// TwinCAT 3 PLC project PLC
// ProgramVersion: 3.1.4024.0
// libraries:
//   Tc2_Standard, * (Beckhoff Automation GmbH)
//   Tc2_System, * (Beckhoff Automation GmbH)
//   Tc3_Module, * (Beckhoff Automation GmbH)
//   VisuSymbols,3.5.10.0,System
// project tree:
//   DUTs/ Input.TcDUT, Output.TcDUT, WeldRobotIn.TcDUT, WeldRobotOut.TcDUT
//   / GlobalTextList.TcGTLO, PlcTask.TcTTO, Visualization Manager.TcVMO (not stored)
//   GVLs/ Fixt1.TcGVL, Fixt2.TcGVL, Gen.TcGVL, Global.TcGVL, GVL.TcGVL, HMI.TcGVL, MH.TcGVL, Safety.TcGVL, WeldRobot.TcGVL, WeldRobots.TcGVL
//   POUs/ Fixt2_Seq_Call.TcPOU, Fixt2_Seq_Call_1.TcPOU, Fixt2_Seq_Call_1_1.TcPOU, MAIN.TcPOU, Mode_Call.TcPOU, Fixt1_Seq_Call.TcPOU
//   POUs/Library/ FB_AutoSeq.TcPOU, FB_CylinderModule.TcPOU, FB_ModeCall.TcPOU, FB_PartMonitoring_Fixt2.TcPOU, FB_Trunion.TcPOU, FB_TurnTable_0_180.TcPOU, FB_Roller_Door.TcPOU, FB_PartMonitoring_Fixt1.TcPOU
//   VISUs/ Visualization.TcVIS
// real-time tasks:
//   TASK PlcTask: cycle T#10ms, priority 20, ADS port 350
// I/O:
//   DEVICE Device 1 (EtherCAT) (disabled), AmsNetId 192.168.4.1.2.1
//     Term 1 (EK1100) [EK1100 EtherCAT Coupler (2A E-Bus)]
//       Term 2 (EL1008) [EL1008 8Ch. Dig. Input 24V, 3ms]
//       Term 4 (EL1904) [EL1904, 4 Ch. Safety Input 24V, TwinSAFE]
//         modules: Module 1 (FSOES)
//       Term 5 (EL2904) [EL2904, 4 Ch. Safety Output 24V, 0.5A, TwinSAFE]
//         modules: Module 1 (FSOES), Module 2 (DO)
//       Term 6 (EL2008) [EL2008 8Ch. Dig. Output 24V, 0.5A]
//       Term 3 (EL6910) [EL6910, TwinSAFE PLC]
// variable links:
//   Device 1 (EtherCAT) <-> Device 1 (EtherCAT)/Term 1 (EK1100)/Term 3 (EL6910)
//     Term 1 (EK1100)/Term 5 (EL2904)/Module 1 (FSOES)/RxPDO/FSOE <-> ConnectionInputs/TwinSafeGroup1.Term 5 (EL2904) - Module 1 (FSOES)_4 TxPDO
//     Term 1 (EK1100)/Term 5 (EL2904)/Module 1 (FSOES)/TxPDO/FSOE <-> ConnectionOutputs/TwinSafeGroup1.Term 5 (EL2904) - Module 1 (FSOES)_4 RxPDO
//   Device 1 (EtherCAT) <-> Device 1 (EtherCAT)/Term 1 (EK1100)/Term 4 (EL1904)
//     Term 1 (EK1100)/Term 3 (EL6910)/ConnectionInputs/TwinSafeGroup1.Term 4 (EL1904) - Module 1 (FSOES)_3 TxPDO <-> Module 1 (FSOES)/RxPDO/FSOE
//     Term 1 (EK1100)/Term 3 (EL6910)/ConnectionOutputs/TwinSafeGroup1.Term 4 (EL1904) - Module 1 (FSOES)_3 RxPDO <-> Module 1 (FSOES)/TxPDO/FSOE
//   PLC/PLC Instance <-> Device 1 (EtherCAT)/Term 1 (EK1100)/Term 3 (EL6910)
//     PlcTask Outputs/Safety.Ack <-> StandardOutputs/TwinSafeGroup1.ErrorAcknowledgement_1
//     PlcTask Outputs/Safety.sRun <-> StandardOutputs/TwinSafeGroup1.Run_2

CONFIGURATION PLC
    RESOURCE PLC ON TwinCAT3
        TASK PlcTask(INTERVAL := T#10ms, PRIORITY := 20);
        PROGRAM MAIN WITH PlcTask : MAIN;
    END_RESOURCE
END_CONFIGURATION

// ---- DUTs/Input.TcDUT
TYPE Input :
STRUCT
i_Control_Pressure_Sw_In1_BPB1	:	BOOL	;	//	Control Pressure Switch Input 1-BPB1  
i_Control_Pressure_Sw_In2_BPB1	:	Bool	;	//	Control Pressure Switch Input 2-BPB1  
i_Valve_Pos_BGB1	:	Bool	;	//	Valve Position-BGB1
i_Reserve_BPB1_0_3	:	Bool	;	//	Free
i_CC6_Clamp_1_Sensor_HP	:	Bool	;	//	Clamping Circuit 6 Clamping Unit 1 sensor  HP
i_CC6_Clamp_1_Sensor_WP	:	Bool	;	//	Clamping Circuit 6 Clamping Unit 1 sensor  WP
i_CC4_Clamp_3_Sensor_HP	:	Bool	;	//	Clamping Circuit 4 Clamping Unit 3 sensor  HP
i_CC4_Clamp_3_Sensor_WP	:	Bool	;	//	Clamping Circuit 4 Clamping Unit 3 sensor  WP
i_PART_CONTROL_B13	:	Bool	;	//	PART CONTROL  B13
i_PART_CONTROL_B27	:	Bool	;	//	PART CONTROL  B27
i_PART_CONTROL_B14	:	Bool	;	//	PART CONTROL  B14
i_PART_CONTROL_B28	:	Bool	;	//	PART CONTROL  B28
i_Reserve_BGB1_1_4	:	Bool	;	//	Free
i_Reserve_BGB1_1_5	:	Bool	;	//	Free
i_KEC6Salvemodule12_1	:	BOOL	;	//	Connect to KEC6 Salve module 1.2
i_KEC6Salvemodule12_2	:	BOOL	;	//	Connect to KEC6 Salve module 1.2
i_Reserve_2_0	:	Bool	;	//	i_Reserve_2_0
i_Reserve_2_1	:	Bool	;	//	i_Reserve_2_1
i_Reserve_2_2	:	Bool	;	//	i_Reserve_2_2
i_Reserve_2_3	:	Bool	;	//	i_Reserve_2_3
i_Reserve_2_4	:	Bool	;	//	i_Reserve_2_4
i_Reserve_2_5	:	Bool	;	//	i_Reserve_2_5
i_Reserve_2_6	:	Bool	;	//	i_Reserve_2_6
i_Reserve_2_7	:	Bool	;	//	i_Reserve_2_7
i_Reserve_3_0	:	Bool	;	//	i_Reserve_3_0
i_Reserve_3_1	:	Bool	;	//	i_Reserve_3_1
i_Reserve_3_2	:	Bool	;	//	i_Reserve_3_2
i_Reserve_3_3	:	Bool	;	//	i_Reserve_3_3
i_Reserve_3_4	:	Bool	;	//	i_Reserve_3_4
i_Reserve_3_5	:	Bool	;	//	i_Reserve_3_5
i_Reserve_3_6	:	Bool	;	//	i_Reserve_3_6
i_Reserve_3_7	:	Bool	;	//	i_Reserve_3_7
i_CC4_Clamp_1_Sensor_HP	:	Bool	;	//	Clamping Circuit 4 Clamping Unit 1 sensor  HP
i_CC4_Clamp_1_Sensor_WP	:	Bool	;	//	Clamping Circuit 4 Clamping Unit 1 sensor  WP
i_CC4_Clamp_2_Sensor_HP	:	Bool	;	//	Clamping Circuit 4 Clamping Unit 2 sensor  HP
i_CC4_Clamp_2_Sensor_WP	:	Bool	;	//	Clamping Circuit 4 Clamping Unit 2 sensor  WP
i_CC2_Clamp_3_Sensor_HP	:	Bool	;	//	Clamping Circuit 2 Clamping Unit 3 sensor  HP
i_CC2_Clamp_3_Sensor_WP	:	Bool	;	//	Clamping Circuit 2 Clamping Unit 3 sensor  WP
i_PART_CONTROL_B12	:	Bool	;	//	PART CONTROL  B12
i_PART_CONTROL_B26	:	Bool	;	//	PART CONTROL  B26
i_PART_CONTROL_B11	:	Bool	;	//	PART CONTROL  B11
i_PART_CONTROL_B25	:	Bool	;	//	PART CONTROL  B25
i_PART_CONTROL_B10	:	Bool	;	//	PART CONTROL  B10
i_PART_CONTROL_B24	:	Bool	;	//	PART CONTROL  B24
i_Reserve_5_4	:	Bool	;	//	Free
i_Reserve_5_5	:	Bool	;	//	Free
i_Reserve_5_6	:	Bool	;	//	Free
i_Reserve_5_7	:	Bool	;	//	Free
i_Reserve_6_0	:	Bool	;	//	i_Reserve_6_0
i_Reserve_6_1	:	Bool	;	//	i_Reserve_6_1
i_Reserve_6_2	:	Bool	;	//	i_Reserve_6_2
i_Reserve_6_3	:	Bool	;	//	i_Reserve_6_3
i_Reserve_6_4	:	Bool	;	//	i_Reserve_6_4
i_Reserve_6_5	:	Bool	;	//	i_Reserve_6_5
i_Reserve_6_6	:	Bool	;	//	i_Reserve_6_6
i_Reserve_6_7	:	Bool	;	//	i_Reserve_6_7
i_Reserve_7_0	:	Bool	;	//	i_Reserve_7_0
i_Reserve_7_1	:	Bool	;	//	i_Reserve_7_1
i_Reserve_7_2	:	Bool	;	//	i_Reserve_7_2
i_Reserve_7_3	:	Bool	;	//	i_Reserve_7_3
i_Reserve_7_4	:	Bool	;	//	i_Reserve_7_4
i_Reserve_7_5	:	Bool	;	//	i_Reserve_7_5
i_Reserve_7_6	:	Bool	;	//	i_Reserve_7_6
i_Reserve_7_7	:	Bool	;	//	i_Reserve_7_7
i_CC3_Clamp_1_Sensor_HP	:	Bool	;	//	Clamping Circuit 3 Clamping Unit 1 sensor  HP
i_CC3_Clamp_1_Sensor_WP	:	Bool	;	//	Clamping Circuit 3 Clamping Unit 1 sensor  WP
i_CC3_Clamp_2_Sensor_HP	:	Bool	;	//	Clamping Circuit 3 Clamping Unit 2 sensor  HP
i_CC3_Clamp_2_Sensor_WP	:	Bool	;	//	Clamping Circuit 3 Clamping Unit 2 sensor  WP
i_CC3_Clamp_3_Sensor_HP	:	Bool	;	//	Clamping Circuit 3 Clamping Unit 3 sensor  HP
i_CC3_Clamp_3_Sensor_WP	:	Bool	;	//	Clamping Circuit 3 Clamping Unit 3 sensor  WP
i_PART_CONTROL_B7	:	Bool	;	//	PART CONTROL  B7
i_PART_CONTROL_B21	:	Bool	;	//	PART CONTROL  B21
i_PART_CONTROL_B6	:	Bool	;	//	PART CONTROL  B6
i_PART_CONTROL_B20	:	Bool	;	//	PART CONTROL  B20
i_PART_CONTROL_B5	:	Bool	;	//	PART CONTROL  B5
i_PART_CONTROL_B19	:	Bool	;	//	PART CONTROL  B19
i_Reserve_9_4	:	Bool	;	//	Free
i_Reserve_9_5	:	Bool	;	//	Free
i_KEC8Salvemodule22_1	:	BOOL	;	//	Connect to KEC8 Salve module 2.2
i_KEC8Salvemodule22_2	:	BOOL	;	//	Connect to KEC8 Salve module 2.2
i_Reserve_10_0	:	Bool	;	//	i_Reserve_10_0
i_Reserve_10_1	:	Bool	;	//	i_Reserve_10_1
i_Reserve_10_2	:	Bool	;	//	i_Reserve_10_2
i_Reserve_10_3	:	Bool	;	//	i_Reserve_10_3
i_Reserve_10_4	:	Bool	;	//	i_Reserve_10_4
i_Reserve_10_5	:	Bool	;	//	i_Reserve_10_5
i_Reserve_10_6	:	Bool	;	//	i_Reserve_10_6
i_Reserve_10_7	:	Bool	;	//	i_Reserve_10_7
i_Reserve_11_0	:	Bool	;	//	i_Reserve_11_0
i_Reserve_11_1	:	Bool	;	//	i_Reserve_11_1
i_Reserve_11_2	:	Bool	;	//	i_Reserve_11_2
i_Reserve_11_3	:	Bool	;	//	i_Reserve_11_3
i_Reserve_11_4	:	Bool	;	//	i_Reserve_11_4
i_Reserve_11_5	:	Bool	;	//	i_Reserve_11_5
i_Reserve_11_6	:	Bool	;	//	i_Reserve_11_6
i_Reserve_11_7	:	Bool	;	//	i_Reserve_11_7
i_CC1_Clamp_1_Sensor_HP	:	Bool	;	//	Clamping Circuit 1 Clamping Unit 1 sensor  HP
i_CC1_Clamp_1_Sensor_WP	:	Bool	;	//	Clamping Circuit 1 Clamping Unit 1 sensor  WP
i_CC1_Clamp_2_Sensor_HP	:	Bool	;	//	Clamping Circuit 1 Clamping Unit 2 sensor  HP
i_CC1_Clamp_2_Sensor_WP	:	Bool	;	//	Clamping Circuit 1 Clamping Unit 2 sensor  WP
i_CC1_Clamp_3_Sensor_HP	:	Bool	;	//	Clamping Circuit 1 Clamping Unit 3 sensor  HP
i_CC1_Clamp_3_Sensor_WP	:	Bool	;	//	Clamping Circuit 1 Clamping Unit 3 sensor  WP
i_PART_CONTROL_B4	:	Bool	;	//	PART CONTROL  B4
i_PART_CONTROL_B18	:	Bool	;	//	PART CONTROL  B18
i_PART_CONTROL_B3	:	Bool	;	//	PART CONTROL  B3
i_PART_CONTROL_B17	:	Bool	;	//	PART CONTROL  B17
i_PART_CONTROL_B2	:	Bool	;	//	PART CONTROL  B2
i_PART_CONTROL_B16	:	Bool	;	//	PART CONTROL  B16
i_Reserve_13_4	:	Bool	;	//	Free
i_Reserve_13_5	:	Bool	;	//	Free
i_Reserve_13_6	:	Bool	;	//	Free
i_Reserve_13_7	:	Bool	;	//	Free
i_Reserve_14_0	:	Bool	;	//	i_Reserve_14_0
i_Reserve_14_1	:	Bool	;	//	i_Reserve_14_1
i_Reserve_14_2	:	Bool	;	//	i_Reserve_14_2
i_Reserve_14_3	:	Bool	;	//	i_Reserve_14_3
i_Reserve_14_4	:	Bool	;	//	i_Reserve_14_4
i_Reserve_14_5	:	Bool	;	//	i_Reserve_14_5
i_Reserve_14_6	:	Bool	;	//	i_Reserve_14_6
i_Reserve_14_7	:	Bool	;	//	i_Reserve_14_7
i_Reserve_15_0	:	Bool	;	//	i_Reserve_15_0
i_Reserve_15_1	:	Bool	;	//	i_Reserve_15_1
i_Reserve_15_2	:	Bool	;	//	i_Reserve_15_2
i_Reserve_15_3	:	Bool	;	//	i_Reserve_15_3
i_Reserve_15_4	:	Bool	;	//	i_Reserve_15_4
i_Reserve_15_5	:	Bool	;	//	i_Reserve_15_5
i_Reserve_15_6	:	Bool	;	//	i_Reserve_15_6
i_Reserve_15_7	:	Bool	;	//	i_Reserve_15_7
i_CC2_Clamp_1_Sensor_HP	:	Bool	;	//	Clamping Circuit 2 Clamping Unit 1 sensor  HP
i_CC2_Clamp_1_Sensor_WP	:	Bool	;	//	Clamping Circuit 2 Clamping Unit 1 sensor  WP
i_CC2_Clamp_2_Sensor_HP	:	Bool	;	//	Clamping Circuit 2 Clamping Unit 2 sensor  HP
i_CC2_Clamp_2_Sensor_WP	:	Bool	;	//	Clamping Circuit 2 Clamping Unit 2 sensor  WP
i_PART_CONTROL_B9	:	Bool	;	//	PART CONTROL  B9
i_PART_CONTROL_B23	:	Bool	;	//	PART CONTROL  B23
i_PART_CONTROL_B8	:	Bool	;	//	PART CONTROL  B8
i_PART_CONTROL_B22	:	Bool	;	//	PART CONTROL  B22
i_Reserve_17_0	:	Bool	;	//	Free
i_Reserve_17_1	:	Bool	;	//	Free
i_Reserve_17_2	:	Bool	;	//	Free
i_Reserve_17_3	:	Bool	;	//	Free
i_Reserve_17_4	:	Bool	;	//	Free
i_Reserve_17_5	:	Bool	;	//	Free
i_Reserve_17_6	:	Bool	;	//	Free
i_Reserve_17_7	:	Bool	;	//	Free
i_Reserve_18_0	:	Bool	;	//	i_Reserve_18_0
i_Reserve_18_1	:	Bool	;	//	i_Reserve_18_1
i_Reserve_18_2	:	Bool	;	//	i_Reserve_18_2
i_Reserve_18_3	:	Bool	;	//	i_Reserve_18_3
i_Reserve_18_4	:	Bool	;	//	i_Reserve_18_4
i_Reserve_18_5	:	Bool	;	//	i_Reserve_18_5
i_Reserve_18_6	:	Bool	;	//	i_Reserve_18_6
i_Reserve_18_7	:	Bool	;	//	i_Reserve_18_7
i_Reserve_19_0	:	Bool	;	//	i_Reserve_19_0
i_Reserve_19_1	:	Bool	;	//	i_Reserve_19_1
i_Reserve_19_2	:	Bool	;	//	i_Reserve_19_2
i_Reserve_19_3	:	Bool	;	//	i_Reserve_19_3
i_Reserve_19_4	:	Bool	;	//	i_Reserve_19_4
i_Reserve_19_5	:	Bool	;	//	i_Reserve_19_5
i_Reserve_19_6	:	Bool	;	//	i_Reserve_19_6
i_Reserve_19_7	:	Bool	;	//	i_Reserve_19_7
i_Reserve_20_0	:	Bool	;	//	i_Reserve_20_0
i_Reserve_20_1	:	Bool	;	//	i_Reserve_20_1
i_Reserve_20_2	:	Bool	;	//	i_Reserve_20_2
i_Reserve_20_3	:	Bool	;	//	i_Reserve_20_3
i_Reserve_20_4	:	Bool	;	//	i_Reserve_20_4
i_Reserve_20_5	:	Bool	;	//	i_Reserve_20_5
i_Reserve_20_6	:	Bool	;	//	i_Reserve_20_6
i_Reserve_20_7	:	Bool	;	//	i_Reserve_20_7
i_Reserve_21_0	:	Bool	;	//	i_Reserve_21_0
i_Reserve_21_1	:	Bool	;	//	i_Reserve_21_1
i_Reserve_21_2	:	Bool	;	//	i_Reserve_21_2
i_Reserve_21_3	:	Bool	;	//	i_Reserve_21_3
i_Reserve_21_4	:	Bool	;	//	i_Reserve_21_4
i_Reserve_21_5	:	Bool	;	//	i_Reserve_21_5
i_Reserve_21_6	:	Bool	;	//	i_Reserve_21_6
i_Reserve_21_7	:	Bool	;	//	i_Reserve_21_7
i_Reserve_22_0	:	Bool	;	//	i_Reserve_22_0
i_Reserve_22_1	:	Bool	;	//	i_Reserve_22_1
i_Reserve_22_2	:	Bool	;	//	i_Reserve_22_2
i_Reserve_22_3	:	Bool	;	//	i_Reserve_22_3
i_Reserve_22_4	:	Bool	;	//	i_Reserve_22_4
i_Reserve_22_5	:	Bool	;	//	i_Reserve_22_5
i_Reserve_22_6	:	Bool	;	//	i_Reserve_22_6
i_Reserve_22_7	:	Bool	;	//	i_Reserve_22_7
i_Reserve_23_0	:	Bool	;	//	i_Reserve_23_0
i_Reserve_23_1	:	Bool	;	//	i_Reserve_23_1
i_Reserve_23_2	:	Bool	;	//	i_Reserve_23_2
i_Reserve_23_3	:	Bool	;	//	i_Reserve_23_3
i_Reserve_23_4	:	Bool	;	//	i_Reserve_23_4
i_Reserve_23_5	:	Bool	;	//	i_Reserve_23_5
i_Reserve_23_6	:	Bool	;	//	i_Reserve_23_6
i_Reserve_23_7	:	Bool	;	//	i_Reserve_23_7
i_CC5_Clamp_1_Sensor_HP	:	Bool	;	//	Clamping Circuit 5 Clamping Unit 1 sensor  HP
i_CC5_Clamp_1_Sensor_WP	:	Bool	;	//	Clamping Circuit 5 Clamping Unit 1 sensor  WP
i_PART_CONTROL_B1	:	Bool	;	//	PART CONTROL  B1
i_PART_CONTROL_B15	:	Bool	;	//	PART CONTROL  B15
i_Reserve_24_4	:	Bool	;	//	Free
i_Reserve_24_5	:	Bool	;	//	Free
i_Reserve_24_6	:	Bool	;	//	Free
i_Reserve_24_7	:	Bool	;	//	Free
i_Reserve_25_0	:	Bool	;	//	Free
i_Reserve_25_1	:	Bool	;	//	Free
i_Reserve_25_2	:	Bool	;	//	Free
i_Reserve_25_3	:	Bool	;	//	Free
i_Reserve_25_4	:	Bool	;	//	Free
i_Reserve_25_5	:	Bool	;	//	Free
i_Reserve_25_6	:	Bool	;	//	Free
i_Reserve_25_7	:	Bool	;	//	Free
i_Reserve_26_0	:	Bool	;	//	i_Reserve_26_0
i_Reserve_26_1	:	Bool	;	//	i_Reserve_26_1
i_Reserve_26_2	:	Bool	;	//	i_Reserve_26_2
i_Reserve_26_3	:	Bool	;	//	i_Reserve_26_3
i_Reserve_26_4	:	Bool	;	//	i_Reserve_26_4
i_Reserve_26_5	:	Bool	;	//	i_Reserve_26_5
i_Reserve_26_6	:	Bool	;	//	i_Reserve_26_6
i_Reserve_26_7	:	Bool	;	//	i_Reserve_26_7
i_Reserve_27_0	:	Bool	;	//	i_Reserve_27_0
i_Reserve_27_1	:	Bool	;	//	i_Reserve_27_1
i_Reserve_27_2	:	Bool	;	//	i_Reserve_27_2
i_Reserve_27_3	:	Bool	;	//	i_Reserve_27_3
i_Reserve_27_4	:	Bool	;	//	i_Reserve_27_4
i_Reserve_27_5	:	Bool	;	//	i_Reserve_27_5
i_Reserve_27_6	:	Bool	;	//	i_Reserve_27_6
i_Reserve_27_7	:	Bool	;	//	i_Reserve_27_7
i_Reserve_28_0	:	Bool	;	//	i_Reserve_28_0
i_Reserve_28_1	:	Bool	;	//	i_Reserve_28_1
i_Reserve_28_2	:	Bool	;	//	i_Reserve_28_2
i_Reserve_28_3	:	Bool	;	//	i_Reserve_28_3
i_Reserve_28_4	:	Bool	;	//	i_Reserve_28_4
i_Reserve_28_5	:	Bool	;	//	i_Reserve_28_5
i_Reserve_28_6	:	Bool	;	//	i_Reserve_28_6
i_Reserve_28_7	:	Bool	;	//	i_Reserve_28_7
i_Reserve_29_0	:	Bool	;	//	i_Reserve_29_0
i_Reserve_29_1	:	Bool	;	//	i_Reserve_29_1
i_Reserve_29_2	:	Bool	;	//	i_Reserve_29_2
i_Reserve_29_3	:	Bool	;	//	i_Reserve_29_3
i_Reserve_29_4	:	Bool	;	//	i_Reserve_29_4
i_Reserve_29_5	:	Bool	;	//	i_Reserve_29_5
i_Reserve_29_6	:	Bool	;	//	i_Reserve_29_6
i_Reserve_29_7	:	Bool	;	//	i_Reserve_29_7
i_Reserve_30_0	:	Bool	;	//	i_Reserve_30_0
i_Reserve_30_1	:	Bool	;	//	i_Reserve_30_1
i_Reserve_30_2	:	Bool	;	//	i_Reserve_30_2
i_Reserve_30_3	:	Bool	;	//	i_Reserve_30_3
i_Reserve_30_4	:	Bool	;	//	i_Reserve_30_4
i_Reserve_30_5	:	Bool	;	//	i_Reserve_30_5
i_Reserve_30_6	:	Bool	;	//	i_Reserve_30_6
i_Reserve_30_7	:	Bool	;	//	i_Reserve_30_7
i_Reserve_31_0	:	Bool	;	//	i_Reserve_31_0
i_Reserve_31_1	:	Bool	;	//	i_Reserve_31_1
i_Reserve_31_2	:	Bool	;	//	i_Reserve_31_2
i_Reserve_31_3	:	Bool	;	//	i_Reserve_31_3
i_Reserve_31_4	:	Bool	;	//	i_Reserve_31_4
i_Reserve_31_5	:	Bool	;	//	i_Reserve_31_5
i_Reserve_31_6	:	Bool	;	//	i_Reserve_31_6
i_Reserve_31_7	:	Bool	;	//	i_Reserve_31_7

END_STRUCT
END_TYPE

// ---- DUTs/Output.TcDUT
TYPE Output :
STRUCT
o_CC1_CLAMPING_UNIT1_3_WP	:	BOOL	;	//	Clamping Circuit 1 Clamping Unit 1-3  WP
o_CC1_CLAMPING_UNIT1_3_HP	:	Bool	;	//	Clamping Circuit 1 Clamping Unit 1-3  HP
o_CC2_CLAMPING_UNIT2_3_WP	:	Bool	;	//	Clamping Circuit 2 Clamping Unit 1-3  WP
o_CC2_CLAMPING_UNIT2_3_HP	:	Bool	;	//	Clamping Circuit 2 Clamping Unit 1-3  HP
o_CC3_CLAMPING_UNIT3_3_WP	:	Bool	;	//	Clamping Circuit 3 Clamping Unit 1-3  WP
o_CC3_CLAMPING_UNIT3_3_HP	:	Bool	;	//	Clamping Circuit 3 Clamping Unit 1-3  HP
o_CC4_CLAMPING_UNIT4_3_WP	:	Bool	;	//	Clamping Circuit 4 Clamping Unit 1-3  WP
o_CC4_CLAMPING_UNIT4_3_HP	:	Bool	;	//	Clamping Circuit 4 Clamping Unit 1-3  HP
o_CC5_CLAMPING_UNIT5_1_WP	:	Bool	;	//	Clamping Circuit 5 Clamping Unit 1  WP
o_CC5_CLAMPING_UNIT5_1_HP	:	Bool	;	//	Clamping Circuit 5 Clamping Unit 1  HP
o_CC6_CLAMPING_UNIT6_1_WP	:	Bool	;	//	Clamping Circuit 6 Clamping Unit 1  WP
o_CC6_CLAMPING_UNIT6_1_HP	:	Bool	;	//	Clamping Circuit 6 Clamping Unit 1  HP
o_RESERVE_1_4	:	Bool	;	//	Free
o_RESERVE_1_5	:	Bool	;	//	Free
o_RESERVE_1_6	:	Bool	;	//	Free
o_RESERVE_1_7	:	Bool	;	//	Free
o_RESERVE_2_0	:	Bool	;	//	Free
o_RESERVE_2_1	:	Bool	;	//	Free
o_RESERVE_2_2	:	Bool	;	//	Free
o_RESERVE_2_3	:	Bool	;	//	Free
o_RESERVE_2_4	:	Bool	;	//	Free
o_RESERVE_2_5	:	Bool	;	//	Free
o_RESERVE_2_6	:	Bool	;	//	Free
o_RESERVE_2_7	:	Bool	;	//	Free
o_RESERVE_3_0	:	Bool	;	//	Free
o_RESERVE_3_1	:	Bool	;	//	Free
o_RESERVE_3_2	:	Bool	;	//	Free
o_RESERVE_3_3	:	Bool	;	//	Free
o_RESERVE_3_4	:	Bool	;	//	Free
o_RESERVE_3_5	:	Bool	;	//	Free
o_RESERVE_3_6	:	Bool	;	//	Free
o_RESERVE_3_7	:	Bool	;	//	Free

END_STRUCT
END_TYPE

// ---- DUTs/WeldRobotIn.TcDUT
TYPE WeldRobotIn :
STRUCT
	iMainJobActive: BOOL;
	iAtParkPos: BOOL;
	iWeldOn:BOOL;
	iProgramNumber: INT;
	Pos_20      : BOOL;
    Pos_0       : BOOL;   // 0 degree feedback
    Pos_M45     : BOOL;
    Pos_M80     : BOOL;
	LS_0        : BOOL;
    LS_180      : BOOL;
	
END_STRUCT
END_TYPE

// ---- DUTs/WeldRobotOut.TcDUT
TYPE WeldRobotOut :
STRUCT
	oProgramNumber: INT;
	oWeldStart: BOOL;
	Move_20     : BOOL;
    Move_0      : BOOL;   // Move to 0 degree
    Move_M45    : BOOL;
    Move_M80    : BOOL;
	Motor_CW_0    : BOOL;
    Motor_CCW_180   : BOOL;
END_STRUCT
END_TYPE

// ---- GVLs/Fixt1.TcGVL
{attribute 'qualified_only'}
VAR_GLOBAL
	I AT %I* :Input;
	O AT %Q* :Output;
	Seq:FB_AutoSeq;
	Trunion:FB_Trunion;
END_VAR

// ---- GVLs/Fixt2.TcGVL
{attribute 'qualified_only'}
VAR_GLOBAL
	I AT %I* :Input;
	O AT %Q* :Output;
	Seq:FB_AutoSeq;
	Trunion:FB_Trunion;
END_VAR

// ---- GVLs/Gen.TcGVL
{attribute 'qualified_only'}
VAR_GLOBAL
	ix_RCD_fuse_fdb	AT	%I*	:	BOOL	;
ix_24VDC_Fuse_TBA1_OK	AT	%I*	:	Bool	;
ix_AIEnergyMeterCbFbOK	AT	%I*	:	BOOL	;
ix_24VDC_Fuse1_OK	AT	%I*	:	Bool	;
ix_24VDC_Fuse2_OK	AT	%I*	:	Bool	;
ix_24VDC_Fuse3_OK	AT	%I*	:	Bool	;
ix_Reserve_0_6	AT	%I*	:	Bool	;
ix_24VDC_PowerSupply_Lightning_OK	AT	%I*	:	Bool	;
ix_TBA2FCB8_Cb_fbb	AT	%I*	:	BOOL	;
ix_AirConditioner_MainCabinet_Error_fdb	AT	%I*	:	Bool	;
ix_RD1_PowerSupply_fdb	AT	%I*	:	Bool	;
ix_RD2_PowerSupply_fdb	AT	%I*	:	Bool	;
ix_Ventilation_Malfunction_fdb	AT	%I*	:	Bool	;
ix_Ventilation_Operating_fdb	AT	%I*	:	Bool	;
ix_BGB1_door_lmt_Sw1_fdb	AT	%I*	:	Bool	;
ix_BGB1_door_lmt_Sw2_fdb	AT	%I*	:	Bool	;
ix_PowerSource_AW1_PowerSupply_fdb	AT	%I*	:	Bool	;
ix_PowerSource_AW1_ON	AT	%I*	:	Bool	;
ix_PowerSource_AW2_PowerSupply_fdb	AT	%I*	:	Bool	;
ix_PowerSource_AW2_ON	AT	%I*	:	Bool	;
ix_RC1_PowerSupply_OK	AT	%I*	:	Bool	;
ix_RC2_PowerSupply_OK	AT	%I*	:	Bool	;
ix_PB_RD2_Open	AT	%I*	:	Bool	;
ix_PB_RD2_Close	AT	%I*	:	Bool	;
ix_RD2_isReady	AT	%I*	:	Bool	;
ix_RD2_isOpen_top	AT	%I*	:	Bool	;
ix_RD2_safetyedge	AT	%I*	:	Bool	;
ix_CompressedAir_Pressure_OK	AT	%I*	:	Bool	;
ix_FlowRate_Sensor_outputA	AT	%I*	:	Bool	;
ix_FlowRate_Sensor_outputB	AT	%I*	:	Bool	;
ix_WireEnd_Sensor_R1	AT	%I*	:	Bool	;
ix_WireEnd_Sensor_R2	AT	%I*	:	Bool	;
ix_PB_PowerON	AT	%I*	:	Bool	;
ix_PB_PowerOFF	AT	%I*	:	Bool	;
ix_PB_Reset	AT	%I*	:	Bool	;
ix_PB_Start	AT	%I*	:	Bool	;
ix_PB_ack_LB	AT	%I*	:	Bool	;
ix_PB_Rbt_Start_Stop	AT	%I*	:	Bool	;
ix_RD1_isReady	AT	%I*	:	Bool	;
ix_RD1_isOpen_top	AT	%I*	:	Bool	;
ix_RD1_Safetyedge	AT	%I*	:	Bool	;
ix_ControlOn	AT	%I*	:	BOOL	;
ix_Reserve_201_2	AT	%I*	:	Bool	;
ix_Reserve_201_3	AT	%I*	:	Bool	;
ix_Reserve_201_4	AT	%I*	:	Bool	;
ix_Reserve_201_5	AT	%I*	:	Bool	;
ix_PB_preAck_UB2	AT	%I*	:	Bool	;
ix_Reserve_201_7	AT	%I*	:	Bool	;
qx_Light_InputArea_ON	AT	%Q*	:	Bool	;
qx_Light_WorkArea_ON	AT	%Q*	:	Bool	;
qx_AirConditionerTurn_ON	AT	%Q*	:	Bool	;
qx_CabinetLight_ON	AT	%Q*	:	Bool	;
qx_ControlPixelCameraST9100	AT	%Q*	:	Bool	;
qx_Valve_CompressedAir_ON	AT	%Q*	:	Bool	;
qx_Valve_GasON_Rob1	AT	%Q*	:	Bool	;
qx_Valve_blowOut_Rob1	AT	%Q*	:	Bool	;
qx_Valve_GasON_Rob2	AT	%Q*	:	Bool	;
qx_Valve_blowOut_Rob2	AT	%Q*	:	Bool	;
qx_Valve_GasON_Rob3	AT	%Q*	:	Bool	;
qx_Valve_blowOut_Rob3	AT	%Q*	:	Bool	;
qx_Valve_GasON_Rob4	AT	%Q*	:	Bool	;
qx_Valve_blowOut_Rob4	AT	%Q*	:	Bool	;
qx_Reserve_1_6	AT	%Q*	:	Bool	;
qx_IL_preAck_Box_UB2	AT	%Q*	:	Bool	;
qx_Reserve_2_0	AT	%Q*	:	Bool	;
qx_Reserve_2_1	AT	%Q*	:	Bool	;
qx_Reserve_2_2	AT	%Q*	:	Bool	;
qx_Reserve_2_3	AT	%Q*	:	Bool	;
qx_Reserve_2_4	AT	%Q*	:	Bool	;
qx_Reserve_2_5	AT	%Q*	:	Bool	;
qx_Reserve_2_6	AT	%Q*	:	Bool	;
qx_Reserve_2_7	AT	%Q*	:	Bool	;
qx_Reserve_3_0	AT	%Q*	:	Bool	;
qx_Reserve_3_1	AT	%Q*	:	Bool	;
qx_Reserve_3_2	AT	%Q*	:	Bool	;
qx_Reserve_3_3	AT	%Q*	:	Bool	;
qx_Reserve_3_4	AT	%Q*	:	Bool	;
qx_Reserve_3_5	AT	%Q*	:	Bool	;
qx_Reserve_3_6	AT	%Q*	:	Bool	;
qx_Reserve_3_7	AT	%Q*	:	Bool	;
qx_RD2_open_narrow_hight	AT	%Q*	:	Bool	;
qx_RD2_open_FullHight	AT	%Q*	:	Bool	;
qx_RD2_close	AT	%Q*	:	Bool	;
qx_Ventilation_ON	AT	%Q*	:	Bool	;
qx_Reserve_6_0	AT	%Q*	:	Bool	;
qx_Reserve_6_1	AT	%Q*	:	Bool	;
qx_Reserve_6_2	AT	%Q*	:	Bool	;
qx_Reserve_6_3	AT	%Q*	:	Bool	;
qx_IL_PowerON	AT	%Q*	:	Bool	;
qx_IL_Reset_PB	AT	%Q*	:	Bool	;
qx_IL_Start_PB	AT	%Q*	:	Bool	;
qx_IL_ack_LB_PB	AT	%Q*	:	Bool	;
qx_IL_RbtStartStop_PB	AT	%Q*	:	Bool	;
qx_Reserve_200_5	AT	%Q*	:	Bool	;
qx_Reserve_200_6	AT	%Q*	:	Bool	;
qx_Reserve_200_7	AT	%Q*	:	Bool	;
qx_Reserve_201_0	AT	%Q*	:	Bool	;
qx_Reserve_201_1	AT	%Q*	:	Bool	;
qx_Reserve_201_2	AT	%Q*	:	Bool	;
qx_Reserve_201_3	AT	%Q*	:	Bool	;
qx_Reserve_201_4	AT	%Q*	:	Bool	;
qx_Reserve_201_5	AT	%Q*	:	Bool	;
qx_Reserve_201_6	AT	%Q*	:	Bool	;
qx_Reserve_201_7	AT	%Q*	:	Bool	;
qx_RD1_open_narrow_hight	AT	%Q*	:	Bool	;
qx_RD1_open_fullHight	AT	%Q*	:	Bool	;
qx_RD1_close	AT	%Q*	:	Bool	;
qx_Reserve_202_3	AT	%Q*	:	Bool	;

END_VAR

// ---- GVLs/Global.TcGVL
{attribute 'qualified_only'}
VAR_GLOBAL
	ModeMang:FB_ModeCall;
	Clamp_1:FB_CylinderModule;
	Clamp_2:FB_CylinderModule;
	Clamp_3:FB_CylinderModule;
	Clamp_4:FB_CylinderModule;
	Clamp_5:FB_CylinderModule;
	Clamp_6:FB_CylinderModule;
	RD1:FB_Roller_Door;
	RD2:FB_Roller_Door;
	Htable:FB_TurnTable_0_180;
END_VAR

// ---- GVLs/GVL.TcGVL
{attribute 'qualified_only'}
VAR_GLOBAL
	start AT %I*:BOOL;
	start1 AT %I*:BOOL;
	FB_ModeCall_0: FB_ModeCall;
END_VAR

// ---- GVLs/HMI.TcGVL
{attribute 'qualified_only'}
VAR_GLOBAL
	Cycle_Start:BOOL;
	Cycle_Stop:BOOL;
	AutoMode:BOOL;
	ManualMode:BOOL;
	Estop:BOOL;
	Reset:BOOL;
	
END_VAR

// ---- GVLs/MH.TcGVL
{attribute 'qualified_only'}
VAR_GLOBAL
//qx_7102R1_CellToHandling	AT	%Q*	:	//udt_HDL_CellToHandling	;	//	
qStatus	AT	%Q*	:	WORD	;	//	0 Auto -- 1 Auto Startup -- 2 Manual -- 3 Error -- 4 LineMode -- 5 PowerOn -- 6 EnergySave -- 7 SafeOk
qTime_Stamp	AT	%Q*	:	DATE_AND_TIME	;	//	
qPartId	AT	%Q*	:	DINT	;	//	Unique Part Id (DMC Serial Number)
qState	AT	%Q*	:	BOOL	;	//	Part state 0=OK, 1=NOK
qPartType	AT	%Q*	:	BOOL	;	//	Part type 1=Long, 0=Short
qExists	AT	%Q*	:	BOOL	;	//	Part exist
qRequest	AT	%Q*	:	USINT	;	//	20 - Pick, 10 - Drop
qRequestPartType	AT	%Q*	:	BOOL	;	//	Part types
qGateOpened	AT	%Q*	:	BOOL	;	//	Handling gate opened
qGateClosed	AT	%Q*	:	BOOL	;	//	Handling gate closed
qFixtureReady	AT	%Q*	:	BOOL	;	//	Postioner in Cube
qRaiseEnable1	AT	%Q*	:	BOOL	;	//	Handshake for raise to go all the way OUT
qRaiseEnable2	AT	%Q*	:	BOOL	;	//	Handshake for raise to go all the way OUT
qReduceEnable1	AT	%Q*	:	BOOL	;	//	Handshake for reduce to go all the way IN
qReduceEnable2	AT	%Q*	:	BOOL	;	//	Handshake for reduce to go all the way IN
qPickJobAck	AT	%Q*	:	BOOL	;	//	Handshake for pick job end
qDropJobAck	AT	%Q*	:	BOOL	;	//	Handshake for drop job end
qHold	AT	%Q*	:	BOOL	;	//	Robot hold
qGripper1ReadyToClose	AT	%Q*	:	BOOL	;	//	Gripper1ReadyToClose
qGripper1ReadyToOpen	AT	%Q*	:	BOOL	;	//	Gripper1ReadyToOpen
qGripper2ReadyToClose	AT	%Q*	:	BOOL	;	//	Gripper2ReadyToClose
qGripper2ReadyToOpen	AT	%Q*	:	BOOL	;	//	Gripper2ReadyToOpen
qFeatureBit6	AT	%Q*	:	BOOL	;	//	Free use
qFeatureBit7	AT	%Q*	:	BOOL	;	//	Free use
//	AT	%Q*	:		;	//	
//ix_7102R1_HandlingToCell	AT	%I*	:	//udt_HDL_HandlingToCell	;	//	
iStatus	AT	%I*	:	WORD	;	//	0 Auto -- 1 Auto Startup -- 2 Manual -- 3 Error -- 4 LineMode -- 5 PowerOn -- 6 EnergySave -- 7 SafeOk
iPartId	AT	%I*	:	DINT	;	//	Unique Part Id (DMC Serial Number)
iState	AT	%I*	:	BOOL	;	//	Part state 0=OK, 1=NOK
iPartType	AT	%I*	:	BOOL	;	//	Part type 1=Long, 0=Short
iExists	AT	%I*	:	BOOL	;	//	Part exist
iGateOpenRequest	AT	%I*	:	BOOL	;	//	Open handling gate
iGateCloseRequest	AT	%I*	:	BOOL	;	//	Close handling gate
iPickJobProceed	AT	%I*	:	BOOL	;	//	Pick job active
iDropJobProceed	AT	%I*	:	BOOL	;	//	Drop job active
iRaiseFinished1	AT	%I*	:	BOOL	;	//	Handshake for raise/ Robot reach at out off fixture pos
iRaiseFinished2	AT	%I*	:	BOOL	;	//	Handshake for reduce/Robot reach at into fixture pos
iReduceFinished1	AT	%I*	:	BOOL	;	//	Handshake for pick job end
iReduceFinished2	AT	%I*	:	BOOL	;	//	Handshake for drop job end
iPickJobOK	AT	%I*	:	BOOL	;	//	Robot in station area/robot infront of cell area
iDropJobOK	AT	%I*	:	BOOL	;	//	PickJobOK
iInArea	AT	%I*	:	BOOL	;	//	DropJobOK
iPickDropProceed	AT	%I*	:	BOOL	;	//	InArea
iGripper1ClosedAck	AT	%I*	:	BOOL	;	//	PickDropProceed
iGripper1OpenedAck	AT	%I*	:	BOOL	;	//	Gripper1OpenedAck
iGripper2ClosedAck	AT	%I*	:	BOOL	;	//	Gripper2ClosedAck
iGripper2OpenedAck	AT	%I*	:	BOOL	;	//	Gripper2OpenedAck
iFeatureBit6	AT	%I*	:	BOOL	;	//	Free use
iFeatureBit7	AT	%I*	:	BOOL	;	//	Free use

END_VAR

// ---- GVLs/Safety.TcGVL
{attribute 'qualified_only'}
VAR_GLOBAL
		ixf_CA1_PowerON_vs	AT	%I*	:	BOOL	;	//	
	ixf_RD2_PowerON_vs	AT	%I*	:	Bool	;	//	
	ixf_FXC1_Safe_24VDC_vs	AT	%I*	:	Bool	;	//	
	ixf_FXC2_Safe_24VDC_vs	AT	%I*	:	Bool	;	//	
	ixf_AW1_PowerSource_vs	AT	%I*	:	Bool	;	//	
	ixf_AW2_PowerSource_vs	AT	%I*	:	Bool	;	//	
	ixf_FXC1_Safe_AirON_vs	AT	%I*	:	Bool	;	//	
	ixf_FXC2_Safe_AirON_vs	AT	%I*	:	Bool	;	//	
	ixf_CA1_EStop_ch1	AT	%I*	:	Bool	;	//	
	ixf_UB3_EStop_ch1	AT	%I*	:	Bool	;	//	
	ixf_UB2_EStop_ch1	AT	%I*	:	Bool	;	//	
	ixf_RD2_isClosed_ch1	AT	%I*	:	Bool	;	//	
	ixf_CA1_EStop_ch2	AT	%I*	:	Bool	;	//	
	ixf_UB3_EStop_ch2	AT	%I*	:	Bool	;	//	
	ixf_UB2_EStop_ch2	AT	%I*	:	Bool	;	//	
	ixf_RD2_isClosed_ch2	AT	%I*	:	Bool	;	//	
	//ixf_CA1_EStop_ch1_vs	AT	%I*	:	Bool	;	//	
	//ixf_UB3_EStop_ch1_vs	AT	%I*	:	Bool	;	//	
	//ixf_UB2_EStop_ch1_vs	AT	%I*	:	Bool	;	//	
	//ixf_RD2_isClosed_ch1_vs	AT	%I*	:	Bool	;	//	
	//ixf_CA1_EStop_ch2_vs	AT	%I*	:	Bool	;	//	
	//ixf_UB3_EStop_ch2_vs	AT	%I*	:	Bool	;	//	
	//ixf_UB2_EStop_ch2_vs	AT	%I*	:	Bool	;	//	
	//ixf_RD2_isClosed_ch2_vs	AT	%I*	:	Bool	;	//	
	//ixf_Reserve_300700_0	AT	%I*	:	Bool	;	//	
	//ixf_Reserve_300700_1	AT	%I*	:	Bool	;	//	
	//ixf_Reserve_300700_2	AT	%I*	:	Bool	;	//	
	//ixf_Reserve_300700_3	AT	%I*	:	Bool	;	//	
	//ixf_Reserve_300700_4	AT	%I*	:	Bool	;	//	
	//ixf_Reserve_300700_5	AT	%I*	:	Bool	;	//	
	//ixf_Reserve_300700_6	AT	%I*	:	Bool	;	//	
	//ixf_Reserve_300700_7	AT	%I*	:	Bool	;	//	
	//ixf_RD1_PowerON_vs	AT	%I*	:	Bool	;	//	
	ixf_UB1_EStop_ch1	AT	%I*	:	Bool	;	//	
	ixf_LB1_InputArea_ch1	AT	%I*	:	Bool	;	//	
	ixf_SW_AutomaticMode	AT	%I*	:	Bool	;	//	
	ixf_RD1_isClosed_ch1	AT	%I*	:	Bool	;	//	
	ixf_UB1_EStop_ch2	AT	%I*	:	Bool	;	//	
	ixf_SW_ManualMode	AT	%I*	:	Bool	;	//	
	ixf_RD1_isClosed_ch2	AT	%I*	:	Bool	;	//	
	//ixf_UB1_EStop_ch1_vs	AT	%I*	:	Bool	;	//	
	//ixf_LB1_InputArea_vs	AT	%I*	:	Bool	;	//	
	//ixf_SW_AutomaticMode_vs	AT	%I*	:	Bool	;	//	
	//ixf_RD1_isClosed_ch1_vs	AT	%I*	:	Bool	;	//	
	//ixf_UB1_EStop_ch2_vs	AT	%I*	:	Bool	;	//	
	//ixf_SW_ManualMode_vs	AT	%I*	:	Bool	;	//	
	//ixf_RD1_isClosed_ch2_vs	AT	%I*	:	Bool	;	//	
	//ixf_Reserve_30150_0	AT	%I*	:	Bool	;	//	
	//ixf_Reserve_30150_1	AT	%I*	:	Bool	;	//	
	//ixf_Reserve_30150_2	AT	%I*	:	Bool	;	//	
	//ixf_Reserve_30150_3	AT	%I*	:	Bool	;	//	
	//ixf_Reserve_30150_4	AT	%I*	:	Bool	;	//	
	//ixf_Reserve_30150_5	AT	%I*	:	Bool	;	//	
	//ixf_Reserve_30150_6	AT	%I*	:	Bool	;	//	
	//ixf_Reserve_30150_7	AT	%I*	:	Bool	;	//	Seq_Reset_WM
	qxf_CA1_PowerON	AT	%Q*	:	Bool	;	//	
	qxf_RD2_PowerON	AT	%Q*	:	Bool	;	//	
	qxf_FXC1_Safe_24VDC	AT	%Q*	:	Bool	;	//	
	qxf_FXC2_Safe_24VDC	AT	%Q*	:	Bool	;	//	
	qxf_AW1_PowerON	AT	%Q*	:	Bool	;	//	
	qxf_AW2_PowerON	AT	%Q*	:	Bool	;	//	
	qxf_FXC1_Safe_AirON	AT	%Q*	:	Bool	;	//	
	qxf_FXC2_Safe_AirON	AT	%Q*	:	Bool	;	//	
	qxf_Reserve_30020_0	AT	%Q*	:	Bool	;	//	
	qxf_Reserve_30020_1	AT	%Q*	:	Bool	;	//	
	qxf_Reserve_30020_2	AT	%Q*	:	Bool	;	//	
	qxf_Reserve_30020_3	AT	%Q*	:	Bool	;	//	
	qxf_RD1_PowerON	AT	%Q*	:	Bool	;	//	
	qxf_Reserve_30100_1	AT	%Q*	:	Bool	;	//	
	qxf_Reserve_30100_2	AT	%Q*	:	Bool	;	//	
	qxf_Reserve_30100_3	AT	%Q*	:	BOOL	;	//	
	sRun AT	%Q*	:BOOL;
	Ack AT	%Q*	:BOOL;
	

END_VAR

// ---- GVLs/WeldRobot.TcGVL
{attribute 'qualified_only'}
VAR_GLOBAL
	In AT %I*:WeldRobotIn;
	Out AT %Q*:WeldRobotOut;
END_VAR

// ---- GVLs/WeldRobots.TcGVL
{attribute 'qualified_only'}
VAR_GLOBAL
	
END_VAR

// ---- POUs/MAIN.TcPOU
PROGRAM MAIN
VAR
END_VAR

END_PROGRAM

// ---- POUs/Library/FB_AutoSeq.TcPOU
FUNCTION_BLOCK FB_AutoSeq
VAR
	
	sRegularCycle: BOOL;
	sJumpWeldSideCycle: BOOL;
	MainJobActive: BOOL;
	temp: BOOL;
END_VAR

VAR_INPUT
	iAutorunning: BOOL;
	iInputAreaActive: BOOL;
	iHTableAt_0_DegreeFB: BOOL;
	iPartPresent: BOOL;
	iWeldRobotAtSafeArea: BOOL;
	iStationDeactivate: BOOL;
	iWorkAreaActive: BOOL;
	iTrunionAt_0_DegreeFB: BOOL;
	iHDLRbtAtSafeArea: BOOL;
	iRollerDoor1CLosed: BOOL;
	iHTableAt_180_DegreeFB: BOOL;
	iRollerDoor2CLosed: BOOL;
	iRawPartPresent1: BOOL;
	iRawPartPresent2: BOOL;
	iRawPartPresent3: bool;
	iRawPartPresent4: BOOL;
	iValve1Home: BOOL;
	iValve2Home: BOOL;
	iValve3Home: BOOL;
	iValve4Home: BOOL;
	iValve5Home: BOOL;
	iValve6Home: BOOL;
	iValve1Work: BOOL;
	iValve2Work: BOOL;
	iValve3Work: BOOL;
	iValve4Work: BOOL;
	iValve5Work: BOOL;
	iValve6Work: BOOL;
	iTrunionAt_20_DegreeFB: BOOL;
	iTrunionAt_minus80_DegreeFB: BOOL;
	iTrunionAt_minus45_DegreeFB: BOOL;
	iRollerDoor1Opened: BOOL;
	iRollerDoor2Opened: BOOL;
	iAuthorization: BOOL;
	iMainJobActive: BOOL;
	iWeldOn:BOOL;
	iHDLGateopenRequest: BOOL;
	iReducedEnable1Finished: BOOL;
	iReducedEnable2Finished: BOOL;
	iHDLGripperClosedFB1: BOOL;
	iHDLGripperClosedFB2: BOOL;
	iHDLRaisedEnable1Finished: BOOL;
	iHDLRaisedEnable2Finished: BOOL;
	iHDLRobotInArea: BOOL;
	iHDLPickJobACK: BOOL;
	iProgramNumber: INT;
END_VAR
VAR RETAIN
	Step: INT;
END_VAR
VAR PERSISTENT
	Steps: INT;
END_VAR
VAR_OUTPUT
	oResetAutoCHain: BOOL;
	
	oHTableStart_0_Degree_OP: BOOL;
	oRollerDoor1Close_OP: BOOL;
	oRollerDoor2Close_OP: BOOL;
	oHTableStart_180_Degree_OP: BOOL;
	oValve1Home: BOOL;
	oValve1Home1: BOOL;
	oValve1Home2: BOOL;
	oValve1Home3: BOOL;
	oValve1Home4: BOOL;
	oValve1Home5: BOOL;
	oValve1Home6: BOOL;
	oTrunionRotate_20_Degree_OP: BOOL;
	oTrunionRotate_0_Degree_OP: BOOL;
	oRollerDoor1Opens_OP: BOOL;
	oRollerDoor2Opens_OP: BOOL;
	oLightcurtainMute: BOOL;
	oValve1Work1: BOOL;
	oValve1Work3: BOOL;
	oValve1Work5: BOOL;
	oAuthorization: BOOL;
	oTrunionRotate_minus80_Degree_OP: BOOL;
	oTrunionRotate_minus45_Degree_OP: BOOL;
	oValve1Work2: BOOL;
	oValve1Work4: BOOL;
	oValve1Work6: BOOL;
	oProgramNumber: INT;
	oWeldStart: BOOL;
	oFixtureReady: BOOL;
	oPickJobReady: BOOL;
	oReducedEnable1: BOOL;
	oReducedEnable2: BOOL;
	oGripperCloseRequest1: BOOL;
	oGripperCloseRequest2: BOOL;
	oHDLRaisedEnable1: BOOL;
	oHDLRaisedEnable2: BOOL;
	oHDLPickJobACK: BOOL;
END_VAR

CASE step OF
	0:// Step0- Idle
	IF iAutorunning THEN
		oResetAutoCHain:= TRUE;
		
		Step:=10;
	END_IF;
	10:// Step10- Init
	IF iAutorunning AND iInputAreaActive 
           AND iTrunionAt_0_DegreeFB AND NOT iPartPresent 
           AND iWeldRobotAtSafeArea AND NOT iStationDeactivate 
           THEN
		   sRegularCycle:= TRUE;
		   oHTableStart_0_Degree_OP:= TRUE;
		   Step:=20;
	ELSIF iAutorunning AND iWorkAreaActive 
           AND iTrunionAt_0_DegreeFB AND NOT iPartPresent 
           AND iWeldRobotAtSafeArea AND NOT iStationDeactivate 
           THEN
		   sJumpWeldSideCycle:= TRUE;
		   Step:=280;
	ELSIF iAutorunning AND iInputAreaActive 
           AND iTrunionAt_0_DegreeFB AND NOT iPartPresent 
           AND iWeldRobotAtSafeArea AND iStationDeactivate
		   THEN
		   IF iStationDeactivate AND iWeldRobotAtSafeArea
			   AND iInputAreaActive
			   THEN
			   oRollerDoor1Close_OP:= TRUE;    
		   END_IF;
		   IF iStationDeactivate AND iWeldRobotAtSafeArea
			   AND iInputAreaActive
			   AND iTrunionAt_0_DegreeFB AND NOT MainJobActive AND iRollerDoor1CLosed
			   THEN 
			   oHTableStart_180_Degree_OP:= TRUE;
		   END_IF;
		   IF iStationDeactivate AND iWeldRobotAtSafeArea AND iRollerDoor2CLosed
			   AND iHDLRbtAtSafeArea AND iWorkAreaActive
			   AND iTrunionAt_0_DegreeFB AND NOT MainJobActive AND iHTableAt_180_DegreeFB
			   THEN
			   temp:=TRUE;
		   END_IF
		   IF iStationDeactivate AND iWeldRobotAtSafeArea
			   AND iHDLRbtAtSafeArea AND iWorkAreaActive AND iRollerDoor2CLosed
			   AND iTrunionAt_0_DegreeFB AND NOT MainJobActive AND iHTableAt_180_DegreeFB
			   THEN
			   oHTableStart_0_Degree_OP:= TRUE;
		   END_IF;
		   IF iHTableAt_0_DegreeFB AND iWeldRobotAtSafeArea
			   AND iInputAreaActive
			   AND iTrunionAt_0_DegreeFB AND NOT MainJobActive AND iRollerDoor1CLosed
			   THEN
			   Step:=0;
			END_IF;     
	END_IF;
	20:// Step20- all Valve Home Commd
	IF iAutorunning AND iInputAreaActive AND sRegularCycle
        AND iHTableAt_0_DegreeFB AND NOT iPartPresent 
        AND NOT iRawPartPresent1 AND NOT iRawPartPresent2
		AND NOT iRawPartPresent3 AND NOT iRawPartPresent4
        AND NOT iStationDeactivate 
        THEN
		oValve1Home1:= TRUE;
		oValve1Home2:= TRUE;
		oValve1Home3:= TRUE;
		oValve1Home4:= TRUE;
		oValve1Home5:= TRUE;
		oValve1Home6:= TRUE;
		Step:=30;
	ELSIF iAutorunning AND iInputAreaActive AND sRegularCycle
        AND iHTableAt_0_DegreeFB AND NOT iPartPresent 
        AND  iRawPartPresent1 AND iRawPartPresent2
		AND NOT iRawPartPresent3 AND NOT iRawPartPresent4
        AND NOT iStationDeactivate
		THEN 
		Step:=777;
	ELSIF iAutorunning AND iInputAreaActive AND sRegularCycle
        AND iHTableAt_0_DegreeFB AND NOT iPartPresent 
        AND  iRawPartPresent1 AND iRawPartPresent2
		AND  iRawPartPresent3 AND iRawPartPresent4
        AND NOT iStationDeactivate
		THEN 
		Step:=777;
	END_IF;
				
    30:// Step30- Trunion 20 degree
	IF iAutorunning AND iInputAreaActive AND sRegularCycle
        AND iHTableAt_0_DegreeFB  
        AND NOT iRawPartPresent1 AND NOT iRawPartPresent2
		AND NOT iRawPartPresent3 AND NOT iRawPartPresent4
        AND NOT iStationDeactivate AND iValve1Home AND iValve2Home
		AND iValve3Home AND iValve4Home AND iValve5Home
		AND iValve6Home
        THEN
		oTrunionRotate_20_Degree_OP:= TRUE;
		Step:=40;
	END_IF;
	40:// Step40- Roller Door 1 open CMD
	IF iAutorunning AND iInputAreaActive
        AND iHTableAt_0_DegreeFB  AND iTrunionAt_20_DegreeFB
        AND NOT iRawPartPresent1 AND NOT iRawPartPresent2
		AND NOT iRawPartPresent3 AND NOT iRawPartPresent4
        AND NOT iStationDeactivate 
        THEN
		oRollerDoor1Opens_OP:= TRUE;
		Step:=50;
	END_IF;
	50:// Step50- Door Open Check
	IF iAutorunning AND iInputAreaActive
        AND iHTableAt_0_DegreeFB  AND iTrunionAt_20_DegreeFB
        AND NOT iRawPartPresent1 AND NOT iRawPartPresent2
		AND NOT iRawPartPresent3 AND NOT iRawPartPresent4
        AND NOT iStationDeactivate AND iRollerDoor1Opened
        THEN
		temp:= TRUE;
		oLightcurtainMute:=TRUE;
		
		Step:=60;
	END_IF;
	60:// Step60- Load part check 
	IF iAutorunning AND iInputAreaActive
        AND iHTableAt_0_DegreeFB  AND iTrunionAt_20_DegreeFB
        AND iRawPartPresent1 AND iRawPartPresent2
		AND NOT iRawPartPresent3 AND NOT iRawPartPresent4
        AND NOT iStationDeactivate AND iRollerDoor1Opened
        THEN
		temp:= TRUE;
		oAuthorization:=TRUE;
		Step:=70;
	END_IF;
	70:// Step70- Clamp Close 1-3-5 and RD close
	IF iAutorunning AND iInputAreaActive
        AND iHTableAt_0_DegreeFB  AND iTrunionAt_20_DegreeFB
        AND iRawPartPresent1 AND iRawPartPresent2
		AND NOT iRawPartPresent3 AND NOT iRawPartPresent4
        AND NOT iStationDeactivate AND iRollerDoor1Opened AND iAuthorization
        THEN
		oValve1Work1:= TRUE;
		oValve1Work3:= TRUE;
		oValve1Work5:= TRUE;
		oRollerDoor1Close_OP:=TRUE;
		Step:=80;
	END_IF;
	80:// Step80- Trunion rotates -80 
	IF iAutorunning AND iInputAreaActive
        AND iHTableAt_0_DegreeFB  AND iTrunionAt_20_DegreeFB
        AND iRawPartPresent1 AND iRawPartPresent2
		AND iValve1Work AND iValve3Work AND iValve5Work
		AND NOT iRawPartPresent3 AND NOT iRawPartPresent4
        AND NOT iStationDeactivate AND iRollerDoor1closed 
        THEN
		oTrunionRotate_minus80_Degree_OP:= TRUE;
		Step:=90;
	END_IF;
	90:// Step90- RD1 Open
	IF iAutorunning AND iInputAreaActive
        AND iHTableAt_0_DegreeFB  AND iTrunionAt_minus80_DegreeFB
        AND iRawPartPresent1 AND iRawPartPresent2
		AND iValve1Work AND iValve3Work AND iValve5Work
		AND NOT iRawPartPresent3 AND NOT iRawPartPresent4
        AND NOT iStationDeactivate AND iRollerDoor1closed 
        THEN
		oRollerDoor1Opens_OP:= TRUE;
		oLightcurtainMute:=TRUE;
		Step:=100;
	END_IF;
	100:// Step100- Load part check 3-4
	IF iAutorunning AND iInputAreaActive
        AND iHTableAt_0_DegreeFB  AND iTrunionAt_minus80_DegreeFB
		AND iValve1Work AND iValve3Work AND iValve5Work
        AND iRawPartPresent1 AND iRawPartPresent2
		AND iRawPartPresent3 AND iRawPartPresent4
        AND NOT iStationDeactivate AND iRollerDoor1Opened
        THEN
		temp:= TRUE;
		oAuthorization:=TRUE;
		Step:=110;
	END_IF;
	110:// Step110- Clamp Close 2-4-6 and RD close
	IF iAutorunning AND iInputAreaActive
        AND iHTableAt_0_DegreeFB  AND iTrunionAt_minus80_DegreeFB
		AND iValve1Work AND iValve3Work AND iValve5Work
        AND iRawPartPresent1 AND iRawPartPresent2
		AND iRawPartPresent3 AND iRawPartPresent4
        AND NOT iStationDeactivate AND iRollerDoor1Opened
        THEN
		oValve1Work2:= TRUE;
		oValve1Work4:= TRUE;
		oValve1Work6:= TRUE;
		oRollerDoor1Close_OP:=TRUE;
		Step:=120;
	END_IF;
	120:// Step120- trunion rotates 0 degree
	IF iAutorunning AND iInputAreaActive
        AND iHTableAt_0_DegreeFB  AND iTrunionAt_minus80_DegreeFB
		AND iValve1Work AND iValve3Work AND iValve5Work
		AND iValve2Work AND iValve4Work AND iValve6Work
        AND iRawPartPresent1 AND iRawPartPresent2
		AND iRawPartPresent3 AND iRawPartPresent4
        AND NOT iStationDeactivate AND iRollerDoor1closed
        THEN
		oTrunionRotate_0_Degree_OP:=TRUE;
		Step:=130;
	END_IF;
	130:// Step130- H-Table Rotates 180 Degree
	IF iAutorunning AND iInputAreaActive
        AND iHTableAt_0_DegreeFB  AND iTrunionAt_0_DegreeFB
		AND iValve1Work AND iValve3Work AND iValve5Work
		AND iValve2Work AND iValve4Work AND iValve6Work
        AND iRawPartPresent1 AND iRawPartPresent2
		AND iRawPartPresent3 AND iRawPartPresent4
        AND NOT iStationDeactivate AND iRollerDoor1closed
		AND iWeldRobotAtSafeArea AND iRollerDoor2closed 
		AND NOT iMainJobActive
        THEN
		oHTableStart_180_Degree_OP:=TRUE;
		Step:=140;
	END_IF;
	140:// Step140- Weld Program Move in Robot
	IF iAutorunning AND iworkAreaActive
        AND iHTableAt_180_DegreeFB  AND iTrunionAt_0_DegreeFB
		AND iValve1Work AND iValve3Work AND iValve5Work
		AND iValve2Work AND iValve4Work AND iValve6Work
        AND iRawPartPresent1 AND iRawPartPresent2
		AND iRawPartPresent3 AND iRawPartPresent4
        AND NOT iStationDeactivate 
		AND iWeldRobotAtSafeArea AND iRollerDoor2closed 
        THEN
		oProgramNumber:=1;
		Step:=150;
	END_IF;
	150:// Step150- Robots Welding Start
	IF iAutorunning AND iworkAreaActive
        AND iHTableAt_180_DegreeFB  AND iTrunionAt_0_DegreeFB
		AND iValve1Work AND iValve3Work AND iValve5Work
		AND iValve2Work AND iValve4Work AND iValve6Work
        AND iRawPartPresent1 AND iRawPartPresent2
		AND iRawPartPresent3 AND iRawPartPresent4
        AND NOT iStationDeactivate AND iRollerDoor2closed 
		AND iProgramNumber =1
        THEN
		oWeldStart:=TRUE;
		Step:=160;
	END_IF;
	160:// Step160- Weld Finish and Unclamp part and RD2 open
	IF iAutorunning AND iWorkAreaActive
        AND iHTableAt_180_DegreeFB  AND iTrunionAt_0_DegreeFB
		AND iValve1Work AND iValve3Work AND iValve5Work
		AND iValve2Work AND iValve4Work AND iValve6Work
        AND iRawPartPresent1 AND iRawPartPresent2
		AND iRawPartPresent3 AND iRawPartPresent4
        AND NOT iStationDeactivate AND iRollerDoor2closed 
		AND NOT iMainJobActive AND NOT iWeldon
        THEN
		iValve1Home:=TRUE;
		iValve3Home:=TRUE;
		iValve5Home:=TRUE;
		oRollerDoor2Opens_OP:=TRUE;
		Step:=170;
	END_IF;
	170:// Step170- Fixtre ready and Pick Job request
	IF iAutorunning AND iWorkAreaActive
        AND iHTableAt_180_DegreeFB  AND iTrunionAt_0_DegreeFB
		AND iValve1home AND iValve3home AND iValve5home
		AND iValve2Work AND iValve4Work AND iValve6Work
        AND iRawPartPresent1 AND iRawPartPresent2
		AND iRawPartPresent3 AND iRawPartPresent4
        AND NOT iStationDeactivate AND iRollerDoor2Opened
		AND NOT iMainJobActive AND NOT iWeldon
        THEN
		oFixtureReady:=TRUE;
		oPickJobReady:=TRUE;
		Step:=175;
	END_IF;
	175:// Step175- Gate Open Request request
	IF iAutorunning AND iWorkAreaActive
        AND iHTableAt_180_DegreeFB  AND iTrunionAt_0_DegreeFB
		AND iValve1home AND iValve3home AND iValve5home
		AND iValve2Work AND iValve4Work AND iValve6Work
        AND iRawPartPresent1 AND iRawPartPresent2
		AND iRawPartPresent3 AND iRawPartPresent4
        AND NOT iStationDeactivate AND iRollerDoor2Opened
		AND NOT iMainJobActive AND NOT iWeldon AND iHDLGateopenRequest
        THEN
		oRollerDoor2Opens_OP:=TRUE;
		oPickJobReady:=TRUE;
		Step:=180;
	END_IF;
	180:// Step180- Reduce enble1 request
	IF iAutorunning AND iWorkAreaActive
        AND iHTableAt_180_DegreeFB  AND iTrunionAt_0_DegreeFB
		AND iValve1home AND iValve3home AND iValve5home
		AND iValve2Work AND iValve4Work AND iValve6Work
        AND iRawPartPresent1 AND iRawPartPresent2
		AND iRawPartPresent3 AND iRawPartPresent4
        AND NOT iStationDeactivate AND iRollerDoor2Opened
		AND NOT iMainJobActive AND NOT iWeldon
        THEN
		oReducedEnable1:=TRUE;
		oPickJobReady:=TRUE;
		Step:=190;
	END_IF;
	190:// Step190- Gripper Close request
	IF iAutorunning AND iWorkAreaActive
        AND iHTableAt_180_DegreeFB  AND iTrunionAt_0_DegreeFB
		AND iValve1home AND iValve3home AND iValve5home
		AND iValve2Work AND iValve4Work AND iValve6Work
        AND iRawPartPresent1 AND iRawPartPresent2
		AND iRawPartPresent3 AND iRawPartPresent4
        AND NOT iStationDeactivate AND iRollerDoor2Opened
		AND NOT iMainJobActive AND NOT iWeldon AND iReducedEnable1Finished
        THEN
		oGripperCloseRequest1:=TRUE;
		oPickJobReady:=TRUE;
		Step:=200;
	END_IF;
	200:// Step200- Raise Enable Request
	IF iAutorunning AND iWorkAreaActive
        AND iHTableAt_180_DegreeFB  AND iTrunionAt_0_DegreeFB
		AND iValve1home AND iValve3home AND iValve5home
		AND iValve2Work AND iValve4Work AND iValve6Work
        AND NOT iRawPartPresent1 AND NOT iRawPartPresent2
		AND iRawPartPresent3 AND iRawPartPresent4
        AND NOT iStationDeactivate AND iRollerDoor2Opened
		AND NOT iMainJobActive AND NOT iWeldon AND iHDLGripperClosedFB1
        THEN
		oHDLRaisedEnable1:=TRUE;
		Step:=210;
	END_IF;
	210:// Step210- Trunion -45 degree
	IF iAutorunning AND iWorkAreaActive
        AND iHTableAt_180_DegreeFB  AND iTrunionAt_0_DegreeFB
		AND iValve1home AND iValve3home AND iValve5home
		AND iValve2Work AND iValve4Work AND iValve6Work
        AND NOT iRawPartPresent1 AND NOT iRawPartPresent2
		AND iRawPartPresent3 AND iRawPartPresent4
        AND NOT iStationDeactivate AND iRollerDoor2Opened
		AND NOT iMainJobActive AND NOT iWeldon AND iHDLRaisedEnable1Finished
        THEN
		oTrunionRotate_minus45_Degree_OP:=TRUE;
		Step:=220;
	END_IF;
	220:// Step220- Unclamp 2-4-6
	IF iAutorunning AND iWorkAreaActive
        AND iHTableAt_180_DegreeFB  AND iTrunionAt_0_DegreeFB
		AND iValve2Work AND iValve4Work AND iValve6Work
        AND iRawPartPresent3 AND iRawPartPresent4
        AND NOT iStationDeactivate AND iRollerDoor2Opened
		AND NOT iMainJobActive AND NOT iWeldon AND iHDLRaisedEnable1Finished
        THEN
		oValve1Home2:=TRUE;
		oValve1Home4:=TRUE;
		oValve1Home6:=TRUE;
		oPickJobReady:=TRUE;
		Step:=230;
	END_IF;
	230:// Step230-Reduced enable 2
	IF iAutorunning AND iWorkAreaActive
        AND iHTableAt_180_DegreeFB  AND iTrunionAt_minus45_DegreeFB
		AND iValve2Home AND iValve4Home AND iValve6Home
		AND iRawPartPresent3 AND iRawPartPresent4
        AND NOT iStationDeactivate AND iRollerDoor2Opened
		AND NOT iMainJobActive AND NOT iWeldon 
        THEN
		oReducedEnable2:=TRUE;
		Step:=240;
	END_IF;
	240:// Step240-Gripper 2 Request
	IF iAutorunning AND iWorkAreaActive
        AND iHTableAt_180_DegreeFB  AND iTrunionAt_minus45_DegreeFB
		AND iValve2Home AND iValve4Home AND iValve6Home
		AND iRawPartPresent3 AND iRawPartPresent4
        AND NOT iStationDeactivate AND iRollerDoor2Opened
		AND NOT iMainJobActive AND NOT iWeldon AND iReducedEnable2Finished
        THEN
		oGripperCloseRequest2:=TRUE;
		Step:=250;
	END_IF;
	250:// Step250-Raised enable 2
	IF iAutorunning AND iWorkAreaActive
        AND iHTableAt_180_DegreeFB  AND iTrunionAt_minus45_DegreeFB
        AND NOT iStationDeactivate AND iRollerDoor2Opened
		AND NOT iMainJobActive AND NOT iWeldon AND iHDLGripperClosedFB2
        THEN
		oHDLRaisedEnable2:=TRUE;
		Step:=260;
	END_IF;
	260:// Step260-HDL Robot Outof work Area
	IF iAutorunning AND iWorkAreaActive
        AND iHTableAt_180_DegreeFB  AND iTrunionAt_minus45_DegreeFB
        AND NOT iStationDeactivate AND iRollerDoor2Opened
		AND NOT iMainJobActive AND NOT iWeldon AND iHDLRaisedEnable2Finished
		AND NOT iHDLRobotInArea 
        THEN
		oHDLPickJobACK:=TRUE;
		Step:=270;
	END_IF;
	270:// Step270-RD2 Close and Trunion 0
	IF iAutorunning AND iWorkAreaActive
        AND iHTableAt_180_DegreeFB  AND iTrunionAt_minus45_DegreeFB
        AND NOT iStationDeactivate AND iRollerDoor2Opened
		AND NOT iMainJobActive AND NOT iWeldon AND iHDLRaisedEnable2Finished
		AND NOT iHDLRobotInArea AND iHDLPickJobACK
        THEN
		oHDLPickJobACK:=FALSE;
		oRollerDoor2Close_OP:=TRUE;
		oTrunionRotate_0_Degree_OP:=TRUE;
		Step:=280;
	END_IF;
	280:// Step280-H Table rotates 0 degree
	IF iAutorunning AND iWorkAreaActive
        AND iHTableAt_180_DegreeFB  AND iTrunionAt_0_DegreeFB
        AND NOT iStationDeactivate AND iRollerDoor2closed
		AND NOT iMainJobActive AND NOT iWeldon AND ((iHDLRaisedEnable2Finished
		AND NOT iHDLRobotInArea AND iHDLPickJobACK) OR sJumpWeldSideCycle) 
        THEN
		oHTableStart_0_Degree_OP:=TRUE;
		Step:=290;
	END_IF;
	300:// Step300- all Valve Home Commd
	IF iAutorunning AND iInputAreaActive 
        AND iHTableAt_0_DegreeFB  
        AND NOT iRawPartPresent1 AND NOT iRawPartPresent2
		AND NOT iRawPartPresent3 AND NOT iRawPartPresent4
        AND NOT iStationDeactivate 
        THEN
		oValve1Home1:= TRUE;
		oValve1Home2:= TRUE;
		oValve1Home3:= TRUE;
		oValve1Home4:= TRUE;
		oValve1Home5:= TRUE;
		oValve1Home6:= TRUE;
		Step:=0;
	END_IF;	
END_CASE

END_FUNCTION_BLOCK

// ---- POUs/Library/FB_Trunion.TcPOU
FUNCTION_BLOCK FB_Trunion
VAR_INPUT
    // Commands
    Cmd_20      : BOOL;
    Cmd_0       : BOOL;   // 0 degree
    Cmd_M45     : BOOL;   // -45 degree
    Cmd_M80     : BOOL;   // -80 degree
    Start       : BOOL;
    Stop        : BOOL;
 
    // Feedbacks
    Pos_20      : BOOL;
    Pos_0       : BOOL;   // 0 degree feedback
    Pos_M45     : BOOL;
    Pos_M80     : BOOL;
END_VAR
 
VAR_OUTPUT
    // Motion Outputs
    Move_20     : BOOL;
    Move_0      : BOOL;   // Move to 0 degree
    Move_M45    : BOOL;
    Move_M80    : BOOL;
 
    // Reached Outputs
    Reached_20  : BOOL;
    Reached_0   : BOOL;   // Reached 0 degree
    Reached_M45 : BOOL;
    Reached_M80 : BOOL;
END_VAR
 
VAR
    Target_20   : BOOL;
    Target_0    : BOOL;   // Target 0 degree
    Target_M45  : BOOL;
    Target_M80  : BOOL;
END_VAR

//--------------------------------------------------
// Command Selection Logic
//--------------------------------------------------
IF Start THEN
    Target_20  := Cmd_20;
    Target_0   := Cmd_0;
    Target_M45 := Cmd_M45;
    Target_M80 := Cmd_M80;
END_IF;
 
// Stop resets everything
IF Stop THEN
    Target_20  := FALSE;
    Target_0   := FALSE;
    Target_M45 := FALSE;
    Target_M80 := FALSE;
 
    Move_20  := FALSE;
    Move_0   := FALSE;
    Move_M45 := FALSE;
    Move_M80 := FALSE;
END_IF;
 
//--------------------------------------------------
// Movement Logic
//--------------------------------------------------
 
// Move to 20°
IF Target_20 AND NOT Pos_20 THEN
    Move_20 := TRUE;
ELSE
    Move_20 := FALSE;
END_IF;
 
// Move to 0°
IF Target_0 AND NOT Pos_0 THEN
    Move_0 := TRUE;
ELSE
    Move_0 := FALSE;
END_IF;
 
// Move to -45°
IF Target_M45 AND NOT Pos_M45 THEN
    Move_M45 := TRUE;
ELSE
    Move_M45 := FALSE;
END_IF;
 
// Move to -80°
IF Target_M80 AND NOT Pos_M80 THEN
    Move_M80 := TRUE;
ELSE
    Move_M80 := FALSE;
END_IF;
 
//--------------------------------------------------
// Reached Status
//--------------------------------------------------
Reached_20  := Pos_20;
Reached_0   := Pos_0;
Reached_M45 := Pos_M45;
Reached_M80 := Pos_M80;

END_FUNCTION_BLOCK

// ---- POUs/Library/FB_ModeCall.TcPOU
FUNCTION_BLOCK FB_ModeCall
VAR_INPUT
	iControlOn: BOOL;
	iAutoMode: BOOL;
	iManMode : BOOL;
	iCycleStart: BOOL;
	iCycleStop:BOOL;
	iHome:BOOL;
	iEndOfCycle:BOOL;
	iDryCycle:BOOL;
	iHomeComplete:BOOL;
	iImmediateStop:BOOL;
	iCycleStartDelay:TIME;
	iFaultReset:BOOL;
	
END_VAR
VAR_OUTPUT
	qAutoModeActive:BOOL;
	qManModeActive:BOOL;
	qWaitForStart:BOOL;
	qAutoRunningActive:BOOL;
	qHomeRunningActive:BOOL;
	qCycleStopActive:BOOL;
	qDryCycleActive:BOOL;
	qMsgCSnotStartNoHome:BOOL;
	qManModeAutoRunning:BOOL;
	
	
END_VAR
VAR
	sAlwaysOn:BOOL;
	sAlwaysOff:BOOL;
	sPowerOnReset: BOOL;
	sManModeActive: BOOL;
	sAutoRunningActive: BOOL;
	sAutoModeActive: BOOL;
	sHomeRunningActive: BOOL;
	sWaitForCycleStart: BOOL;
	CycleStartOn: TON;
	sDryCycleActive: BOOL;
	sCycleStopActive: BOOL;
	sMsgCStartandNoHome: BOOL;
	sMsgManModeInAutoRunning: BOOL;
END_VAR

// Always ON Logic
sAlwaysOn := TRUE;
sPowerOnReset := NOT iControlOn;
//Manual_Mode_active:
IF (
    (iManMode ) OR 
    (sManModeActive)
   )
   AND NOT iAutoMode
   AND NOT sAutoRunningActive
   AND NOT sPowerOnReset
THEN
    sManModeActive := TRUE;
ELSE
    sManModeActive := FALSE;
END_IF;
//Auto_Mode_active:
IF (
    (iAutoMode ) OR 
    (sAutoModeActive)
   )
   AND NOT iManMode
   AND NOT sPowerOnReset
   AND NOT sHomeRunningActive
   AND NOT iImmediateStop
THEN
    sAutoModeActive := TRUE;
ELSE
    sAutoModeActive := FALSE;
END_IF;
//Wait_For_Cycle_Start:
IF (
    (sAutoModeActive AND NOT iManMode ) OR 
    (sWaitForCycleStart)
   )
   AND NOT sManModeActive
   AND NOT sPowerOnReset
   AND NOT sAutoRunningActive
   AND NOT iImmediateStop
THEN
    sWaitForCycleStart := TRUE;
ELSE
    sWaitForCycleStart := FALSE;
END_IF;
// Sensor Timeout Timer
CycleStartOn(
    IN := (
            (iCycleStart AND sWaitForCycleStart AND iHomeComplete AND NOT iCycleStop)
                   ),
    PT := iCycleStartDelay
);
//CycleStartOn.Q:= CycleStartOn.Q;
//Dry Cycle Active:
IF (
    (iDryCycle AND NOT sWaitForCycleStart ) OR
    sWaitForCycleStart
   )
   AND  sAutoModeActive
   AND NOT sManModeActive
   AND NOT sPowerOnReset
   AND NOT iImmediateStop
THEN
    sDryCycleActive := TRUE;
ELSE
    sDryCycleActive := FALSE;
END_IF;
//Cycle stop Active:
IF (
    (iCycleStop ) OR
    sCycleStopActive
   )
   AND  sAutoModeActive
   AND NOT sManModeActive
   AND NOT sPowerOnReset
   AND NOT iHomeComplete
THEN
    sCycleStopActive := TRUE;
ELSE
    sCycleStopActive := FALSE;
END_IF;
//AutoCycleStart:
IF (
    (sWaitForCycleStart AND CycleStartOn.Q ) OR
    (sAutoRunningActive AND NOT iImmediateStop)
   )
   AND  sAutoModeActive
   AND NOT sManModeActive
   AND NOT sPowerOnReset
   AND NOT sCycleStopActive
THEN
    sAutoRunningActive := TRUE;
ELSE
    sAutoRunningActive := FALSE;
END_IF;
//HomeCycleStart:
IF (
    (iHome ) OR
    (sHomeRunningActive)
   )
   AND  sManModeActive
   AND NOT sAutoModeActive
   AND NOT sPowerOnReset
   AND NOT iImmediateStop
   AND NOT iHomeComplete
THEN
    sHomeRunningActive := TRUE;
ELSE
    sHomeRunningActive := FALSE;
END_IF;
//AutoCycleNotStart:
IF    iCycleStart
   AND sWaitForCycleStart
   AND NOT sPowerOnReset
   AND NOT iHomeComplete
THEN
    sMsgCStartandNoHome := TRUE;
ELSE
    sMsgCStartandNoHome := FALSE;
END_IF;
//ManModeinAutoRunning:
IF    sAutoRunningActive
   AND sManModeActive
  
THEN
    sMsgManModeInAutoRunning := TRUE;
ELSE
    sMsgManModeInAutoRunning := FALSE;
END_IF;
qManModeActive:=sManModeActive;
qAutoModeActive:=sAutoModeActive;
qWaitForStart:=sWaitForCycleStart;
qDryCycleActive:=sDryCycleActive;
qAutoRunningActive:=sAutoRunningActive;
qHomeRunningActive:=sHomeRunningActive;
qMsgCSnotStartNoHome:=sMsgCStartandNoHome;
qManModeAutoRunning:=sMsgManModeInAutoRunning;

END_FUNCTION_BLOCK

// ---- POUs/Library/FB_CylinderModule.TcPOU
FUNCTION_BLOCK FB_CylinderModule
VAR_INPUT
	iResetModule:BOOL ;
    iResetFaults:BOOL;//Reset Fault CMD
    iEnergizeAtPwrOn:BOOL; // Energize Poweron Input
    iWorkCmd:BOOL ;//Cyl Work Postion CMD
    iHomeCmd:BOOL ;//Cyl Home Postion CMD
    iWorkSen:BOOL ;// Cyl Work Postion Input
    iHomeSen:BOOL ;// Cyl Home Postion Input
    iWorkCleartoMove:BOOL ;// Condition Healthy then 1
    iHomeCleartoMove:BOOL ;// Condition Healthy then 1
    iTimeoutValue:TIME ;// Time Required E.gT#500MS,T#2S
    iWorkSensDebounceVal:TIME ;//Time Required E.gT#500MS,T#2S
    iHomeSensDebounceVal:TIME;
END_VAR
VAR_OUTPUT
	qWorkSol: BOOL; // Cyl Work Position Sol Output
    qHomeSol: BOOL; //Cyl Home Position Sol Output
    qWorkOver: BOOL; // Cyl AT Work Position
    qHomeOver: BOOL; //Cyl AT Home Position
    qErrBothSensorOn: BOOL; //IF both WorkSen AND Homeen inputs are high AT the same TIME.
    qErrHomeInterlock: BOOL; //homeCleartoMove is low AND home command is active.
    qErrHomeSenNotLeft: BOOL; //home position sensor did NOT turn off within defined TIME
    qErrHomeTout: BOOL; //cylinder did NOT reachhome position within definedTIME
    qHomePosLost: BOOL; //home position achieved AND lost its position withoutwork
    qErrWorkInterlock: BOOL; //WorkCleartoMove is low AND work command is active.
    qErrWorkSenNotLeft: BOOL; //work position sensor didnot turn off within definedtime
    qErrWorkTout: BOOL; //cylinder did NOT reachwork position within definedtime
    qWorkPosLost: BOOL; //work position achievedand lost its position withouthome
    qErrPipeSwaped: BOOL; //Pipe OR sensor swapped
    qModError: BOOL; //Module error output
END_VAR
VAR
	sFltRstPls: BOOL; //Stat BIT FOR positive edge OF reset fault input
    sFltEdge: R_TRIG; //Positive edge OF fault reset input
    sWorkPosMemBit: BOOL; //Stat BIT FOR work positionmemory BIT
    sHomePosMemBit: BOOL; //Stat BIT FOR Home positionmemory BIT
    sModError: BOOL; //Stat BIT FOR Module error
    sRodLockTestNegBit: BOOL; //Stat BIT FOR Rod lock test negative pulse
    sModuleResNegBit: BOOL; //Stat BIT FOR reset module negative pulse
    sBrakeSolOffBit: BOOL; //Stat BIT FOR Brake solenoid offbit
    sWorkSensDebTime: TIME; //Stat BIT work sensor debouncetime
    sHomeSensDebTime: TIME; //Stat BIT work sensor debouncetime
    sTimeoutValue: TIME; //Stat BIT FOR TIME out value
    sPosEdge1: BOOL; //Positive Edge
    sPosEdge4: BOOL; //Positive Edge
    sPosEdge3: BOOL; //Positive Edge
    sPosEdge2: BOOL; //Positive Edge
    sPosEdge: BOOL; //Positive Edge
    sRegainHomePos: BOOL; //Regain Home Position
    sRegainWrkPos: BOOL; //Regain Work Position
    sPipeSwapHomePulse: BOOL; //Pipe Swap pulse FOR Home solenoid
	sWorkPosLost: BOOL; // 
    sHomeSol: BOOL; //
    sWorkSol: BOOL; //
    sErrBothSensorOn: BOOL; 
    sErrWorkInterlock: BOOL; 
    sErrHomeInterlock: BOOL; 
    sHomePosLost: BOOL; 
    sErrWorkTout: BOOL; 
    sErrWorkSenNotLeft: BOOL; 
    sErrHomeTOut: BOOL; 
    sErrHomeSenNotLeft: BOOL; 
    sErrPipeSwaped: BOOL; 
    sWorkOver: BOOL; 
    sHomeOver: BOOL; 
    sErrWorkCommon: BOOL; 
    sErrHomeCommon: BOOL; 
	tAlwaysOn: BOOL; //Temporary BIT FOR Always On
    tAlwaysOff: BOOL; //Temporary BIT FOR Always Off

	sDlyWorkSens: TON;
	TON_0: TON;
	sDlyHomeSens: TON;
	sDlyTimeOutt: TON;
END_VAR

// Always ON Logic
tAlwaysOn := TRUE;
 // Rising Edge Detection for Fault Reset

sFltEdge(CLK := iResetFaults);
sFltRstPls := sFltEdge.Q;
 
 
// Work Sensor Debounce Timer
sDlyWorkSens(

    IN := iWorkSen,
    PT := iWorkSensDebounceVal
);
 
// Output after debounce (optional if needed)
//sDlyWorkSens.Q := sDlyWorkSens.Q;
 
 // Home Sensor Debounce Timer
sDlyHomeSens(
    IN := iHomeSen,
    PT := iHomeSensDebounceVal
);
 
// Output after debounce (optional if needed)
//sDlyHomeSens.Q:= sDlyHomeSens.Q;
 // Work Command Logic
IF (
    (iWorkCmd AND iWorkCleartomove) OR 
    (sWorkSol AND sDlyWorkSens.Q AND NOT sDlyHomeSens.Q)
   )
   AND NOT iHomeCmd
   AND NOT sHomeSol
   AND NOT iResetModule
   AND NOT sModError
THEN
    sWorkSol := TRUE;
ELSE
    sWorkSol := FALSE;
END_IF;
// Home Command Logic
IF (
    (iHomeCmd AND iHomeCleartomove) OR 
    (sHomeSol AND sDlyHomeSens.Q AND NOT sDlyWorkSens.Q)
   )
   AND NOT iWorkCmd
   AND NOT sWorkSol
   AND NOT iResetModule
   AND NOT sModError
THEN
    sHomeSol := TRUE;
ELSE
    sHomeSol := FALSE;
END_IF;
// Both Sensors ON Error
IF (sDlyWorkSens.Q AND sDlyHomeSens.Q) THEN
    sErrBothSensoron := TRUE;
ELSIF (sFltRstPls) THEN
    sErrBothSensoron := FALSE;
END_IF;
// Work Interlock Error
IF (iWorkCmd AND NOT iWorkCleartomove) THEN
    sErrWorkInterlock := TRUE;
ELSIF (sFltRstPls) THEN
    sErrWorkInterlock := FALSE;
END_IF;
// Home Interlock Error
IF (iHomeCmd AND NOT iHomeCleartomove) THEN
    sErrHomeInterlock := TRUE;
 
ELSIF (sFltRstPls) THEN
    sErrHomeInterlock := FALSE;
END_IF;
// Sensor Timeout Timer
sDlyTimeOutt(
    IN := (
            (sWorkSol AND NOT sDlyWorkSens.Q AND NOT sErrWorkTout)
         OR (sHomeSol AND NOT sDlyHomeSens.Q AND NOT sErrHomeTout)
          ),
    PT := iTimeoutValue
);
//sDlyTimeOutt.Q:= sDlyTimeOutt.Q;
//Work Timeout Error
IF (
   (sWorkSol AND NOT sDlyWorkSens.Q AND sDlyTimeOutt.Q) OR
   (sErrWorkTout AND NOT sFltRstPls)
   )
   THEN
   sErrWorkTout := TRUE;
   ELSE
	   sErrWorkTout := FALSE;
   END_IF;
   
   //Home Timeout Error
IF (
   (sHomeSol AND NOT sDlyHomeSens.Q AND sDlyTimeOutt.Q) OR
   (sErrHomeTOut AND NOT sFltRstPls)
   )
   THEN
   sErrHomeTOut := TRUE;
   ELSE
	   sErrHomeTOut := FALSE;
   END_IF;
//mode errors   
   IF (
   (sErrBothSensoron OR sErrWorkinterlock OR sErrHomeinterlock OR sErrWorkSenNotleft OR sErrWorkTout OR sErrHomeSennotleft OR sErrHomeTOut OR sErrPipeSwaped  OR sHomePosLost OR sWorkPosLost)
   )
   THEN
   sModError := TRUE;
   ELSE
	   sModError := FALSE;
   END_IF;
	
//Workover
IF (
   (sDlyWorkSens.Q AND NOT sDlyHomeSens.Q AND NOT sModError AND NOT iResetModule AND NOT sHomePosLost ) 
   )
   THEN
   sWorkOver := TRUE;
   ELSE
	   sWorkOver := FALSE;
   END_IF; 
//Homeover
IF (
   (sDlyHomeSens.Q AND NOT sDlyWorkSens.Q AND NOT sModError AND NOT iResetModule AND NOT sWorkPosLost ) 
   )
   THEN
   sHomeOver := TRUE;
   ELSE
	   sHomeOver := FALSE;
   END_IF;   
   
   qHomeSol := sHomeSol;
   qWorkSol := sWorkSol;
   qErrBothSensoron := sErrBothSensoron;
   qErrWorkinterlock := sErrWorkinterlock;
   qErrHomeinterlock := sErrHomeinterlock;
   qErrWorkSenNotleft := sErrWorkSenNotleft;
   qErrHomeSennotleft := sErrHomeSennotleft;
   qErrWorkTout := sErrWorkTout;
   qErrHomeTout := sErrHomeTOut;
   qErrPipeSwaped := sErrPipeSwaped;
   qWorkPosLost := sWorkPosLost;
   qHomePosLost := sHomePosLost;
   qModError := sModError;
   qWorkOver := sWorkOver;
   qHomeOver := sHomeOver;

END_FUNCTION_BLOCK

// ---- POUs/Library/FB_Roller_Door.TcPOU
FUNCTION_BLOCK FB_Roller_Door
VAR_INPUT
	// Inputs
    OpenBtn   : BOOL;
    CloseBtn  : BOOL;
    StopBtn   : BOOL;
    LS_Open   : BOOL;
    LS_Close  : BOOL;
END_VAR
VAR_OUTPUT
	// Outputs
    Motor_Up   : BOOL;
    Motor_Down : BOOL;
	Motor_Up_Reached:BOOL;
	Motor_Down_Reached:BOOL;
END_VAR
VAR
	// Internal states (latch)
    Opening : BOOL := FALSE;
    Closing : BOOL := FALSE;
END_VAR

// OPEN command
IF OpenBtn AND NOT LS_Open THEN
    Opening := TRUE;
    Closing := FALSE;
END_IF;
  
// CLOSE command
IF CloseBtn AND NOT LS_Close THEN
    Closing := TRUE;
    Opening := FALSE;
END_IF;
  
// STOP command
IF StopBtn THEN
    Opening := FALSE;
    Closing := FALSE;
END_IF;
  
// Limit conditions (auto stop)
IF LS_Open THEN
    Opening := FALSE;
END_IF;
 
IF LS_Close THEN
    Closing := FALSE;
END_IF;

// --- Outputs ---
Motor_Up := Opening AND NOT LS_Open;
Motor_Down := Closing AND NOT LS_Close;


Motor_Up_Reached := LS_Open;
Motor_Down_Reached := LS_Close;

END_FUNCTION_BLOCK

// ---- POUs/Library/FB_TurnTable_0_180.TcPOU
FUNCTION_BLOCK FB_TurnTable_0_180
VAR_INPUT
	// Inputs
    Start_0     : BOOL;
    Start_180   : BOOL;
    LS_0        : BOOL;
    LS_180      : BOOL;
    StopBtn     : BOOL;

END_VAR
VAR_OUTPUT
	// Outputs
    Motor_CW    : BOOL;
    Motor_CCW   : BOOL;
    Reached_180 : BOOL;
    Reached_0   : BOOL;
END_VAR
VAR
	// Internal states
    Move_0      : BOOL := FALSE;
    Move_180    : BOOL := FALSE;
END_VAR

// =========================
// COMMAND LOGIC
// =========================
// Move to 0°
IF Start_0 AND NOT LS_0 THEN
    Move_0 := TRUE;
    Move_180 := FALSE;
END_IF;

// Move to 180°
IF Start_180 AND NOT LS_180 THEN
    Move_180 := TRUE;
    Move_0 := FALSE;
END_IF;

// =========================
// STOP LOGIC
// =========================
IF StopBtn THEN
    Move_0 := FALSE;
    Move_180 := FALSE;
END_IF;

// =========================
// LIMIT SWITCH STOP
// =========================
IF LS_0 THEN
    Move_0 := FALSE;
END_IF;
IF LS_180 THEN
    Move_180 := FALSE;
END_IF;

// =========================
// SAFETY: BOTH LIMIT ACTIVE
// =========================
IF LS_0 AND LS_180 THEN
    Move_0 := FALSE;
    Move_180 := FALSE;
END_IF;

// =========================
// OUTPUT LOGIC
// =========================
Motor_CCW := Move_0;     // Move toward 0°
Motor_CW  := Move_180;   // Move toward 180°

// =========================
// INTERLOCK (VERY IMPORTANT)
// =========================
IF Motor_CW THEN
    Motor_CCW := FALSE;
END_IF;
IF Motor_CCW THEN
    Motor_CW := FALSE;
END_IF;

// =========================
// POSITION REACHED SIGNALS
// =========================
Reached_0   := LS_0 AND NOT Move_0;
Reached_180 := LS_180 AND NOT Move_180;
 
// =========================
// COMMAND LOGIC
// =========================
// Move to 0°

IF Start_0 AND NOT LS_0 THEN
    Move_0 := TRUE;
    Move_180 := FALSE;
END_IF;
// Move to 180°
IF Start_180 AND NOT LS_180 THEN
    Move_180 := TRUE;
    Move_0 := FALSE;
END_IF;

// =========================
// STOP LOGIC
// =========================
IF StopBtn THEN
    Move_0 := FALSE;
    Move_180 := FALSE;
END_IF;

// =========================
// LIMIT SWITCH STOP
// =========================
IF LS_0 THEN
    Move_0 := FALSE;
END_IF;
IF LS_180 THEN
    Move_180 := FALSE;
END_IF;

// =========================
// SAFETY: BOTH LIMIT ACTIVE
// =========================
IF LS_0 AND LS_180 THEN
    Move_0 := FALSE;
    Move_180 := FALSE;
END_IF;

// =========================
// OUTPUT LOGIC
// =========================
Motor_CCW := Move_0;     // Move toward 0°
Motor_CW  := Move_180;   // Move toward 180°

// =========================
// INTERLOCK (VERY IMPORTANT)
// =========================
IF Motor_CW THEN
    Motor_CCW := FALSE;
END_IF;
IF Motor_CCW THEN
    Motor_CW := FALSE;
END_IF;

// =========================
// POSITION REACHED SIGNALS
// =========================
Reached_0   := LS_0 AND NOT Move_0;
Reached_180 := LS_180 AND NOT Move_180;

END_FUNCTION_BLOCK

// ---- POUs/Fixt2_Seq_Call.TcPOU
PROGRAM Fixt2_Seq_Call
VAR
	Clamp_1: FB_CylinderModule;
	Clamp_2: FB_CylinderModule;
	Clamp_3: FB_CylinderModule;
	Clamp_4: FB_CylinderModule;
	Clamp_5: FB_CylinderModule;
	Clamp_6: FB_CylinderModule;
	sAlwaysoff: BOOL;
	FB_AutoSeq_0: FB_AutoSeq;
	alwayson:BOOL;
	partmonitor:FB_PartMonitoring_fixt2;
	trunion:FB_Trunion;
END_VAR
VAR // added by the converter: edge detectors and wires of the graphical bodies
    _w1, _w2, _w3, _w4, _w5, _w6 : BOOL;
END_VAR

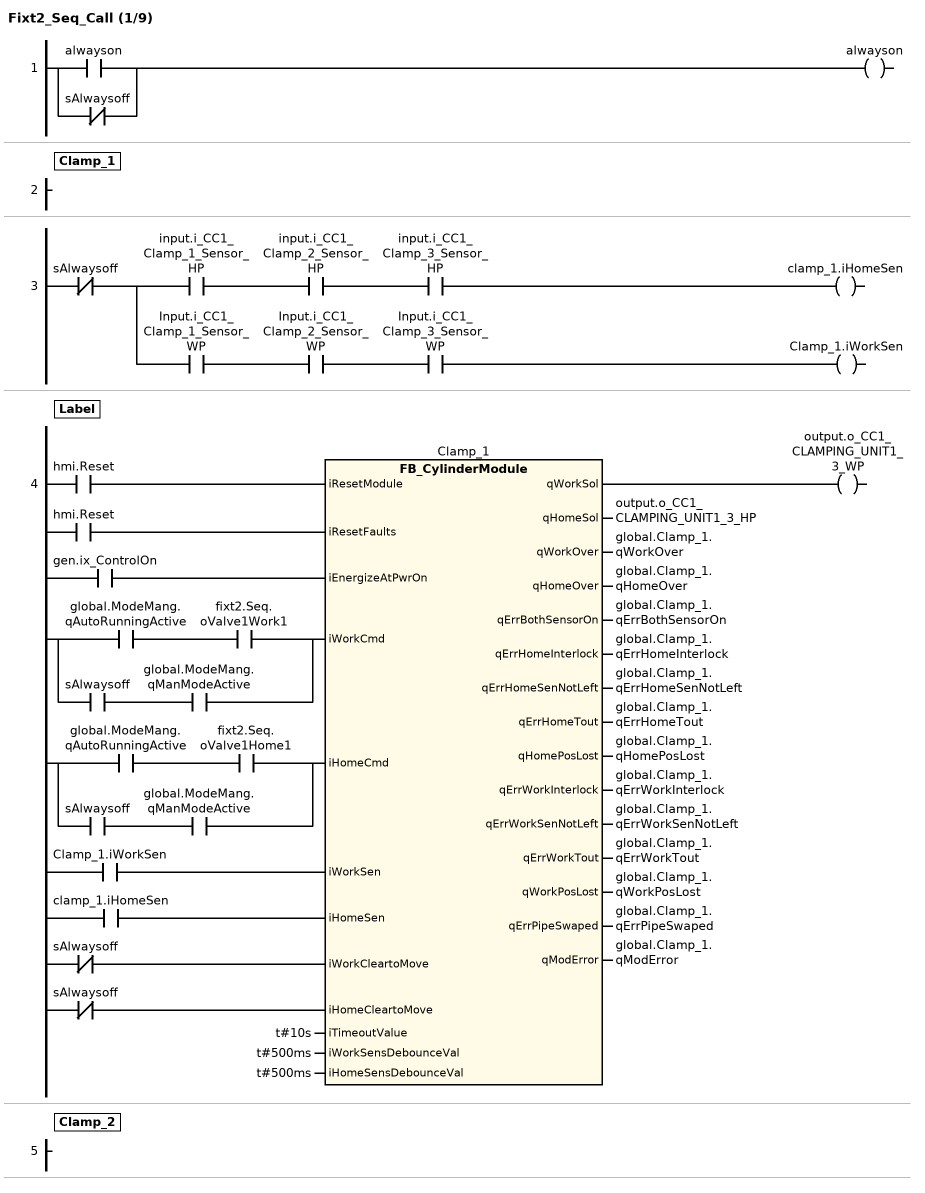
// NETWORK 1
alwayson := alwayson OR NOT sAlwaysoff;

// NETWORK 2
Clamp_1: ;

// NETWORK 3
_w1 := NOT sAlwaysoff;
clamp_1.iHomeSen := _w1 AND input.i_CC1_Clamp_1_Sensor_HP AND input.i_CC1_Clamp_2_Sensor_HP AND input.i_CC1_Clamp_3_Sensor_HP;
Clamp_1.iWorkSen := _w1 AND Input.i_CC1_Clamp_1_Sensor_WP AND Input.i_CC1_Clamp_2_Sensor_WP AND Input.i_CC1_Clamp_3_Sensor_WP;

// NETWORK 4
Label:
Clamp_1(
    iResetModule := hmi.Reset,
    iResetFaults := hmi.Reset,
    iEnergizeAtPwrOn := gen.ix_ControlOn,
    iWorkCmd := global.ModeMang.qAutoRunningActive AND fixt2.Seq.oValve1Work1 OR sAlwaysoff AND global.ModeMang.qManModeActive,
    iHomeCmd := global.ModeMang.qAutoRunningActive AND fixt2.Seq.oValve1Home1 OR sAlwaysoff AND global.ModeMang.qManModeActive,
    iWorkSen := Clamp_1.iWorkSen,
    iHomeSen := clamp_1.iHomeSen,
    iWorkCleartoMove := NOT sAlwaysoff,
    iHomeCleartoMove := NOT sAlwaysoff,
    iTimeoutValue := t#10s,
    iWorkSensDebounceVal := t#500ms,
    iHomeSensDebounceVal := t#500ms,
    qHomeSol => output.o_CC1_CLAMPING_UNIT1_3_HP,
    qWorkOver => global.Clamp_1.qWorkOver,
    qHomeOver => global.Clamp_1.qHomeOver,
    qErrBothSensorOn => global.Clamp_1.qErrBothSensorOn,
    qErrHomeInterlock => global.Clamp_1.qErrHomeInterlock,
    qErrHomeSenNotLeft => global.Clamp_1.qErrHomeSenNotLeft,
    qErrHomeTout => global.Clamp_1.qErrHomeTout,
    qHomePosLost => global.Clamp_1.qHomePosLost,
    qErrWorkInterlock => global.Clamp_1.qErrWorkInterlock,
    qErrWorkSenNotLeft => global.Clamp_1.qErrWorkSenNotLeft,
    qErrWorkTout => global.Clamp_1.qErrWorkTout,
    qWorkPosLost => global.Clamp_1.qWorkPosLost,
    qErrPipeSwaped => global.Clamp_1.qErrPipeSwaped,
    qModError => global.Clamp_1.qModError); // FB_CylinderModule
output.o_CC1_CLAMPING_UNIT1_3_WP := Clamp_1.qWorkSol;

// NETWORK 5
Clamp_2: ;

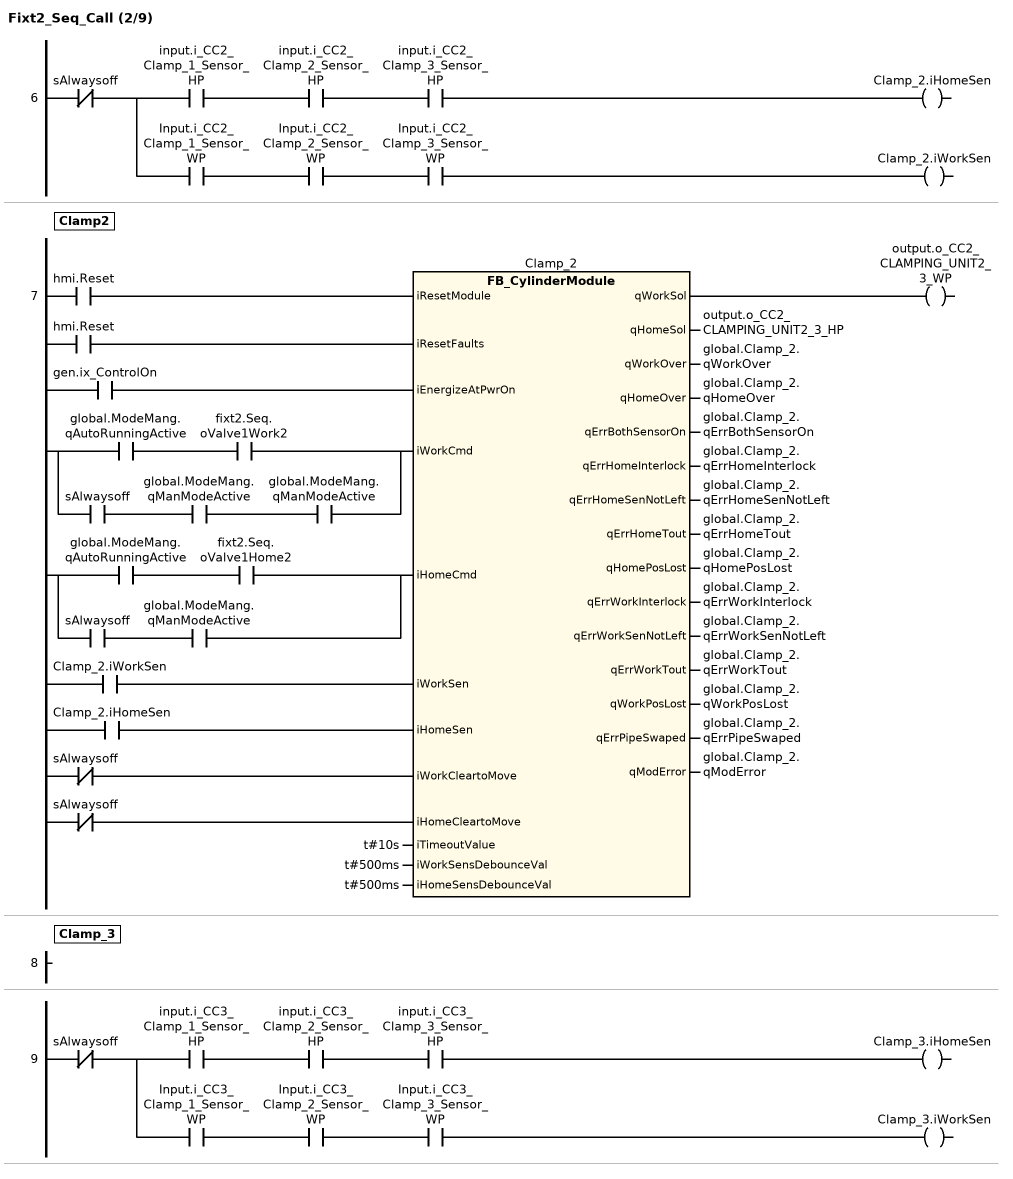
// NETWORK 6
_w2 := NOT sAlwaysoff;
Clamp_2.iHomeSen := _w2 AND input.i_CC2_Clamp_1_Sensor_HP AND input.i_CC2_Clamp_2_Sensor_HP AND input.i_CC2_Clamp_3_Sensor_HP;
Clamp_2.iWorkSen := _w2 AND Input.i_CC2_Clamp_1_Sensor_WP AND Input.i_CC2_Clamp_2_Sensor_WP AND Input.i_CC2_Clamp_3_Sensor_WP;

// NETWORK 7
Clamp2:
Clamp_2(
    iResetModule := hmi.Reset,
    iResetFaults := hmi.Reset,
    iEnergizeAtPwrOn := gen.ix_ControlOn,
    iWorkCmd := global.ModeMang.qAutoRunningActive AND fixt2.Seq.oValve1Work2 OR sAlwaysoff AND global.ModeMang.qManModeActive AND global.ModeMang.qManModeActive,
    iHomeCmd := global.ModeMang.qAutoRunningActive AND fixt2.Seq.oValve1Home2 OR sAlwaysoff AND global.ModeMang.qManModeActive,
    iWorkSen := Clamp_2.iWorkSen,
    iHomeSen := Clamp_2.iHomeSen,
    iWorkCleartoMove := NOT sAlwaysoff,
    iHomeCleartoMove := NOT sAlwaysoff,
    iTimeoutValue := t#10s,
    iWorkSensDebounceVal := t#500ms,
    iHomeSensDebounceVal := t#500ms,
    qHomeSol => output.o_CC2_CLAMPING_UNIT2_3_HP,
    qWorkOver => global.Clamp_2.qWorkOver,
    qHomeOver => global.Clamp_2.qHomeOver,
    qErrBothSensorOn => global.Clamp_2.qErrBothSensorOn,
    qErrHomeInterlock => global.Clamp_2.qErrHomeInterlock,
    qErrHomeSenNotLeft => global.Clamp_2.qErrHomeSenNotLeft,
    qErrHomeTout => global.Clamp_2.qErrHomeTout,
    qHomePosLost => global.Clamp_2.qHomePosLost,
    qErrWorkInterlock => global.Clamp_2.qErrWorkInterlock,
    qErrWorkSenNotLeft => global.Clamp_2.qErrWorkSenNotLeft,
    qErrWorkTout => global.Clamp_2.qErrWorkTout,
    qWorkPosLost => global.Clamp_2.qWorkPosLost,
    qErrPipeSwaped => global.Clamp_2.qErrPipeSwaped,
    qModError => global.Clamp_2.qModError); // FB_CylinderModule
output.o_CC2_CLAMPING_UNIT2_3_WP := Clamp_2.qWorkSol;

// NETWORK 8
Clamp_3: ;

// NETWORK 9
_w3 := NOT sAlwaysoff;
Clamp_3.iHomeSen := _w3 AND input.i_CC3_Clamp_1_Sensor_HP AND input.i_CC3_Clamp_2_Sensor_HP AND input.i_CC3_Clamp_3_Sensor_HP;
Clamp_3.iWorkSen := _w3 AND Input.i_CC3_Clamp_1_Sensor_WP AND Input.i_CC3_Clamp_2_Sensor_WP AND Input.i_CC3_Clamp_3_Sensor_WP;

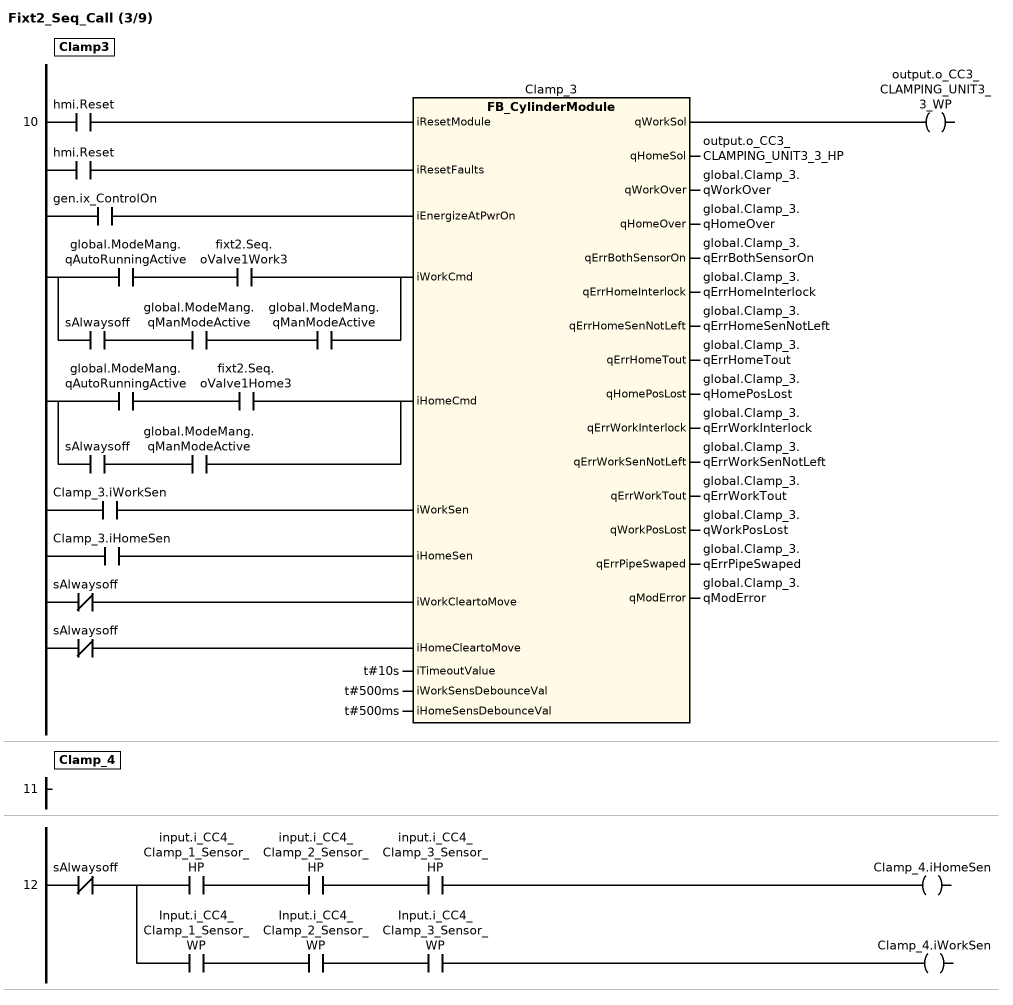
// NETWORK 10
Clamp3:
Clamp_3(
    iResetModule := hmi.Reset,
    iResetFaults := hmi.Reset,
    iEnergizeAtPwrOn := gen.ix_ControlOn,
    iWorkCmd := global.ModeMang.qAutoRunningActive AND fixt2.Seq.oValve1Work3 OR sAlwaysoff AND global.ModeMang.qManModeActive AND global.ModeMang.qManModeActive,
    iHomeCmd := global.ModeMang.qAutoRunningActive AND fixt2.Seq.oValve1Home3 OR sAlwaysoff AND global.ModeMang.qManModeActive,
    iWorkSen := Clamp_3.iWorkSen,
    iHomeSen := Clamp_3.iHomeSen,
    iWorkCleartoMove := NOT sAlwaysoff,
    iHomeCleartoMove := NOT sAlwaysoff,
    iTimeoutValue := t#10s,
    iWorkSensDebounceVal := t#500ms,
    iHomeSensDebounceVal := t#500ms,
    qHomeSol => output.o_CC3_CLAMPING_UNIT3_3_HP,
    qWorkOver => global.Clamp_3.qWorkOver,
    qHomeOver => global.Clamp_3.qHomeOver,
    qErrBothSensorOn => global.Clamp_3.qErrBothSensorOn,
    qErrHomeInterlock => global.Clamp_3.qErrHomeInterlock,
    qErrHomeSenNotLeft => global.Clamp_3.qErrHomeSenNotLeft,
    qErrHomeTout => global.Clamp_3.qErrHomeTout,
    qHomePosLost => global.Clamp_3.qHomePosLost,
    qErrWorkInterlock => global.Clamp_3.qErrWorkInterlock,
    qErrWorkSenNotLeft => global.Clamp_3.qErrWorkSenNotLeft,
    qErrWorkTout => global.Clamp_3.qErrWorkTout,
    qWorkPosLost => global.Clamp_3.qWorkPosLost,
    qErrPipeSwaped => global.Clamp_3.qErrPipeSwaped,
    qModError => global.Clamp_3.qModError); // FB_CylinderModule
output.o_CC3_CLAMPING_UNIT3_3_WP := Clamp_3.qWorkSol;

// NETWORK 11
Clamp_4: ;

// NETWORK 12
_w4 := NOT sAlwaysoff;
Clamp_4.iHomeSen := _w4 AND input.i_CC4_Clamp_1_Sensor_HP AND input.i_CC4_Clamp_2_Sensor_HP AND input.i_CC4_Clamp_3_Sensor_HP;
Clamp_4.iWorkSen := _w4 AND Input.i_CC4_Clamp_1_Sensor_WP AND Input.i_CC4_Clamp_2_Sensor_WP AND Input.i_CC4_Clamp_3_Sensor_WP;

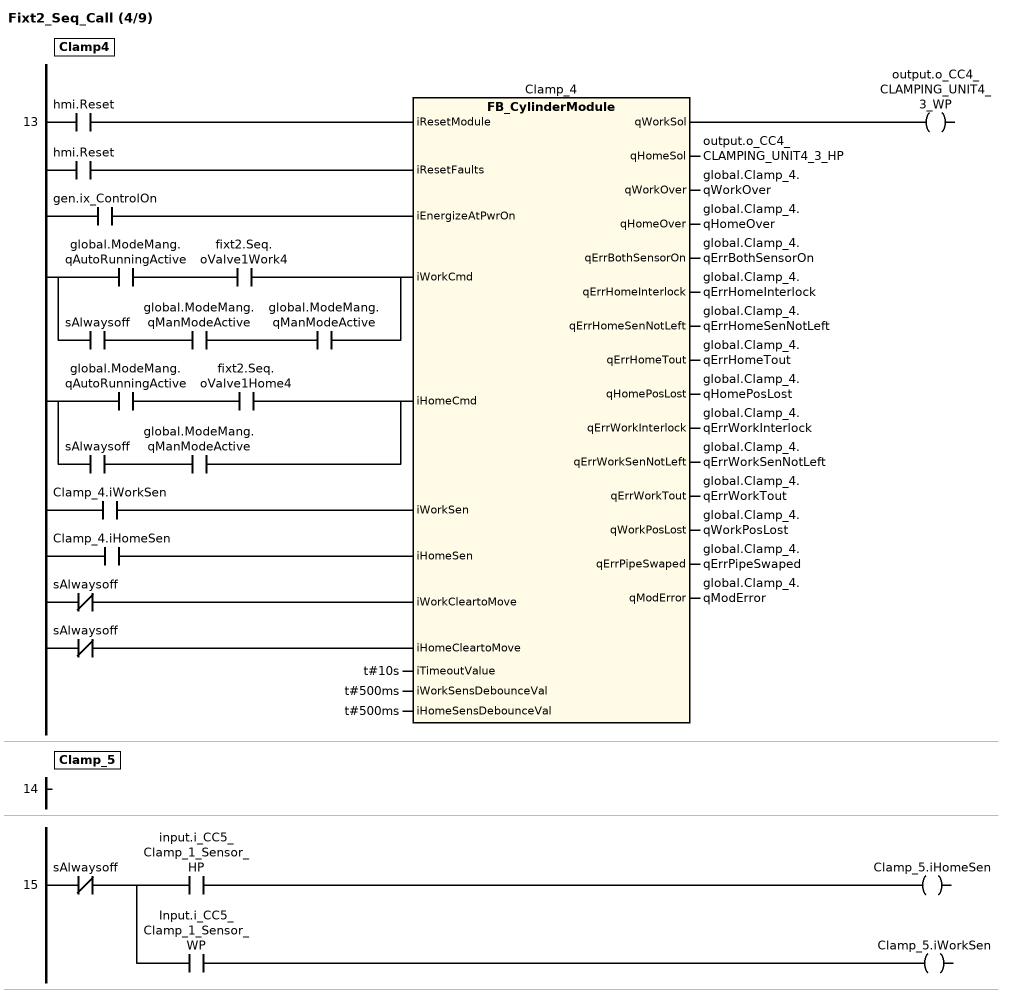
// NETWORK 13
Clamp4:
Clamp_4(
    iResetModule := hmi.Reset,
    iResetFaults := hmi.Reset,
    iEnergizeAtPwrOn := gen.ix_ControlOn,
    iWorkCmd := global.ModeMang.qAutoRunningActive AND fixt2.Seq.oValve1Work4 OR sAlwaysoff AND global.ModeMang.qManModeActive AND global.ModeMang.qManModeActive,
    iHomeCmd := global.ModeMang.qAutoRunningActive AND fixt2.Seq.oValve1Home4 OR sAlwaysoff AND global.ModeMang.qManModeActive,
    iWorkSen := Clamp_4.iWorkSen,
    iHomeSen := Clamp_4.iHomeSen,
    iWorkCleartoMove := NOT sAlwaysoff,
    iHomeCleartoMove := NOT sAlwaysoff,
    iTimeoutValue := t#10s,
    iWorkSensDebounceVal := t#500ms,
    iHomeSensDebounceVal := t#500ms,
    qHomeSol => output.o_CC4_CLAMPING_UNIT4_3_HP,
    qWorkOver => global.Clamp_4.qWorkOver,
    qHomeOver => global.Clamp_4.qHomeOver,
    qErrBothSensorOn => global.Clamp_4.qErrBothSensorOn,
    qErrHomeInterlock => global.Clamp_4.qErrHomeInterlock,
    qErrHomeSenNotLeft => global.Clamp_4.qErrHomeSenNotLeft,
    qErrHomeTout => global.Clamp_4.qErrHomeTout,
    qHomePosLost => global.Clamp_4.qHomePosLost,
    qErrWorkInterlock => global.Clamp_4.qErrWorkInterlock,
    qErrWorkSenNotLeft => global.Clamp_4.qErrWorkSenNotLeft,
    qErrWorkTout => global.Clamp_4.qErrWorkTout,
    qWorkPosLost => global.Clamp_4.qWorkPosLost,
    qErrPipeSwaped => global.Clamp_4.qErrPipeSwaped,
    qModError => global.Clamp_4.qModError); // FB_CylinderModule
output.o_CC4_CLAMPING_UNIT4_3_WP := Clamp_4.qWorkSol;

// NETWORK 14
Clamp_5: ;

// NETWORK 15
_w5 := NOT sAlwaysoff;
Clamp_5.iHomeSen := _w5 AND input.i_CC5_Clamp_1_Sensor_HP;
Clamp_5.iWorkSen := _w5 AND Input.i_CC5_Clamp_1_Sensor_WP;

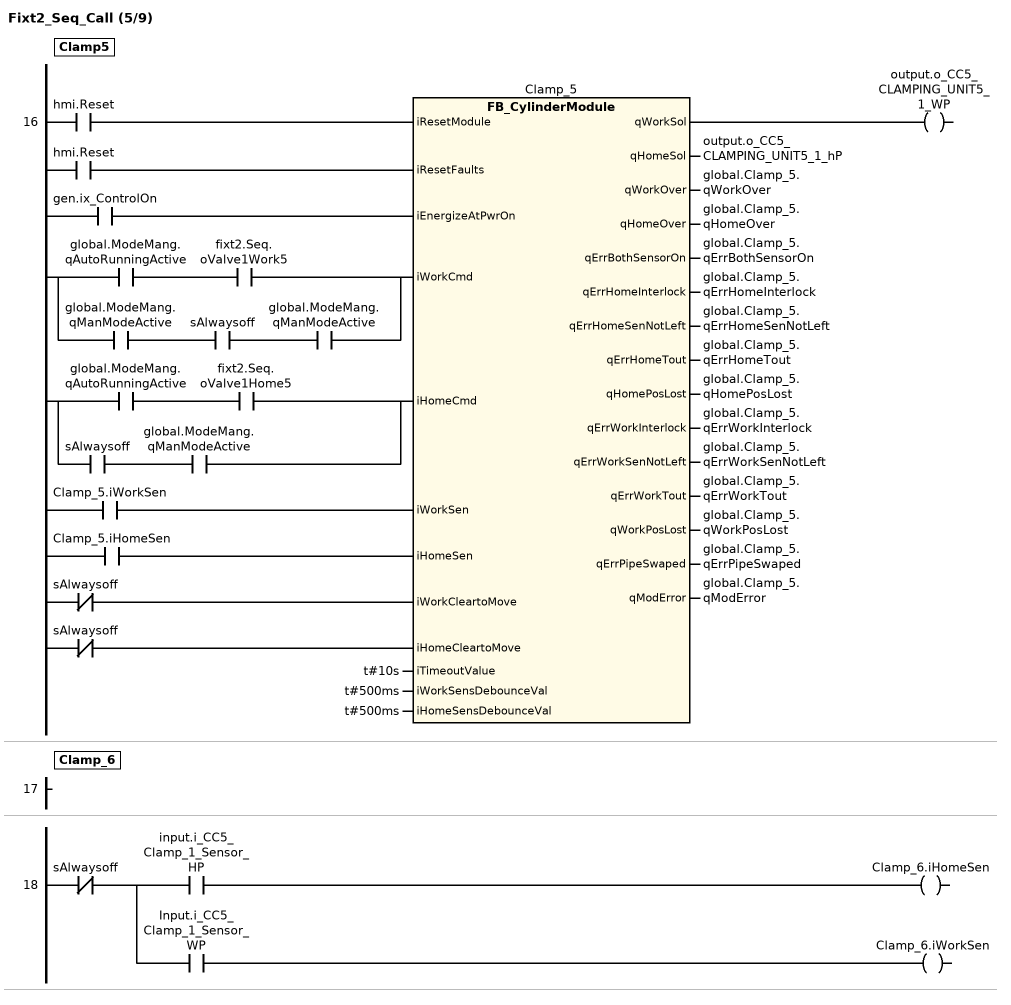
// NETWORK 16
Clamp5:
Clamp_5(
    iResetModule := hmi.Reset,
    iResetFaults := hmi.Reset,
    iEnergizeAtPwrOn := gen.ix_ControlOn,
    iWorkCmd := global.ModeMang.qAutoRunningActive AND fixt2.Seq.oValve1Work5 OR global.ModeMang.qManModeActive AND sAlwaysoff AND global.ModeMang.qManModeActive,
    iHomeCmd := global.ModeMang.qAutoRunningActive AND fixt2.Seq.oValve1Home5 OR sAlwaysoff AND global.ModeMang.qManModeActive,
    iWorkSen := Clamp_5.iWorkSen,
    iHomeSen := Clamp_5.iHomeSen,
    iWorkCleartoMove := NOT sAlwaysoff,
    iHomeCleartoMove := NOT sAlwaysoff,
    iTimeoutValue := t#10s,
    iWorkSensDebounceVal := t#500ms,
    iHomeSensDebounceVal := t#500ms,
    qHomeSol => output.o_CC5_CLAMPING_UNIT5_1_hP,
    qWorkOver => global.Clamp_5.qWorkOver,
    qHomeOver => global.Clamp_5.qHomeOver,
    qErrBothSensorOn => global.Clamp_5.qErrBothSensorOn,
    qErrHomeInterlock => global.Clamp_5.qErrHomeInterlock,
    qErrHomeSenNotLeft => global.Clamp_5.qErrHomeSenNotLeft,
    qErrHomeTout => global.Clamp_5.qErrHomeTout,
    qHomePosLost => global.Clamp_5.qHomePosLost,
    qErrWorkInterlock => global.Clamp_5.qErrWorkInterlock,
    qErrWorkSenNotLeft => global.Clamp_5.qErrWorkSenNotLeft,
    qErrWorkTout => global.Clamp_5.qErrWorkTout,
    qWorkPosLost => global.Clamp_5.qWorkPosLost,
    qErrPipeSwaped => global.Clamp_5.qErrPipeSwaped,
    qModError => global.Clamp_5.qModError); // FB_CylinderModule
output.o_CC5_CLAMPING_UNIT5_1_WP := Clamp_5.qWorkSol;

// NETWORK 17
Clamp_6: ;

// NETWORK 18
_w6 := NOT sAlwaysoff;
Clamp_6.iHomeSen := _w6 AND input.i_CC5_Clamp_1_Sensor_HP;
Clamp_6.iWorkSen := _w6 AND Input.i_CC5_Clamp_1_Sensor_WP;

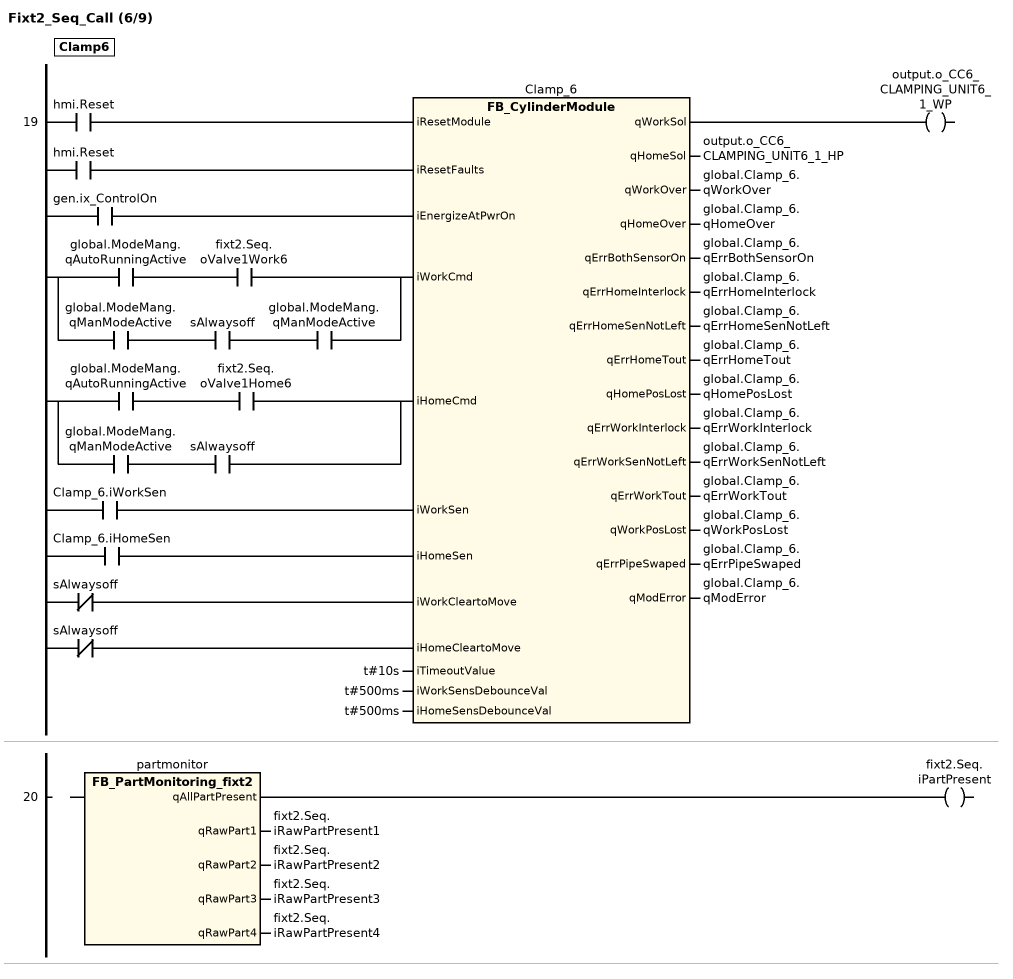
// NETWORK 19
Clamp6:
Clamp_6(
    iResetModule := hmi.Reset,
    iResetFaults := hmi.Reset,
    iEnergizeAtPwrOn := gen.ix_ControlOn,
    iWorkCmd := global.ModeMang.qAutoRunningActive AND fixt2.Seq.oValve1Work6 OR global.ModeMang.qManModeActive AND sAlwaysoff AND global.ModeMang.qManModeActive,
    iHomeCmd := global.ModeMang.qAutoRunningActive AND fixt2.Seq.oValve1Home6 OR global.ModeMang.qManModeActive AND sAlwaysoff,
    iWorkSen := Clamp_6.iWorkSen,
    iHomeSen := Clamp_6.iHomeSen,
    iWorkCleartoMove := NOT sAlwaysoff,
    iHomeCleartoMove := NOT sAlwaysoff,
    iTimeoutValue := t#10s,
    iWorkSensDebounceVal := t#500ms,
    iHomeSensDebounceVal := t#500ms,
    qHomeSol => output.o_CC6_CLAMPING_UNIT6_1_HP,
    qWorkOver => global.Clamp_6.qWorkOver,
    qHomeOver => global.Clamp_6.qHomeOver,
    qErrBothSensorOn => global.Clamp_6.qErrBothSensorOn,
    qErrHomeInterlock => global.Clamp_6.qErrHomeInterlock,
    qErrHomeSenNotLeft => global.Clamp_6.qErrHomeSenNotLeft,
    qErrHomeTout => global.Clamp_6.qErrHomeTout,
    qHomePosLost => global.Clamp_6.qHomePosLost,
    qErrWorkInterlock => global.Clamp_6.qErrWorkInterlock,
    qErrWorkSenNotLeft => global.Clamp_6.qErrWorkSenNotLeft,
    qErrWorkTout => global.Clamp_6.qErrWorkTout,
    qWorkPosLost => global.Clamp_6.qWorkPosLost,
    qErrPipeSwaped => global.Clamp_6.qErrPipeSwaped,
    qModError => global.Clamp_6.qModError); // FB_CylinderModule
output.o_CC6_CLAMPING_UNIT6_1_WP := Clamp_6.qWorkSol;

// NETWORK 20
partmonitor(
    qRawPart1 => fixt2.Seq.iRawPartPresent1,
    qRawPart2 => fixt2.Seq.iRawPartPresent2,
    qRawPart3 => fixt2.Seq.iRawPartPresent3,
    qRawPart4 => fixt2.Seq.iRawPartPresent4); // FB_PartMonitoring_fixt2
fixt2.Seq.iPartPresent := partmonitor.qAllPartPresent;

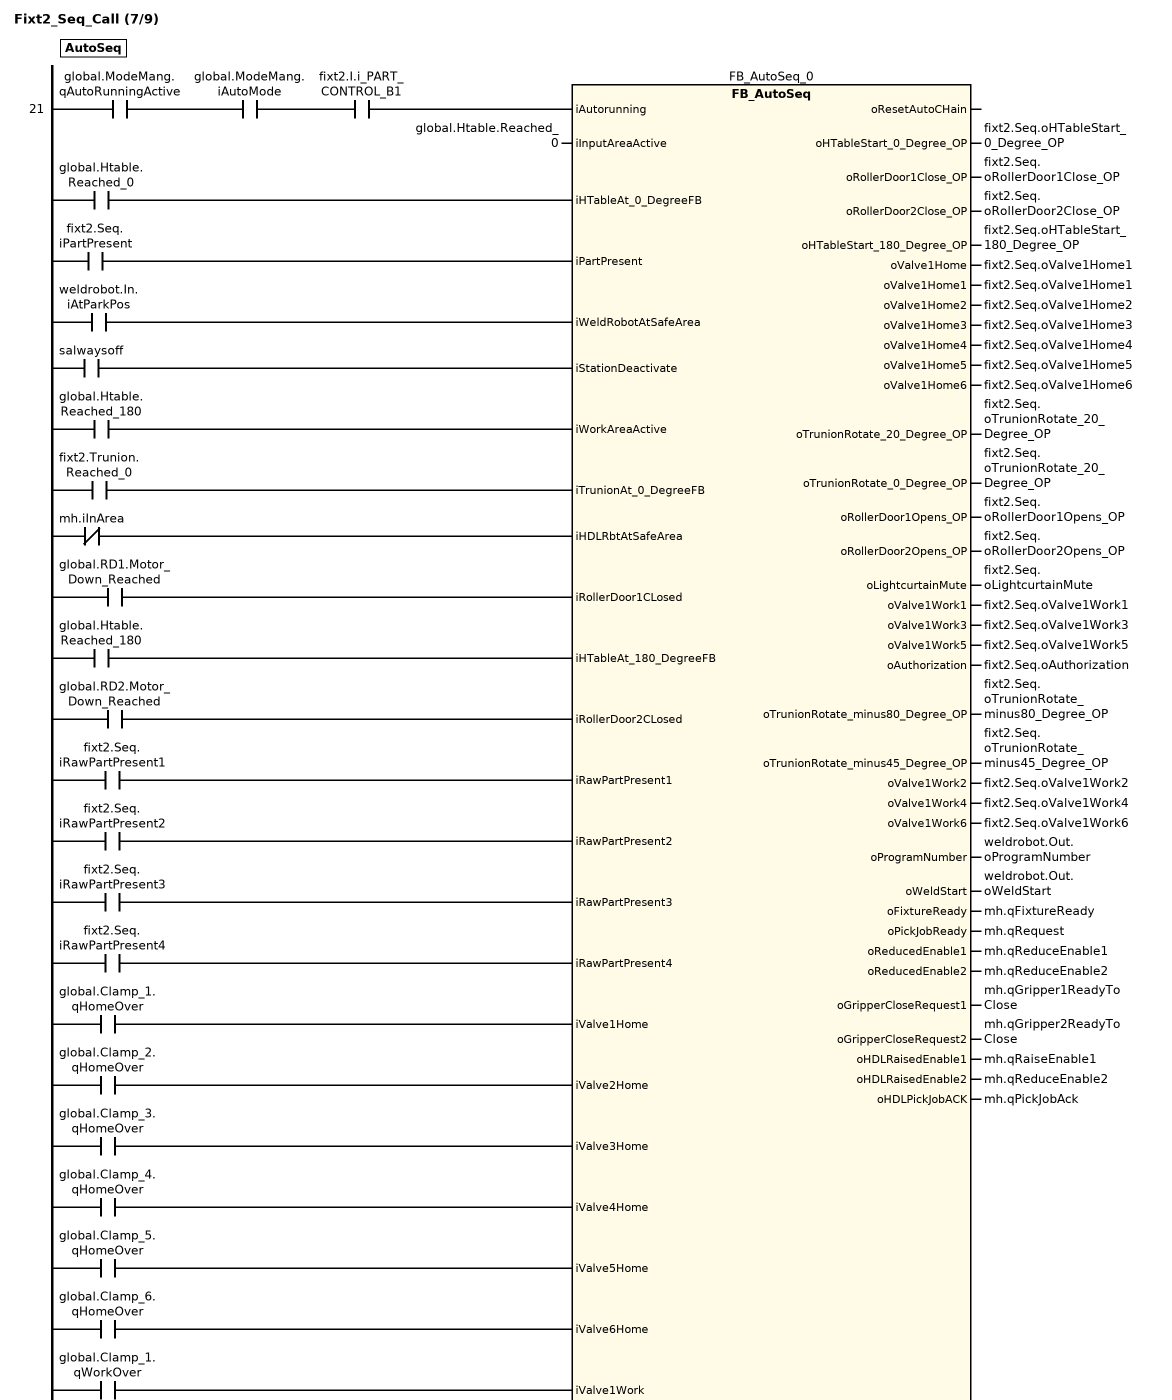
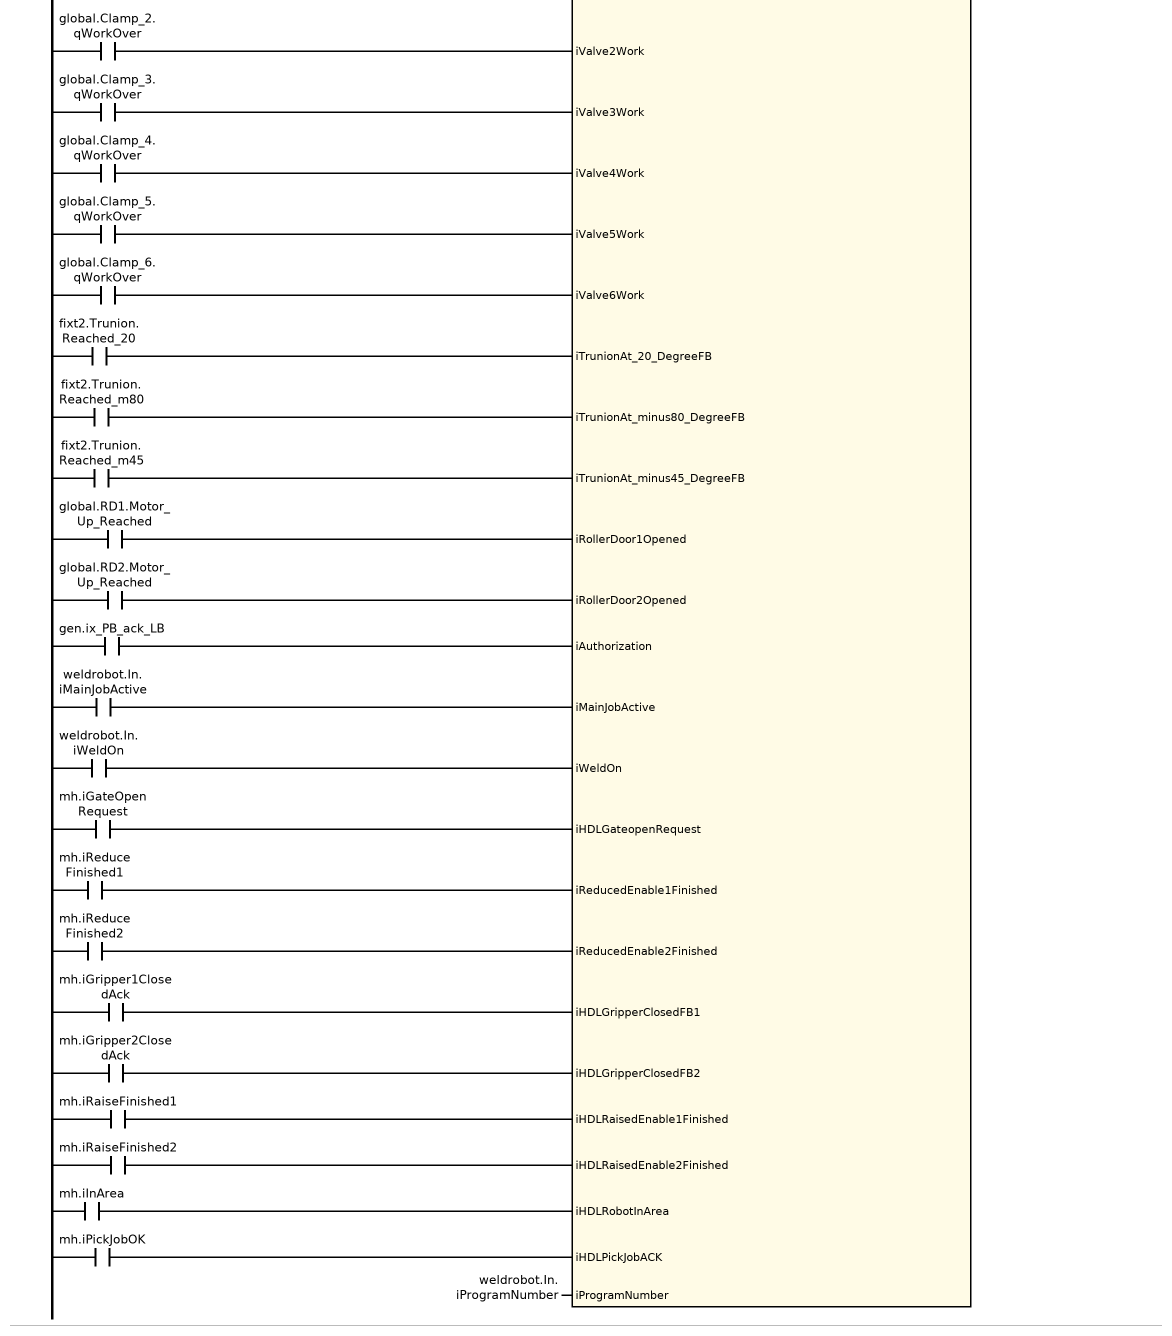
// NETWORK 21
AutoSeq:
FB_AutoSeq_0(
    iAutorunning := global.ModeMang.qAutoRunningActive AND global.ModeMang.iAutoMode AND fixt2.I.i_PART_CONTROL_B1,
    iInputAreaActive := global.Htable.Reached_0,
    iHTableAt_0_DegreeFB := global.Htable.Reached_0,
    iPartPresent := fixt2.Seq.iPartPresent,
    iWeldRobotAtSafeArea := weldrobot.In.iAtParkPos,
    iStationDeactivate := salwaysoff,
    iWorkAreaActive := global.Htable.Reached_180,
    iTrunionAt_0_DegreeFB := fixt2.Trunion.Reached_0,
    iHDLRbtAtSafeArea := NOT mh.iInArea,
    iRollerDoor1CLosed := global.RD1.Motor_Down_Reached,
    iHTableAt_180_DegreeFB := global.Htable.Reached_180,
    iRollerDoor2CLosed := global.RD2.Motor_Down_Reached,
    iRawPartPresent1 := fixt2.Seq.iRawPartPresent1,
    iRawPartPresent2 := fixt2.Seq.iRawPartPresent2,
    iRawPartPresent3 := fixt2.Seq.iRawPartPresent3,
    iRawPartPresent4 := fixt2.Seq.iRawPartPresent4,
    iValve1Home := global.Clamp_1.qHomeOver,
    iValve2Home := global.Clamp_2.qHomeOver,
    iValve3Home := global.Clamp_3.qHomeOver,
    iValve4Home := global.Clamp_4.qHomeOver,
    iValve5Home := global.Clamp_5.qHomeOver,
    iValve6Home := global.Clamp_6.qHomeOver,
    iValve1Work := global.Clamp_1.qWorkOver,
    iValve2Work := global.Clamp_2.qWorkOver,
    iValve3Work := global.Clamp_3.qWorkOver,
    iValve4Work := global.Clamp_4.qWorkOver,
    iValve5Work := global.Clamp_5.qWorkOver,
    iValve6Work := global.Clamp_6.qWorkOver,
    iTrunionAt_20_DegreeFB := fixt2.Trunion.Reached_20,
    iTrunionAt_minus80_DegreeFB := fixt2.Trunion.Reached_m80,
    iTrunionAt_minus45_DegreeFB := fixt2.Trunion.Reached_m45,
    iRollerDoor1Opened := global.RD1.Motor_Up_Reached,
    iRollerDoor2Opened := global.RD2.Motor_Up_Reached,
    iAuthorization := gen.ix_PB_ack_LB,
    iMainJobActive := weldrobot.In.iMainJobActive,
    iWeldOn := weldrobot.In.iWeldOn,
    iHDLGateopenRequest := mh.iGateOpenRequest,
    iReducedEnable1Finished := mh.iReduceFinished1,
    iReducedEnable2Finished := mh.iReduceFinished2,
    iHDLGripperClosedFB1 := mh.iGripper1ClosedAck,
    iHDLGripperClosedFB2 := mh.iGripper2ClosedAck,
    iHDLRaisedEnable1Finished := mh.iRaiseFinished1,
    iHDLRaisedEnable2Finished := mh.iRaiseFinished2,
    iHDLRobotInArea := mh.iInArea,
    iHDLPickJobACK := mh.iPickJobOK,
    iProgramNumber := weldrobot.In.iProgramNumber,
    oHTableStart_0_Degree_OP => fixt2.Seq.oHTableStart_0_Degree_OP,
    oRollerDoor1Close_OP => fixt2.Seq.oRollerDoor1Close_OP,
    oRollerDoor2Close_OP => fixt2.Seq.oRollerDoor2Close_OP,
    oHTableStart_180_Degree_OP => fixt2.Seq.oHTableStart_180_Degree_OP,
    oValve1Home => fixt2.Seq.oValve1Home1,
    oValve1Home1 => fixt2.Seq.oValve1Home1,
    oValve1Home2 => fixt2.Seq.oValve1Home2,
    oValve1Home3 => fixt2.Seq.oValve1Home3,
    oValve1Home4 => fixt2.Seq.oValve1Home4,
    oValve1Home5 => fixt2.Seq.oValve1Home5,
    oValve1Home6 => fixt2.Seq.oValve1Home6,
    oTrunionRotate_20_Degree_OP => fixt2.Seq.oTrunionRotate_20_Degree_OP,
    oTrunionRotate_0_Degree_OP => fixt2.Seq.oTrunionRotate_20_Degree_OP,
    oRollerDoor1Opens_OP => fixt2.Seq.oRollerDoor1Opens_OP,
    oRollerDoor2Opens_OP => fixt2.Seq.oRollerDoor2Opens_OP,
    oLightcurtainMute => fixt2.Seq.oLightcurtainMute,
    oValve1Work1 => fixt2.Seq.oValve1Work1,
    oValve1Work3 => fixt2.Seq.oValve1Work3,
    oValve1Work5 => fixt2.Seq.oValve1Work5,
    oAuthorization => fixt2.Seq.oAuthorization,
    oTrunionRotate_minus80_Degree_OP => fixt2.Seq.oTrunionRotate_minus80_Degree_OP,
    oTrunionRotate_minus45_Degree_OP => fixt2.Seq.oTrunionRotate_minus45_Degree_OP,
    oValve1Work2 => fixt2.Seq.oValve1Work2,
    oValve1Work4 => fixt2.Seq.oValve1Work4,
    oValve1Work6 => fixt2.Seq.oValve1Work6,
    oProgramNumber => weldrobot.Out.oProgramNumber,
    oWeldStart => weldrobot.Out.oWeldStart,
    oFixtureReady => mh.qFixtureReady,
    oPickJobReady => mh.qRequest,
    oReducedEnable1 => mh.qReduceEnable1,
    oReducedEnable2 => mh.qReduceEnable2,
    oGripperCloseRequest1 => mh.qGripper1ReadyToClose,
    oGripperCloseRequest2 => mh.qGripper2ReadyToClose,
    oHDLRaisedEnable1 => mh.qRaiseEnable1,
    oHDLRaisedEnable2 => mh.qReduceEnable2,
    oHDLPickJobACK => mh.qPickJobAck); // FB_AutoSeq

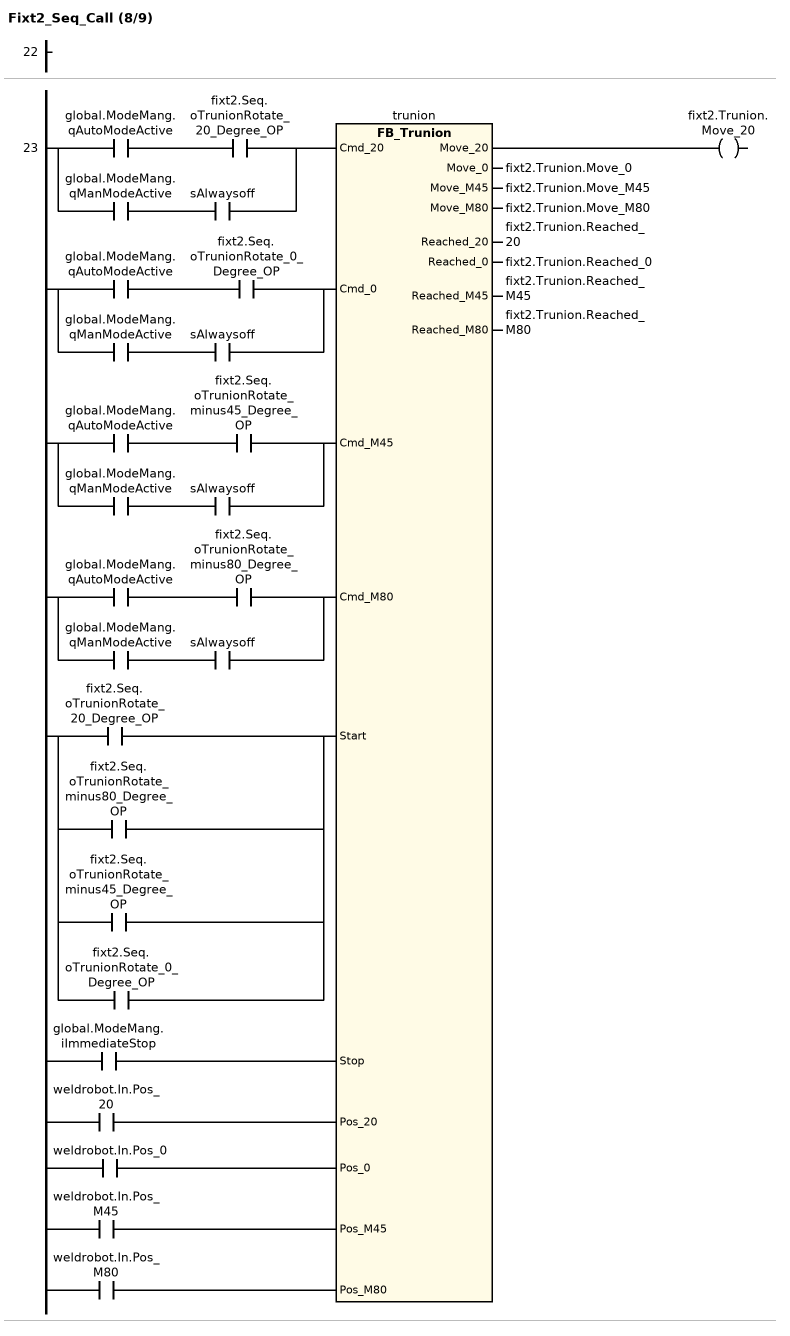
// NETWORK 22

// NETWORK 23
trunion(
    Cmd_20 := global.ModeMang.qAutoModeActive AND fixt2.Seq.oTrunionRotate_20_Degree_OP OR global.ModeMang.qManModeActive AND sAlwaysoff,
    Cmd_0 := global.ModeMang.qAutoModeActive AND fixt2.Seq.oTrunionRotate_0_Degree_OP OR global.ModeMang.qManModeActive AND sAlwaysoff,
    Cmd_M45 := global.ModeMang.qAutoModeActive AND fixt2.Seq.oTrunionRotate_minus45_Degree_OP OR global.ModeMang.qManModeActive AND sAlwaysoff,
    Cmd_M80 := global.ModeMang.qAutoModeActive AND fixt2.Seq.oTrunionRotate_minus80_Degree_OP OR global.ModeMang.qManModeActive AND sAlwaysoff,
    Start := fixt2.Seq.oTrunionRotate_20_Degree_OP OR fixt2.Seq.oTrunionRotate_minus80_Degree_OP OR fixt2.Seq.oTrunionRotate_minus45_Degree_OP OR fixt2.Seq.oTrunionRotate_0_Degree_OP,
    Stop := global.ModeMang.iImmediateStop,
    Pos_20 := weldrobot.In.Pos_20,
    Pos_0 := weldrobot.In.Pos_0,
    Pos_M45 := weldrobot.In.Pos_M45,
    Pos_M80 := weldrobot.In.Pos_M80,
    Move_0 => fixt2.Trunion.Move_0,
    Move_M45 => fixt2.Trunion.Move_M45,
    Move_M80 => fixt2.Trunion.Move_M80,
    Reached_20 => fixt2.Trunion.Reached_20,
    Reached_0 => fixt2.Trunion.Reached_0,
    Reached_M45 => fixt2.Trunion.Reached_M45,
    Reached_M80 => fixt2.Trunion.Reached_M80); // FB_Trunion
fixt2.Trunion.Move_20 := trunion.Move_20;

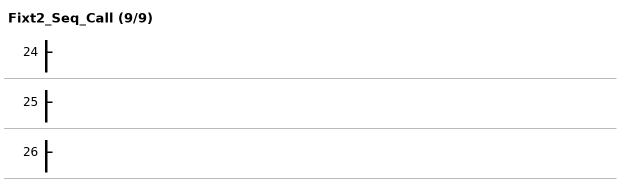
// NETWORK 24

// NETWORK 25

// NETWORK 26

END_PROGRAM

// ---- POUs/Library/FB_PartMonitoring_Fixt2.TcPOU
FUNCTION_BLOCK FB_PartMonitoring_Fixt2
VAR_INPUT
END_VAR
VAR_OUTPUT
	qRawPart1:BOOL;
	qRawPart2:BOOL;
	qRawPart3:BOOL;
	qRawPart4:BOOL;
	qAllPartPresent:BOOL;
	
END_VAR
VAR
END_VAR

qRawPart1:= (
             fixt2.I.i_PART_CONTROL_B1 AND fixt2.I.i_PART_CONTROL_B2 AND fixt2.I.i_PART_CONTROL_B3 AND fixt2.I.i_PART_CONTROL_B4
			 AND fixt2.I.i_PART_CONTROL_B5 AND fixt2.I.i_PART_CONTROL_B6 AND fixt2.I.i_PART_CONTROL_B7
			 );
qRawPart2:= (
             fixt2.I.i_PART_CONTROL_B15 AND fixt2.I.i_PART_CONTROL_B16 AND fixt2.I.i_PART_CONTROL_B17 AND fixt2.I.i_PART_CONTROL_B18
			 AND fixt2.I.i_PART_CONTROL_B19 AND fixt2.I.i_PART_CONTROL_B20 AND fixt2.I.i_PART_CONTROL_B21
			 );
qRawPart3:= (
             fixt2.I.i_PART_CONTROL_B8 AND fixt2.I.i_PART_CONTROL_B9 AND fixt2.I.i_PART_CONTROL_B10 AND fixt2.I.i_PART_CONTROL_B11
			 AND fixt2.I.i_PART_CONTROL_B12 AND fixt2.I.i_PART_CONTROL_B13 AND fixt2.I.i_PART_CONTROL_B14
			 );
qRawPart4:= (
             fixt2.I.i_PART_CONTROL_B22 AND fixt2.I.i_PART_CONTROL_B23 AND fixt2.I.i_PART_CONTROL_B24 AND fixt2.I.i_PART_CONTROL_B25
			 AND fixt2.I.i_PART_CONTROL_B26 AND fixt2.I.i_PART_CONTROL_B27 AND fixt2.I.i_PART_CONTROL_B28
			 );			 
			 
qAllPartPresent:= (
             fixt2.I.i_PART_CONTROL_B22 AND fixt2.I.i_PART_CONTROL_B23 AND fixt2.I.i_PART_CONTROL_B24 AND fixt2.I.i_PART_CONTROL_B25
			 AND fixt2.I.i_PART_CONTROL_B26 AND fixt2.I.i_PART_CONTROL_B27 AND fixt2.I.i_PART_CONTROL_B28
			 AND fixt2.I.i_PART_CONTROL_B1 AND fixt2.I.i_PART_CONTROL_B2 AND fixt2.I.i_PART_CONTROL_B3 AND fixt2.I.i_PART_CONTROL_B4
			 AND fixt2.I.i_PART_CONTROL_B5 AND fixt2.I.i_PART_CONTROL_B6 AND fixt2.I.i_PART_CONTROL_B7
			 AND fixt2.I.i_PART_CONTROL_B15 AND fixt2.I.i_PART_CONTROL_B16 AND fixt2.I.i_PART_CONTROL_B17 AND fixt2.I.i_PART_CONTROL_B18
			 AND fixt2.I.i_PART_CONTROL_B19 AND fixt2.I.i_PART_CONTROL_B20 AND fixt2.I.i_PART_CONTROL_B21
             AND fixt2.I.i_PART_CONTROL_B8 AND fixt2.I.i_PART_CONTROL_B9 AND fixt2.I.i_PART_CONTROL_B10 AND fixt2.I.i_PART_CONTROL_B11
			 AND fixt2.I.i_PART_CONTROL_B12 AND fixt2.I.i_PART_CONTROL_B13 AND fixt2.I.i_PART_CONTROL_B14 
			 );

END_FUNCTION_BLOCK

// ---- POUs/Fixt2_Seq_Call_1.TcPOU
PROGRAM Fixt2_Seq_Call_1
VAR
	Clamp_1: FB_CylinderModule;
	Clamp_2: FB_CylinderModule;
	Clamp_3: FB_CylinderModule;
	Clamp_4: FB_CylinderModule;
	Clamp_5: FB_CylinderModule;
	Clamp_6: FB_CylinderModule;
	sAlwaysoff: BOOL;
	FB_AutoSeq_0: FB_AutoSeq;
	alwayson:BOOL;
	partmonitor:FB_PartMonitoring_fixt2;
	trunion:FB_Trunion;
END_VAR
VAR // added by the converter: edge detectors and wires of the graphical bodies
    _w1, _w2, _w3, _w4, _w5, _w6 : BOOL;
END_VAR

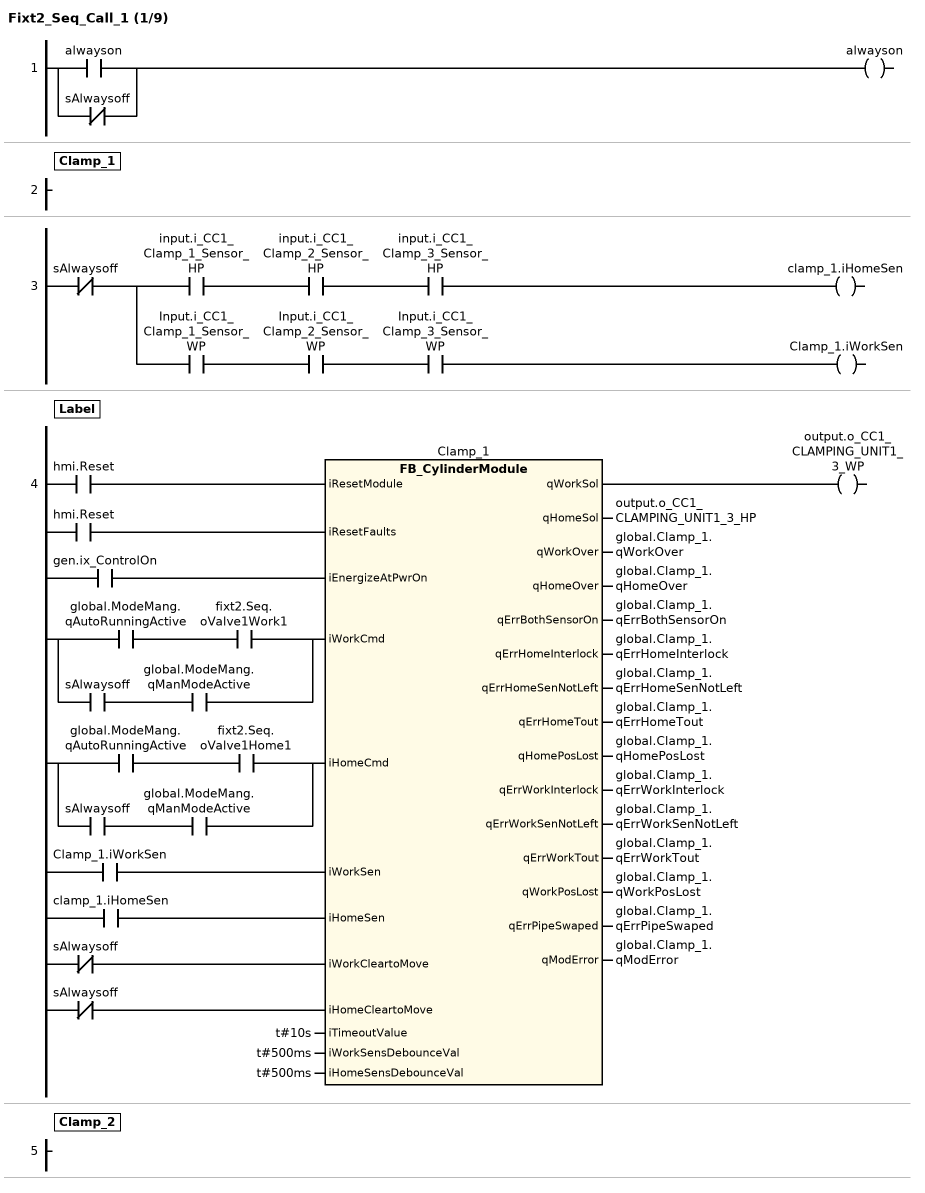
// NETWORK 1
alwayson := alwayson OR NOT sAlwaysoff;

// NETWORK 2
Clamp_1: ;

// NETWORK 3
_w1 := NOT sAlwaysoff;
clamp_1.iHomeSen := _w1 AND input.i_CC1_Clamp_1_Sensor_HP AND input.i_CC1_Clamp_2_Sensor_HP AND input.i_CC1_Clamp_3_Sensor_HP;
Clamp_1.iWorkSen := _w1 AND Input.i_CC1_Clamp_1_Sensor_WP AND Input.i_CC1_Clamp_2_Sensor_WP AND Input.i_CC1_Clamp_3_Sensor_WP;

// NETWORK 4
Label:
Clamp_1(
    iResetModule := hmi.Reset,
    iResetFaults := hmi.Reset,
    iEnergizeAtPwrOn := gen.ix_ControlOn,
    iWorkCmd := global.ModeMang.qAutoRunningActive AND fixt2.Seq.oValve1Work1 OR sAlwaysoff AND global.ModeMang.qManModeActive,
    iHomeCmd := global.ModeMang.qAutoRunningActive AND fixt2.Seq.oValve1Home1 OR sAlwaysoff AND global.ModeMang.qManModeActive,
    iWorkSen := Clamp_1.iWorkSen,
    iHomeSen := clamp_1.iHomeSen,
    iWorkCleartoMove := NOT sAlwaysoff,
    iHomeCleartoMove := NOT sAlwaysoff,
    iTimeoutValue := t#10s,
    iWorkSensDebounceVal := t#500ms,
    iHomeSensDebounceVal := t#500ms,
    qHomeSol => output.o_CC1_CLAMPING_UNIT1_3_HP,
    qWorkOver => global.Clamp_1.qWorkOver,
    qHomeOver => global.Clamp_1.qHomeOver,
    qErrBothSensorOn => global.Clamp_1.qErrBothSensorOn,
    qErrHomeInterlock => global.Clamp_1.qErrHomeInterlock,
    qErrHomeSenNotLeft => global.Clamp_1.qErrHomeSenNotLeft,
    qErrHomeTout => global.Clamp_1.qErrHomeTout,
    qHomePosLost => global.Clamp_1.qHomePosLost,
    qErrWorkInterlock => global.Clamp_1.qErrWorkInterlock,
    qErrWorkSenNotLeft => global.Clamp_1.qErrWorkSenNotLeft,
    qErrWorkTout => global.Clamp_1.qErrWorkTout,
    qWorkPosLost => global.Clamp_1.qWorkPosLost,
    qErrPipeSwaped => global.Clamp_1.qErrPipeSwaped,
    qModError => global.Clamp_1.qModError); // FB_CylinderModule
output.o_CC1_CLAMPING_UNIT1_3_WP := Clamp_1.qWorkSol;

// NETWORK 5
Clamp_2: ;

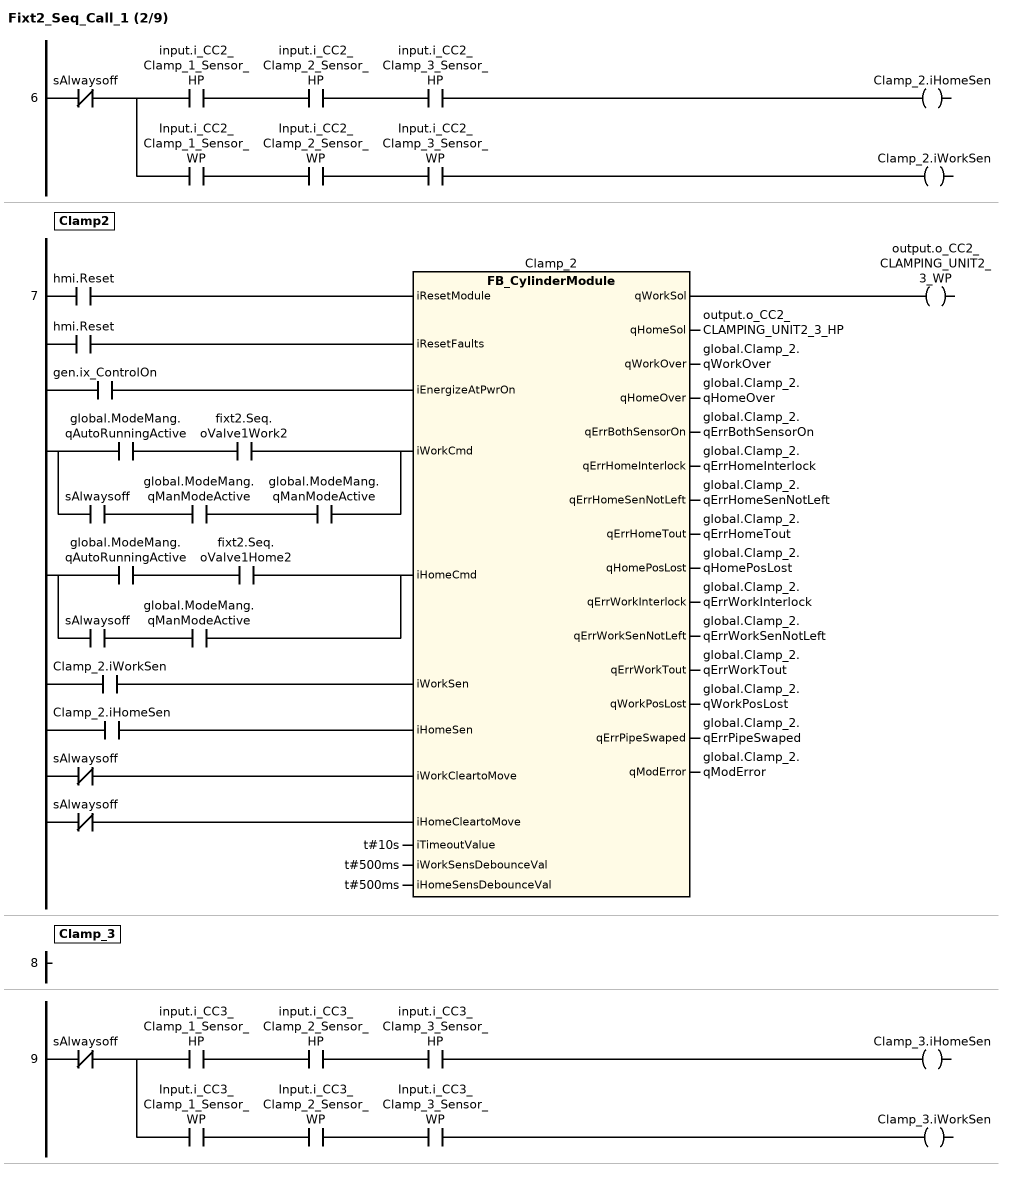
// NETWORK 6
_w2 := NOT sAlwaysoff;
Clamp_2.iHomeSen := _w2 AND input.i_CC2_Clamp_1_Sensor_HP AND input.i_CC2_Clamp_2_Sensor_HP AND input.i_CC2_Clamp_3_Sensor_HP;
Clamp_2.iWorkSen := _w2 AND Input.i_CC2_Clamp_1_Sensor_WP AND Input.i_CC2_Clamp_2_Sensor_WP AND Input.i_CC2_Clamp_3_Sensor_WP;

// NETWORK 7
Clamp2:
Clamp_2(
    iResetModule := hmi.Reset,
    iResetFaults := hmi.Reset,
    iEnergizeAtPwrOn := gen.ix_ControlOn,
    iWorkCmd := global.ModeMang.qAutoRunningActive AND fixt2.Seq.oValve1Work2 OR sAlwaysoff AND global.ModeMang.qManModeActive AND global.ModeMang.qManModeActive,
    iHomeCmd := global.ModeMang.qAutoRunningActive AND fixt2.Seq.oValve1Home2 OR sAlwaysoff AND global.ModeMang.qManModeActive,
    iWorkSen := Clamp_2.iWorkSen,
    iHomeSen := Clamp_2.iHomeSen,
    iWorkCleartoMove := NOT sAlwaysoff,
    iHomeCleartoMove := NOT sAlwaysoff,
    iTimeoutValue := t#10s,
    iWorkSensDebounceVal := t#500ms,
    iHomeSensDebounceVal := t#500ms,
    qHomeSol => output.o_CC2_CLAMPING_UNIT2_3_HP,
    qWorkOver => global.Clamp_2.qWorkOver,
    qHomeOver => global.Clamp_2.qHomeOver,
    qErrBothSensorOn => global.Clamp_2.qErrBothSensorOn,
    qErrHomeInterlock => global.Clamp_2.qErrHomeInterlock,
    qErrHomeSenNotLeft => global.Clamp_2.qErrHomeSenNotLeft,
    qErrHomeTout => global.Clamp_2.qErrHomeTout,
    qHomePosLost => global.Clamp_2.qHomePosLost,
    qErrWorkInterlock => global.Clamp_2.qErrWorkInterlock,
    qErrWorkSenNotLeft => global.Clamp_2.qErrWorkSenNotLeft,
    qErrWorkTout => global.Clamp_2.qErrWorkTout,
    qWorkPosLost => global.Clamp_2.qWorkPosLost,
    qErrPipeSwaped => global.Clamp_2.qErrPipeSwaped,
    qModError => global.Clamp_2.qModError); // FB_CylinderModule
output.o_CC2_CLAMPING_UNIT2_3_WP := Clamp_2.qWorkSol;

// NETWORK 8
Clamp_3: ;

// NETWORK 9
_w3 := NOT sAlwaysoff;
Clamp_3.iHomeSen := _w3 AND input.i_CC3_Clamp_1_Sensor_HP AND input.i_CC3_Clamp_2_Sensor_HP AND input.i_CC3_Clamp_3_Sensor_HP;
Clamp_3.iWorkSen := _w3 AND Input.i_CC3_Clamp_1_Sensor_WP AND Input.i_CC3_Clamp_2_Sensor_WP AND Input.i_CC3_Clamp_3_Sensor_WP;

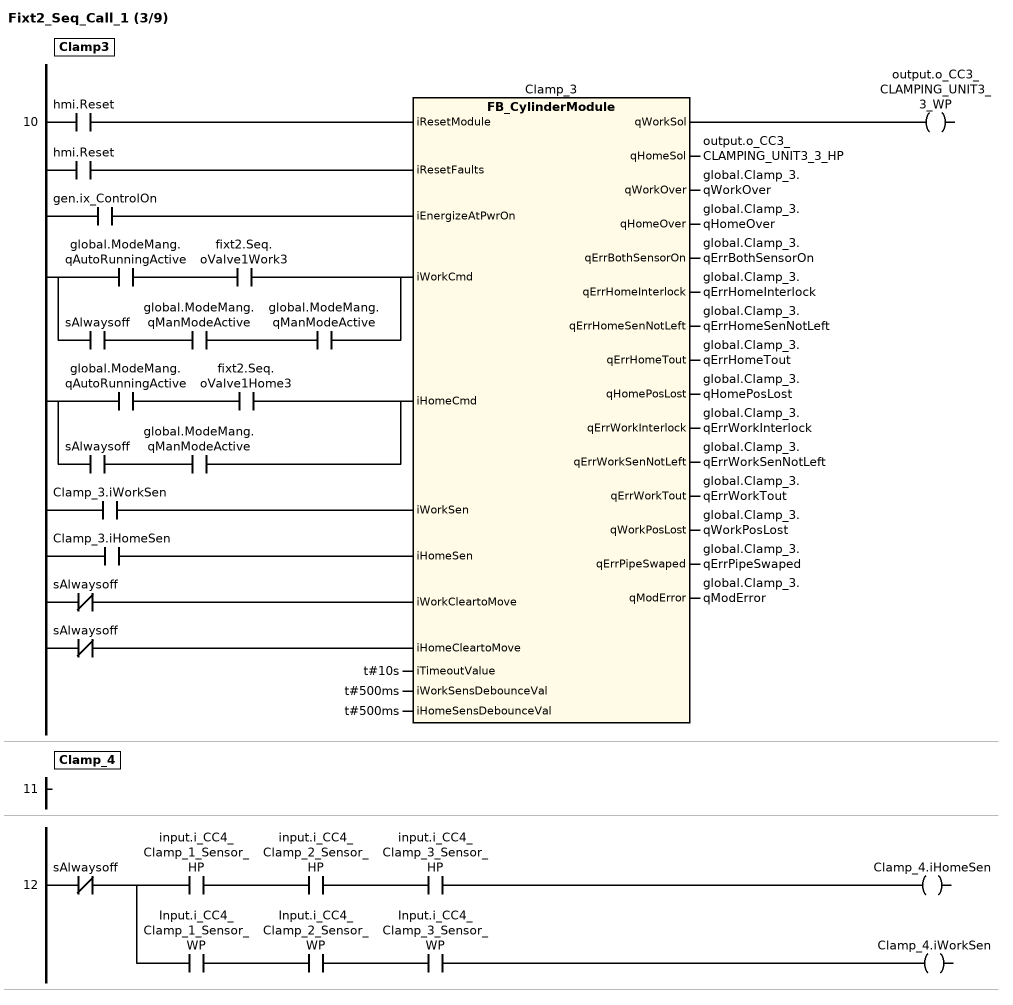
// NETWORK 10
Clamp3:
Clamp_3(
    iResetModule := hmi.Reset,
    iResetFaults := hmi.Reset,
    iEnergizeAtPwrOn := gen.ix_ControlOn,
    iWorkCmd := global.ModeMang.qAutoRunningActive AND fixt2.Seq.oValve1Work3 OR sAlwaysoff AND global.ModeMang.qManModeActive AND global.ModeMang.qManModeActive,
    iHomeCmd := global.ModeMang.qAutoRunningActive AND fixt2.Seq.oValve1Home3 OR sAlwaysoff AND global.ModeMang.qManModeActive,
    iWorkSen := Clamp_3.iWorkSen,
    iHomeSen := Clamp_3.iHomeSen,
    iWorkCleartoMove := NOT sAlwaysoff,
    iHomeCleartoMove := NOT sAlwaysoff,
    iTimeoutValue := t#10s,
    iWorkSensDebounceVal := t#500ms,
    iHomeSensDebounceVal := t#500ms,
    qHomeSol => output.o_CC3_CLAMPING_UNIT3_3_HP,
    qWorkOver => global.Clamp_3.qWorkOver,
    qHomeOver => global.Clamp_3.qHomeOver,
    qErrBothSensorOn => global.Clamp_3.qErrBothSensorOn,
    qErrHomeInterlock => global.Clamp_3.qErrHomeInterlock,
    qErrHomeSenNotLeft => global.Clamp_3.qErrHomeSenNotLeft,
    qErrHomeTout => global.Clamp_3.qErrHomeTout,
    qHomePosLost => global.Clamp_3.qHomePosLost,
    qErrWorkInterlock => global.Clamp_3.qErrWorkInterlock,
    qErrWorkSenNotLeft => global.Clamp_3.qErrWorkSenNotLeft,
    qErrWorkTout => global.Clamp_3.qErrWorkTout,
    qWorkPosLost => global.Clamp_3.qWorkPosLost,
    qErrPipeSwaped => global.Clamp_3.qErrPipeSwaped,
    qModError => global.Clamp_3.qModError); // FB_CylinderModule
output.o_CC3_CLAMPING_UNIT3_3_WP := Clamp_3.qWorkSol;

// NETWORK 11
Clamp_4: ;

// NETWORK 12
_w4 := NOT sAlwaysoff;
Clamp_4.iHomeSen := _w4 AND input.i_CC4_Clamp_1_Sensor_HP AND input.i_CC4_Clamp_2_Sensor_HP AND input.i_CC4_Clamp_3_Sensor_HP;
Clamp_4.iWorkSen := _w4 AND Input.i_CC4_Clamp_1_Sensor_WP AND Input.i_CC4_Clamp_2_Sensor_WP AND Input.i_CC4_Clamp_3_Sensor_WP;

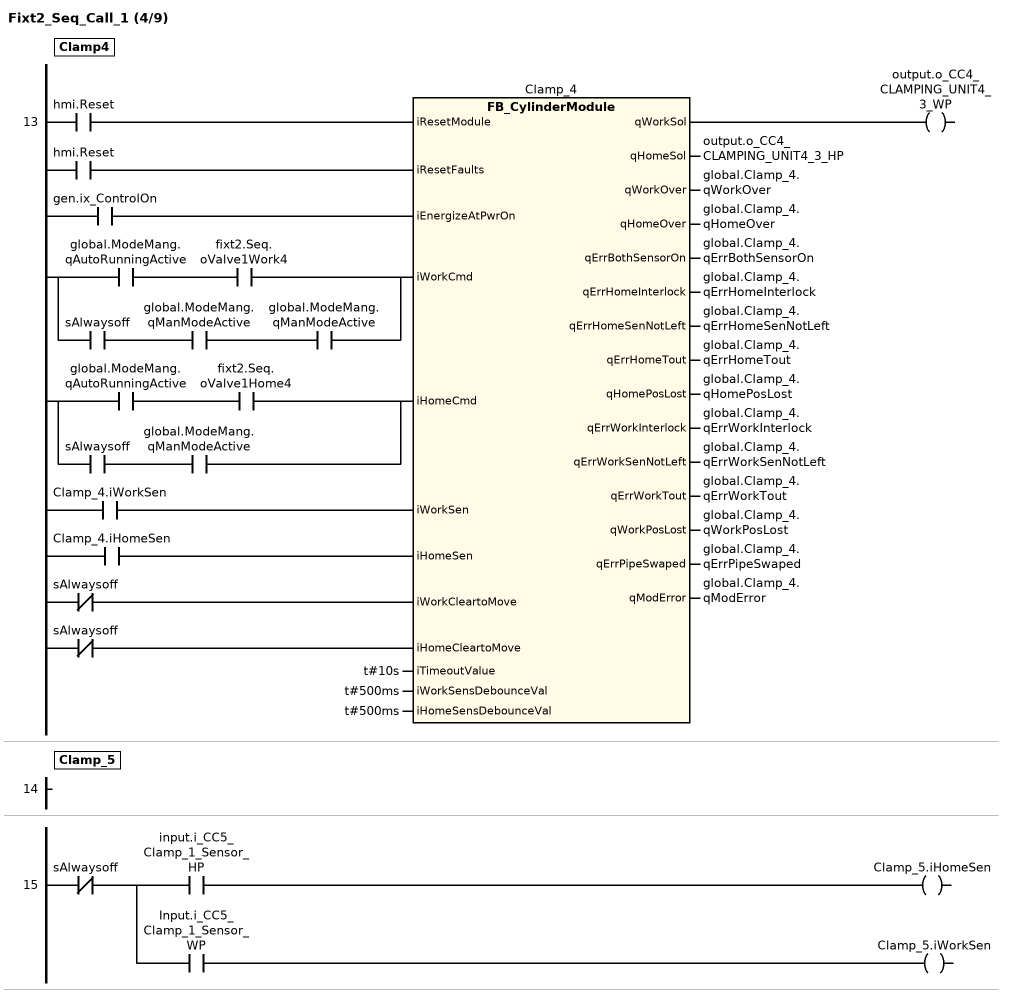
// NETWORK 13
Clamp4:
Clamp_4(
    iResetModule := hmi.Reset,
    iResetFaults := hmi.Reset,
    iEnergizeAtPwrOn := gen.ix_ControlOn,
    iWorkCmd := global.ModeMang.qAutoRunningActive AND fixt2.Seq.oValve1Work4 OR sAlwaysoff AND global.ModeMang.qManModeActive AND global.ModeMang.qManModeActive,
    iHomeCmd := global.ModeMang.qAutoRunningActive AND fixt2.Seq.oValve1Home4 OR sAlwaysoff AND global.ModeMang.qManModeActive,
    iWorkSen := Clamp_4.iWorkSen,
    iHomeSen := Clamp_4.iHomeSen,
    iWorkCleartoMove := NOT sAlwaysoff,
    iHomeCleartoMove := NOT sAlwaysoff,
    iTimeoutValue := t#10s,
    iWorkSensDebounceVal := t#500ms,
    iHomeSensDebounceVal := t#500ms,
    qHomeSol => output.o_CC4_CLAMPING_UNIT4_3_HP,
    qWorkOver => global.Clamp_4.qWorkOver,
    qHomeOver => global.Clamp_4.qHomeOver,
    qErrBothSensorOn => global.Clamp_4.qErrBothSensorOn,
    qErrHomeInterlock => global.Clamp_4.qErrHomeInterlock,
    qErrHomeSenNotLeft => global.Clamp_4.qErrHomeSenNotLeft,
    qErrHomeTout => global.Clamp_4.qErrHomeTout,
    qHomePosLost => global.Clamp_4.qHomePosLost,
    qErrWorkInterlock => global.Clamp_4.qErrWorkInterlock,
    qErrWorkSenNotLeft => global.Clamp_4.qErrWorkSenNotLeft,
    qErrWorkTout => global.Clamp_4.qErrWorkTout,
    qWorkPosLost => global.Clamp_4.qWorkPosLost,
    qErrPipeSwaped => global.Clamp_4.qErrPipeSwaped,
    qModError => global.Clamp_4.qModError); // FB_CylinderModule
output.o_CC4_CLAMPING_UNIT4_3_WP := Clamp_4.qWorkSol;

// NETWORK 14
Clamp_5: ;

// NETWORK 15
_w5 := NOT sAlwaysoff;
Clamp_5.iHomeSen := _w5 AND input.i_CC5_Clamp_1_Sensor_HP;
Clamp_5.iWorkSen := _w5 AND Input.i_CC5_Clamp_1_Sensor_WP;

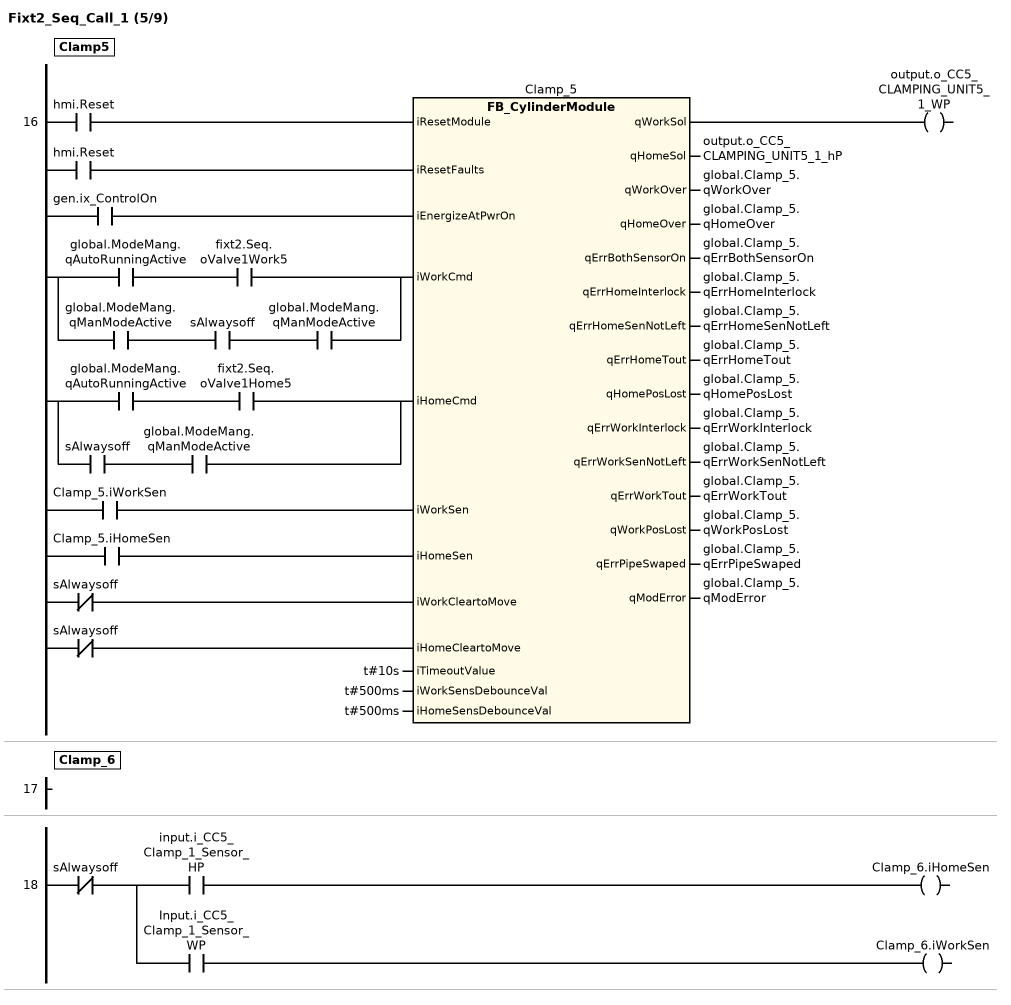
// NETWORK 16
Clamp5:
Clamp_5(
    iResetModule := hmi.Reset,
    iResetFaults := hmi.Reset,
    iEnergizeAtPwrOn := gen.ix_ControlOn,
    iWorkCmd := global.ModeMang.qAutoRunningActive AND fixt2.Seq.oValve1Work5 OR global.ModeMang.qManModeActive AND sAlwaysoff AND global.ModeMang.qManModeActive,
    iHomeCmd := global.ModeMang.qAutoRunningActive AND fixt2.Seq.oValve1Home5 OR sAlwaysoff AND global.ModeMang.qManModeActive,
    iWorkSen := Clamp_5.iWorkSen,
    iHomeSen := Clamp_5.iHomeSen,
    iWorkCleartoMove := NOT sAlwaysoff,
    iHomeCleartoMove := NOT sAlwaysoff,
    iTimeoutValue := t#10s,
    iWorkSensDebounceVal := t#500ms,
    iHomeSensDebounceVal := t#500ms,
    qHomeSol => output.o_CC5_CLAMPING_UNIT5_1_hP,
    qWorkOver => global.Clamp_5.qWorkOver,
    qHomeOver => global.Clamp_5.qHomeOver,
    qErrBothSensorOn => global.Clamp_5.qErrBothSensorOn,
    qErrHomeInterlock => global.Clamp_5.qErrHomeInterlock,
    qErrHomeSenNotLeft => global.Clamp_5.qErrHomeSenNotLeft,
    qErrHomeTout => global.Clamp_5.qErrHomeTout,
    qHomePosLost => global.Clamp_5.qHomePosLost,
    qErrWorkInterlock => global.Clamp_5.qErrWorkInterlock,
    qErrWorkSenNotLeft => global.Clamp_5.qErrWorkSenNotLeft,
    qErrWorkTout => global.Clamp_5.qErrWorkTout,
    qWorkPosLost => global.Clamp_5.qWorkPosLost,
    qErrPipeSwaped => global.Clamp_5.qErrPipeSwaped,
    qModError => global.Clamp_5.qModError); // FB_CylinderModule
output.o_CC5_CLAMPING_UNIT5_1_WP := Clamp_5.qWorkSol;

// NETWORK 17
Clamp_6: ;

// NETWORK 18
_w6 := NOT sAlwaysoff;
Clamp_6.iHomeSen := _w6 AND input.i_CC5_Clamp_1_Sensor_HP;
Clamp_6.iWorkSen := _w6 AND Input.i_CC5_Clamp_1_Sensor_WP;

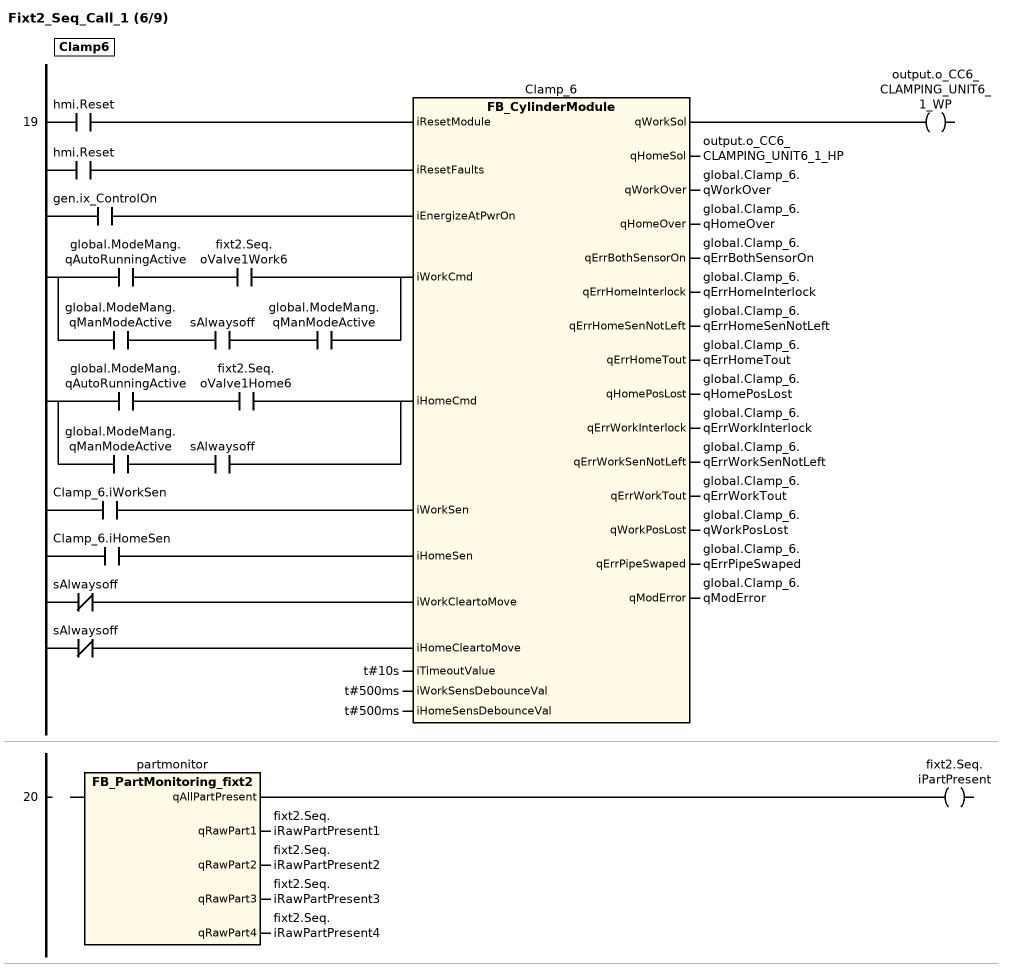
// NETWORK 19
Clamp6:
Clamp_6(
    iResetModule := hmi.Reset,
    iResetFaults := hmi.Reset,
    iEnergizeAtPwrOn := gen.ix_ControlOn,
    iWorkCmd := global.ModeMang.qAutoRunningActive AND fixt2.Seq.oValve1Work6 OR global.ModeMang.qManModeActive AND sAlwaysoff AND global.ModeMang.qManModeActive,
    iHomeCmd := global.ModeMang.qAutoRunningActive AND fixt2.Seq.oValve1Home6 OR global.ModeMang.qManModeActive AND sAlwaysoff,
    iWorkSen := Clamp_6.iWorkSen,
    iHomeSen := Clamp_6.iHomeSen,
    iWorkCleartoMove := NOT sAlwaysoff,
    iHomeCleartoMove := NOT sAlwaysoff,
    iTimeoutValue := t#10s,
    iWorkSensDebounceVal := t#500ms,
    iHomeSensDebounceVal := t#500ms,
    qHomeSol => output.o_CC6_CLAMPING_UNIT6_1_HP,
    qWorkOver => global.Clamp_6.qWorkOver,
    qHomeOver => global.Clamp_6.qHomeOver,
    qErrBothSensorOn => global.Clamp_6.qErrBothSensorOn,
    qErrHomeInterlock => global.Clamp_6.qErrHomeInterlock,
    qErrHomeSenNotLeft => global.Clamp_6.qErrHomeSenNotLeft,
    qErrHomeTout => global.Clamp_6.qErrHomeTout,
    qHomePosLost => global.Clamp_6.qHomePosLost,
    qErrWorkInterlock => global.Clamp_6.qErrWorkInterlock,
    qErrWorkSenNotLeft => global.Clamp_6.qErrWorkSenNotLeft,
    qErrWorkTout => global.Clamp_6.qErrWorkTout,
    qWorkPosLost => global.Clamp_6.qWorkPosLost,
    qErrPipeSwaped => global.Clamp_6.qErrPipeSwaped,
    qModError => global.Clamp_6.qModError); // FB_CylinderModule
output.o_CC6_CLAMPING_UNIT6_1_WP := Clamp_6.qWorkSol;

// NETWORK 20
partmonitor(
    qRawPart1 => fixt2.Seq.iRawPartPresent1,
    qRawPart2 => fixt2.Seq.iRawPartPresent2,
    qRawPart3 => fixt2.Seq.iRawPartPresent3,
    qRawPart4 => fixt2.Seq.iRawPartPresent4); // FB_PartMonitoring_fixt2
fixt2.Seq.iPartPresent := partmonitor.qAllPartPresent;

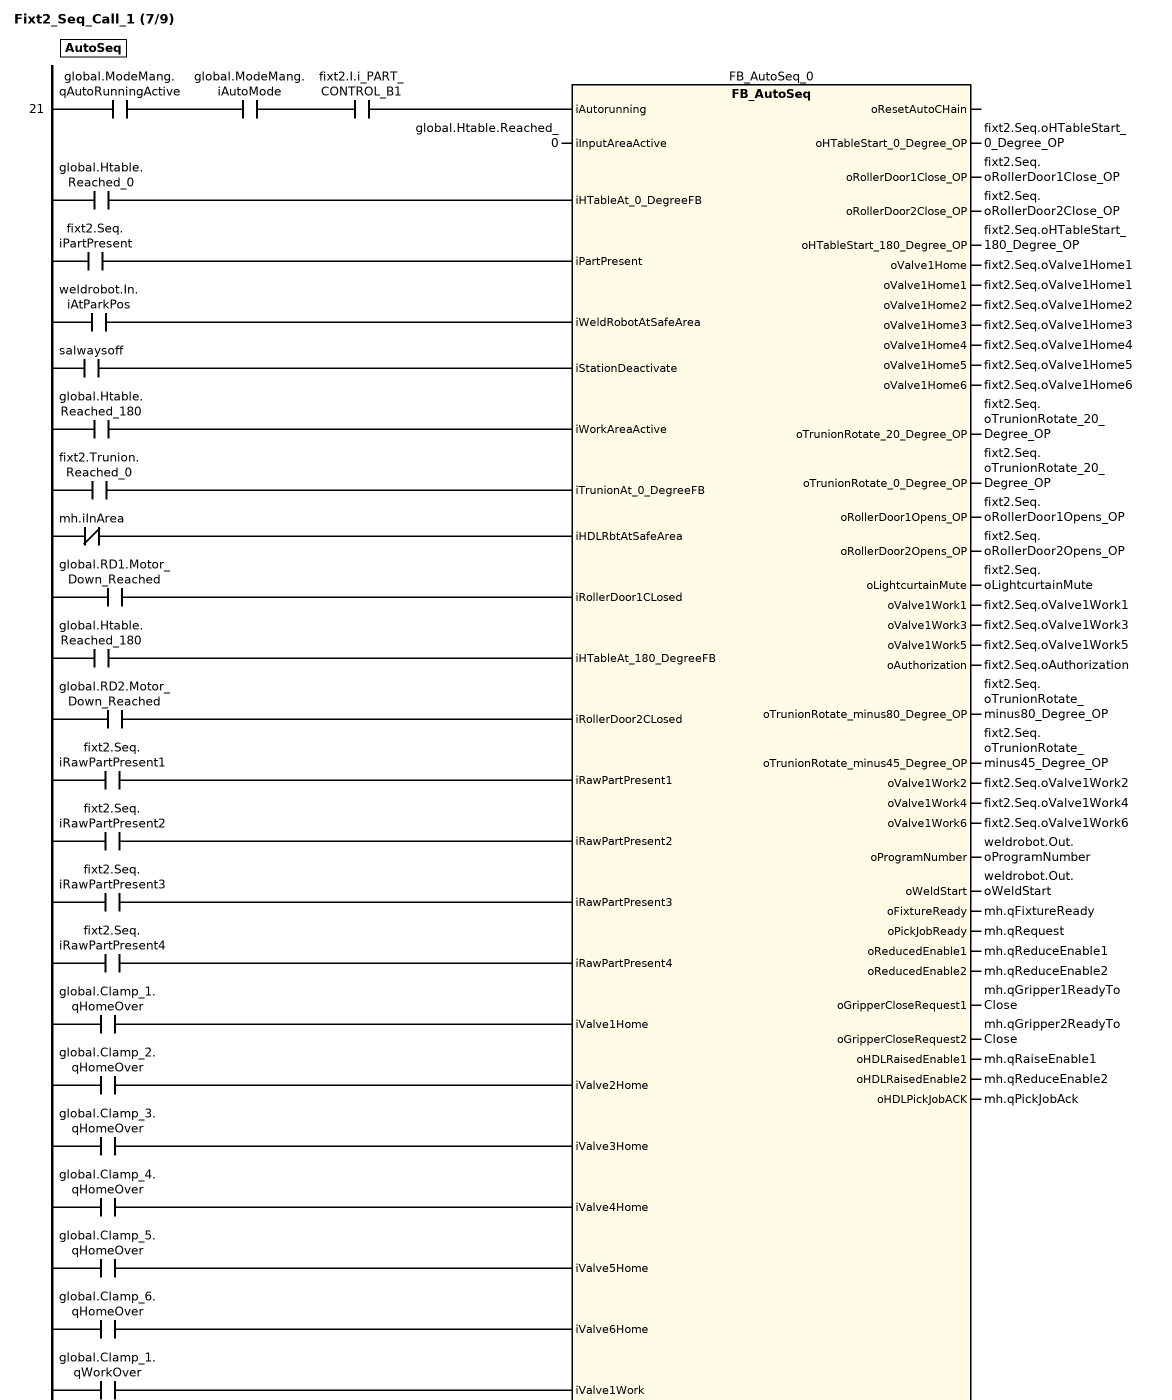
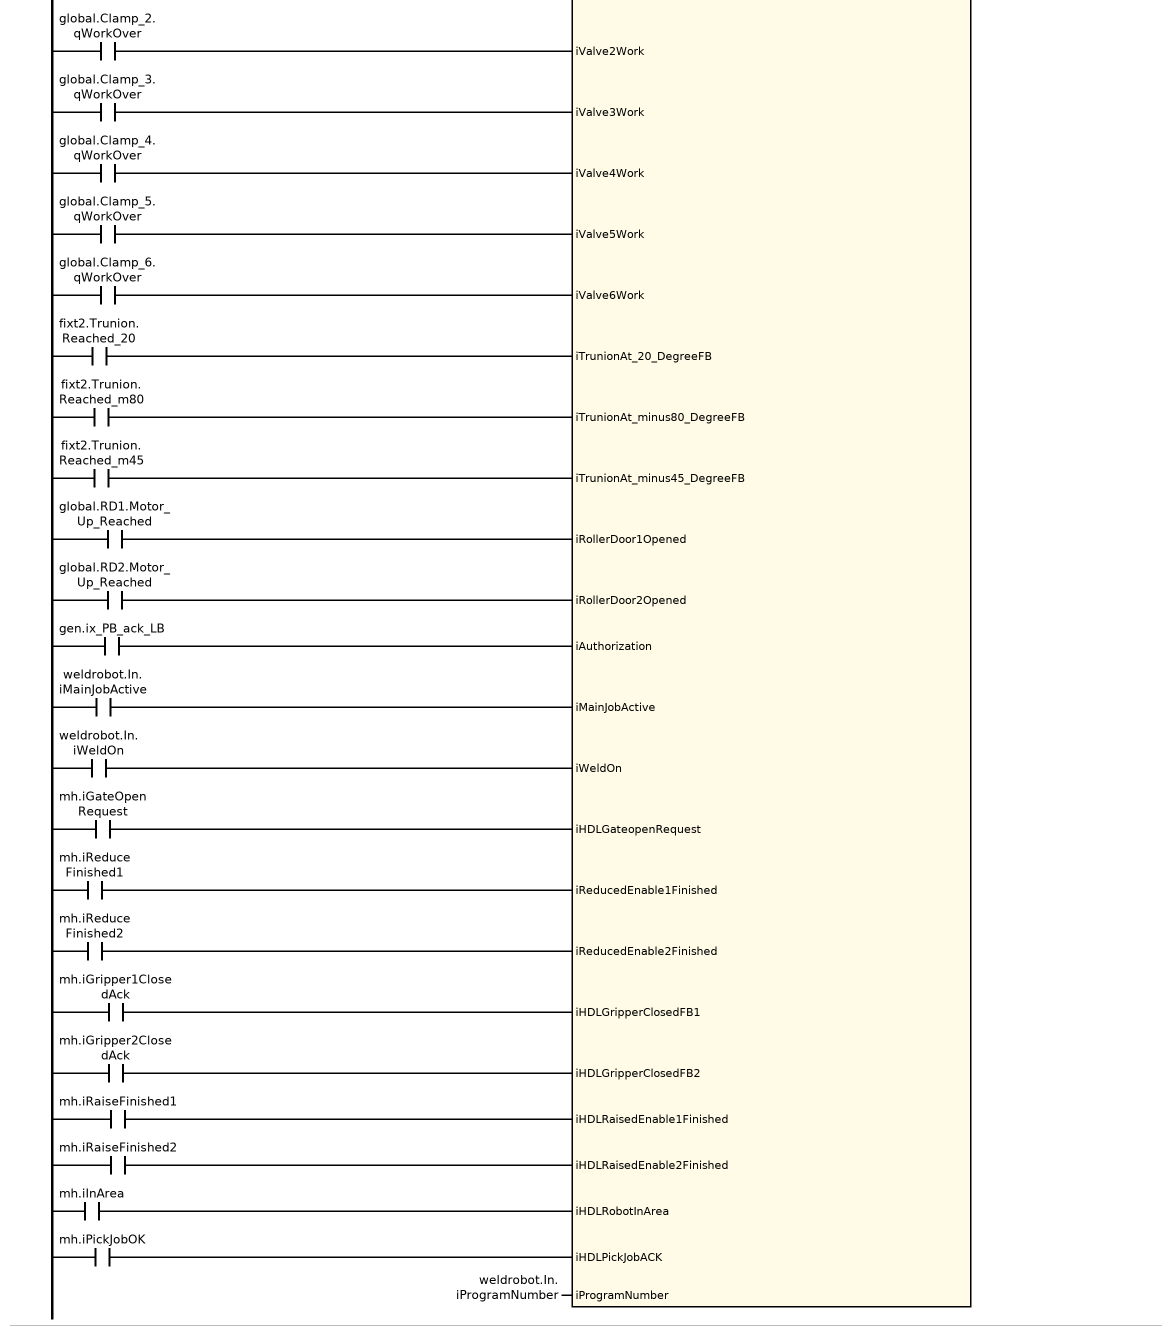
// NETWORK 21
AutoSeq:
FB_AutoSeq_0(
    iAutorunning := global.ModeMang.qAutoRunningActive AND global.ModeMang.iAutoMode AND fixt2.I.i_PART_CONTROL_B1,
    iInputAreaActive := global.Htable.Reached_0,
    iHTableAt_0_DegreeFB := global.Htable.Reached_0,
    iPartPresent := fixt2.Seq.iPartPresent,
    iWeldRobotAtSafeArea := weldrobot.In.iAtParkPos,
    iStationDeactivate := salwaysoff,
    iWorkAreaActive := global.Htable.Reached_180,
    iTrunionAt_0_DegreeFB := fixt2.Trunion.Reached_0,
    iHDLRbtAtSafeArea := NOT mh.iInArea,
    iRollerDoor1CLosed := global.RD1.Motor_Down_Reached,
    iHTableAt_180_DegreeFB := global.Htable.Reached_180,
    iRollerDoor2CLosed := global.RD2.Motor_Down_Reached,
    iRawPartPresent1 := fixt2.Seq.iRawPartPresent1,
    iRawPartPresent2 := fixt2.Seq.iRawPartPresent2,
    iRawPartPresent3 := fixt2.Seq.iRawPartPresent3,
    iRawPartPresent4 := fixt2.Seq.iRawPartPresent4,
    iValve1Home := global.Clamp_1.qHomeOver,
    iValve2Home := global.Clamp_2.qHomeOver,
    iValve3Home := global.Clamp_3.qHomeOver,
    iValve4Home := global.Clamp_4.qHomeOver,
    iValve5Home := global.Clamp_5.qHomeOver,
    iValve6Home := global.Clamp_6.qHomeOver,
    iValve1Work := global.Clamp_1.qWorkOver,
    iValve2Work := global.Clamp_2.qWorkOver,
    iValve3Work := global.Clamp_3.qWorkOver,
    iValve4Work := global.Clamp_4.qWorkOver,
    iValve5Work := global.Clamp_5.qWorkOver,
    iValve6Work := global.Clamp_6.qWorkOver,
    iTrunionAt_20_DegreeFB := fixt2.Trunion.Reached_20,
    iTrunionAt_minus80_DegreeFB := fixt2.Trunion.Reached_m80,
    iTrunionAt_minus45_DegreeFB := fixt2.Trunion.Reached_m45,
    iRollerDoor1Opened := global.RD1.Motor_Up_Reached,
    iRollerDoor2Opened := global.RD2.Motor_Up_Reached,
    iAuthorization := gen.ix_PB_ack_LB,
    iMainJobActive := weldrobot.In.iMainJobActive,
    iWeldOn := weldrobot.In.iWeldOn,
    iHDLGateopenRequest := mh.iGateOpenRequest,
    iReducedEnable1Finished := mh.iReduceFinished1,
    iReducedEnable2Finished := mh.iReduceFinished2,
    iHDLGripperClosedFB1 := mh.iGripper1ClosedAck,
    iHDLGripperClosedFB2 := mh.iGripper2ClosedAck,
    iHDLRaisedEnable1Finished := mh.iRaiseFinished1,
    iHDLRaisedEnable2Finished := mh.iRaiseFinished2,
    iHDLRobotInArea := mh.iInArea,
    iHDLPickJobACK := mh.iPickJobOK,
    iProgramNumber := weldrobot.In.iProgramNumber,
    oHTableStart_0_Degree_OP => fixt2.Seq.oHTableStart_0_Degree_OP,
    oRollerDoor1Close_OP => fixt2.Seq.oRollerDoor1Close_OP,
    oRollerDoor2Close_OP => fixt2.Seq.oRollerDoor2Close_OP,
    oHTableStart_180_Degree_OP => fixt2.Seq.oHTableStart_180_Degree_OP,
    oValve1Home => fixt2.Seq.oValve1Home1,
    oValve1Home1 => fixt2.Seq.oValve1Home1,
    oValve1Home2 => fixt2.Seq.oValve1Home2,
    oValve1Home3 => fixt2.Seq.oValve1Home3,
    oValve1Home4 => fixt2.Seq.oValve1Home4,
    oValve1Home5 => fixt2.Seq.oValve1Home5,
    oValve1Home6 => fixt2.Seq.oValve1Home6,
    oTrunionRotate_20_Degree_OP => fixt2.Seq.oTrunionRotate_20_Degree_OP,
    oTrunionRotate_0_Degree_OP => fixt2.Seq.oTrunionRotate_20_Degree_OP,
    oRollerDoor1Opens_OP => fixt2.Seq.oRollerDoor1Opens_OP,
    oRollerDoor2Opens_OP => fixt2.Seq.oRollerDoor2Opens_OP,
    oLightcurtainMute => fixt2.Seq.oLightcurtainMute,
    oValve1Work1 => fixt2.Seq.oValve1Work1,
    oValve1Work3 => fixt2.Seq.oValve1Work3,
    oValve1Work5 => fixt2.Seq.oValve1Work5,
    oAuthorization => fixt2.Seq.oAuthorization,
    oTrunionRotate_minus80_Degree_OP => fixt2.Seq.oTrunionRotate_minus80_Degree_OP,
    oTrunionRotate_minus45_Degree_OP => fixt2.Seq.oTrunionRotate_minus45_Degree_OP,
    oValve1Work2 => fixt2.Seq.oValve1Work2,
    oValve1Work4 => fixt2.Seq.oValve1Work4,
    oValve1Work6 => fixt2.Seq.oValve1Work6,
    oProgramNumber => weldrobot.Out.oProgramNumber,
    oWeldStart => weldrobot.Out.oWeldStart,
    oFixtureReady => mh.qFixtureReady,
    oPickJobReady => mh.qRequest,
    oReducedEnable1 => mh.qReduceEnable1,
    oReducedEnable2 => mh.qReduceEnable2,
    oGripperCloseRequest1 => mh.qGripper1ReadyToClose,
    oGripperCloseRequest2 => mh.qGripper2ReadyToClose,
    oHDLRaisedEnable1 => mh.qRaiseEnable1,
    oHDLRaisedEnable2 => mh.qReduceEnable2,
    oHDLPickJobACK => mh.qPickJobAck); // FB_AutoSeq

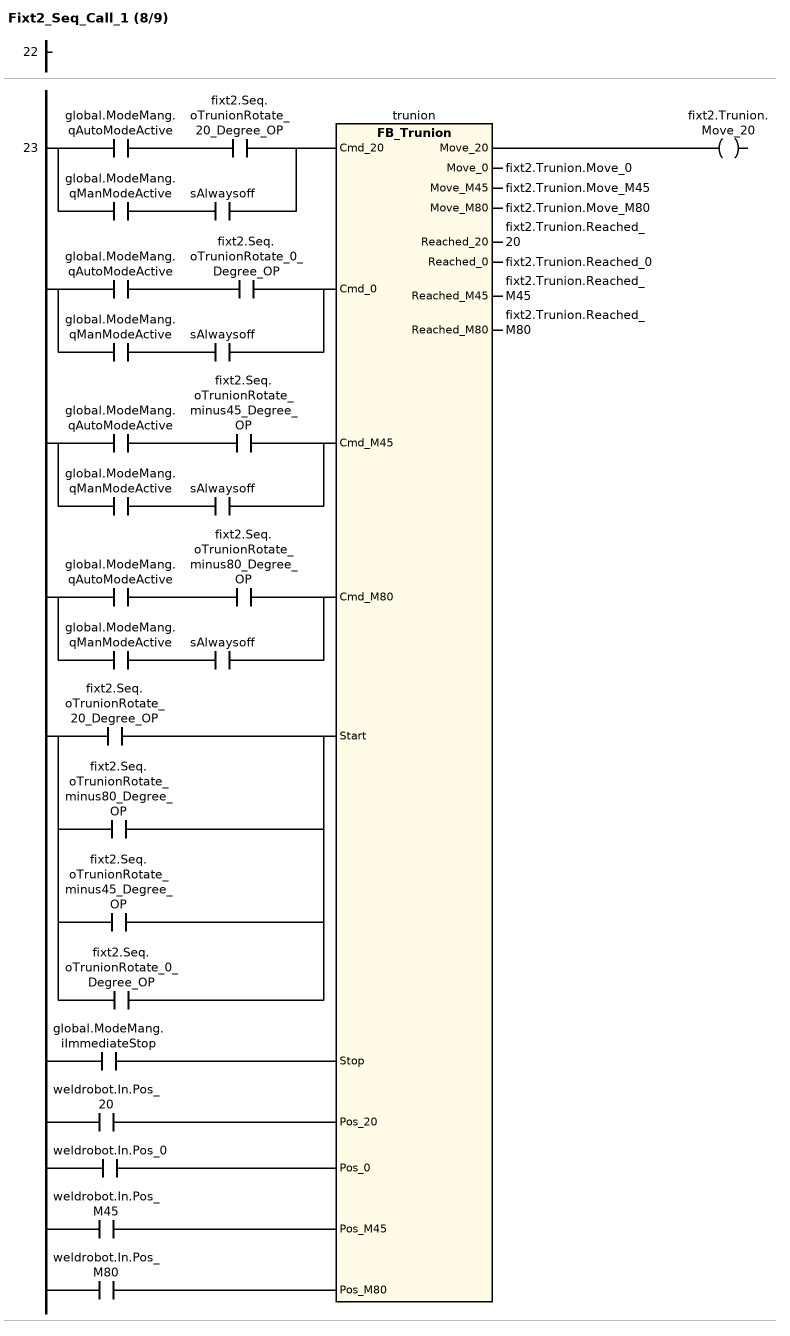
// NETWORK 22

// NETWORK 23
trunion(
    Cmd_20 := global.ModeMang.qAutoModeActive AND fixt2.Seq.oTrunionRotate_20_Degree_OP OR global.ModeMang.qManModeActive AND sAlwaysoff,
    Cmd_0 := global.ModeMang.qAutoModeActive AND fixt2.Seq.oTrunionRotate_0_Degree_OP OR global.ModeMang.qManModeActive AND sAlwaysoff,
    Cmd_M45 := global.ModeMang.qAutoModeActive AND fixt2.Seq.oTrunionRotate_minus45_Degree_OP OR global.ModeMang.qManModeActive AND sAlwaysoff,
    Cmd_M80 := global.ModeMang.qAutoModeActive AND fixt2.Seq.oTrunionRotate_minus80_Degree_OP OR global.ModeMang.qManModeActive AND sAlwaysoff,
    Start := fixt2.Seq.oTrunionRotate_20_Degree_OP OR fixt2.Seq.oTrunionRotate_minus80_Degree_OP OR fixt2.Seq.oTrunionRotate_minus45_Degree_OP OR fixt2.Seq.oTrunionRotate_0_Degree_OP,
    Stop := global.ModeMang.iImmediateStop,
    Pos_20 := weldrobot.In.Pos_20,
    Pos_0 := weldrobot.In.Pos_0,
    Pos_M45 := weldrobot.In.Pos_M45,
    Pos_M80 := weldrobot.In.Pos_M80,
    Move_0 => fixt2.Trunion.Move_0,
    Move_M45 => fixt2.Trunion.Move_M45,
    Move_M80 => fixt2.Trunion.Move_M80,
    Reached_20 => fixt2.Trunion.Reached_20,
    Reached_0 => fixt2.Trunion.Reached_0,
    Reached_M45 => fixt2.Trunion.Reached_M45,
    Reached_M80 => fixt2.Trunion.Reached_M80); // FB_Trunion
fixt2.Trunion.Move_20 := trunion.Move_20;

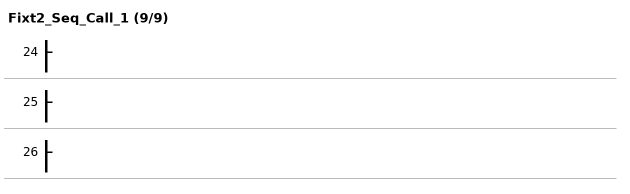
// NETWORK 24

// NETWORK 25

// NETWORK 26

END_PROGRAM

